    R369_2_I_RB_SP_1_14 AT %MW84091.14 : BOOL; (* R369_2_I_RB_SP_1_14 *)
    R369_2_I_RB_SP_1_15 AT %MW84091.15 : BOOL; (* R369_2_I_RB_SP_1_15 *)
    R369_2_I_RB_TC_이상 AT %MW84092.8 : BOOL; (* R369_2_I_RB_TC_이상 *)
    R369_2_I_RB_TIP_CHANGE AT %MW84093.13 : BOOL; (* R369_2_I_RB_TIP_CHANGE *)
    R369_2_I_RB_TIP_DRESSING AT %MW84090.7 : BOOL; (* R369_2_I_RB_TIP_DRESSING *)
    R369_2_I_RB__PLT_카운터리셋완료 AT %MW84093.10 : BOOL; (* R369_2_I_RB__PLT_카운터리셋완료 *)
    R369_2_I_RB_공기압_이상 AT %MW84092.9 : BOOL; (* R369_2_I_RB_공기압_이상 *)
    R369_2_I_RB_냉각수_이상 AT %MW84092.10 : BOOL; (* R369_2_I_RB_냉각수_이상 *)
    R369_2_I_RB_비상정지_NC AT %MW84090.8 : BOOL; (* R369_2_I_RB_비상정지_NC *)
    R369_2_I_RB_비전이상 AT %MW84092.14 : BOOL; (* R369_2_I_RB_비전이상 *)
    R369_2_I_RB_상호인터록_INT1 AT %MW84093.0 : BOOL; (* R369_2_I_RB_상호인터록_INT1 *)
    R369_2_I_RB_상호인터록_INT2 AT %MW84093.1 : BOOL; (* R369_2_I_RB_상호인터록_INT2 *)
    R369_2_I_RB_상호인터록_INT3 AT %MW84093.2 : BOOL; (* R369_2_I_RB_상호인터록_INT3 *)
    R369_2_I_RB_상호인터록_INT4 AT %MW84093.3 : BOOL; (* R369_2_I_RB_상호인터록_INT4 *)
    R369_2_I_RB_상호인터록_INT5 AT %MW84093.4 : BOOL; (* R369_2_I_RB_상호인터록_INT5 *)
    R369_2_I_RB_상호인터록_INT6 AT %MW84093.5 : BOOL; (* R369_2_I_RB_상호인터록_INT6 *)
    R369_2_I_RB_상호인터록_INT7 AT %MW84093.6 : BOOL; (* R369_2_I_RB_상호인터록_INT7 *)
    R369_2_I_RB_상호인터록_INT8 AT %MW84093.7 : BOOL; (* R369_2_I_RB_상호인터록_INT8 *)
    R369_2_I_RB_실러이상 AT %MW84092.13 : BOOL; (* R369_2_I_RB_실러이상 *)
    R369_2_I_RB_용접카운터이상 AT %MW84092.15 : BOOL; (* R369_2_I_RB_용접카운터이상 *)
    R369_2_I_RB_용접타점수 AT %MW84095 : WORD; (* R369_2_I_RB_용접타점수 *)
    R369_2_I_RB_운전준비 AT %MW84090.3 : BOOL; (* R369_2_I_RB_운전준비 *)
    R369_2_I_RB_원위치 AT %MW84090.0 : BOOL; (* R369_2_I_RB_원위치 *)
    R369_2_I_RB_이상리셋 AT %MW84090.2 : BOOL; (* R369_2_I_RB_이상리셋 *)
    R369_2_I_RB_자동 AT %MW84090.4 : BOOL; (* R369_2_I_RB_자동 *)
    R369_2_I_RB_자동기동 AT %MW84090.5 : BOOL; (* R369_2_I_RB_자동기동 *)
    R369_2_I_RB_최종_작업완료 AT %MW84090.1 : BOOL; (* R369_2_I_RB_최종_작업완료 *)
    R369_2_I_RB_통신이상 AT %MW84092.12 : BOOL; (* R369_2_I_RB_통신이상 *)
    R369_2_M_I_RB_1차_작업완료 AT %MW20091.2 : BOOL; (* R369_2_M_I_RB_1차_작업완료 *)
    R369_2_M_I_RB_2차_작업완료 AT %MW20091.3 : BOOL; (* R369_2_M_I_RB_2차_작업완료 *)
    R369_2_M_I_RB_3차_작업완료 AT %MW20091.4 : BOOL; (* R369_2_M_I_RB_3차_작업완료 *)
    R369_2_M_I_RB_4차_작업완료 AT %MW20091.5 : BOOL; (* R369_2_M_I_RB_4차_작업완료 *)
    R369_2_M_I_RB_5차_작업완료 AT %MW20091.6 : BOOL; (* R369_2_M_I_RB_5차_작업완료 *)
    R369_2_M_I_RB_6차_작업완료 AT %MW20091.7 : BOOL; (* R369_2_M_I_RB_6차_작업완료 *)
    R369_2_M_I_RB_7차_작업완료 AT %MW20091.8 : BOOL; (* R369_2_M_I_RB_7차_작업완료 *)
    R369_2_M_I_RB_PAUSE_보조 AT %MW20090.5 : BOOL; (* R369_2_M_I_RB_PAUSE_보조 *)
    R369_2_M_I_RB_PLC_RUN_CHK_이상 AT %MW20090.7 : BOOL; (* R369_2_M_I_RB_PLC_RUN_CHK_이상 *)
    R369_2_M_I_RB_간섭무_1 AT %MW20092.0 : BOOL; (* R369_2_M_I_RB_간섭무_1 *)
    R369_2_M_I_RB_간섭무_10 AT %MW20092.9 : BOOL; (* R369_2_M_I_RB_간섭무_10 *)
    R369_2_M_I_RB_간섭무_11 AT %MW20092.10 : BOOL; (* R369_2_M_I_RB_간섭무_11 *)
    R369_2_M_I_RB_간섭무_12 AT %MW20092.11 : BOOL; (* R369_2_M_I_RB_간섭무_12 *)
    R369_2_M_I_RB_간섭무_2 AT %MW20092.1 : BOOL; (* R369_2_M_I_RB_간섭무_2 *)
    R369_2_M_I_RB_간섭무_3 AT %MW20092.2 : BOOL; (* R369_2_M_I_RB_간섭무_3 *)
    R369_2_M_I_RB_간섭무_4 AT %MW20092.3 : BOOL; (* R369_2_M_I_RB_간섭무_4 *)
    R369_2_M_I_RB_간섭무_5 AT %MW20092.4 : BOOL; (* R369_2_M_I_RB_간섭무_5 *)
    R369_2_M_I_RB_간섭무_6 AT %MW20092.5 : BOOL; (* R369_2_M_I_RB_간섭무_6 *)
    R369_2_M_I_RB_간섭무_7 AT %MW20092.6 : BOOL; (* R369_2_M_I_RB_간섭무_7 *)
    R369_2_M_I_RB_간섭무_8 AT %MW20092.7 : BOOL; (* R369_2_M_I_RB_간섭무_8 *)
    R369_2_M_I_RB_간섭무_9 AT %MW20092.8 : BOOL; (* R369_2_M_I_RB_간섭무_9 *)
    R369_2_M_I_RB_비상정지 AT %MW20090.4 : BOOL; (* R369_2_M_I_RB_비상정지 *)
    R369_2_M_I_RB_운전준비 AT %MW20090.0 : BOOL; (* R369_2_M_I_RB_운전준비 *)
    R369_2_M_I_RB_원위치 AT %MW20090.3 : BOOL; (* R369_2_M_I_RB_원위치 *)
    R369_2_M_I_RB_이상 AT %MW20090.2 : BOOL; (* R369_2_M_I_RB_이상 *)
    R369_2_M_I_RB_자동 AT %MW20090.1 : BOOL; (* R369_2_M_I_RB_자동 *)
    R369_2_M_I_RB_최종작업완료 AT %MW20091.0 : BOOL; (* R369_2_M_I_RB_최종작업완료 *)
    R369_2_M_I_RB_프로그램_이상 AT %MW20090.6 : BOOL; (* R369_2_M_I_RB_프로그램_이상 *)
    R369_2_M_O_RB_1_CYCLE_SET AT %MW21090.3 : BOOL; (* R369_2_M_O_RB_1_CYCLE_SET *)
    R369_2_M_O_RB_1_CYCLE_리셋 AT %MW21090.4 : BOOL; (* R369_2_M_O_RB_1_CYCLE_리셋 *)
    R369_2_M_O_RB_1차_작업완료_리셋 AT %MW21092.0 : BOOL; (* R369_2_M_O_RB_1차_작업완료_리셋 *)
    R369_2_M_O_RB_2차_작업완료_리셋 AT %MW21092.1 : BOOL; (* R369_2_M_O_RB_2차_작업완료_리셋 *)
    R369_2_M_O_RB_2차_진입OK AT %MW21091.8 : BOOL; (* R369_2_M_O_RB_2차_진입OK *)
    R369_2_M_O_RB_3차_작업완료_리셋 AT %MW21092.2 : BOOL; (* R369_2_M_O_RB_3차_작업완료_리셋 *)
    R369_2_M_O_RB_3차_진입OK AT %MW21091.9 : BOOL; (* R369_2_M_O_RB_3차_진입OK *)
    R369_2_M_O_RB_4차_작업완료_리셋 AT %MW21092.3 : BOOL; (* R369_2_M_O_RB_4차_작업완료_리셋 *)
    R369_2_M_O_RB_4차_진입OK AT %MW21091.10 : BOOL; (* R369_2_M_O_RB_4차_진입OK *)
    R369_2_M_O_RB_5차_작업완료_리셋 AT %MW21092.4 : BOOL; (* R369_2_M_O_RB_5차_작업완료_리셋 *)
    R369_2_M_O_RB_5차_진입OK AT %MW21091.11 : BOOL; (* R369_2_M_O_RB_5차_진입OK *)
    R369_2_M_O_RB_6차_작업완료_리셋 AT %MW21092.5 : BOOL; (* R369_2_M_O_RB_6차_작업완료_리셋 *)
    R369_2_M_O_RB_6차_진입OK AT %MW21091.12 : BOOL; (* R369_2_M_O_RB_6차_진입OK *)
    R369_2_M_O_RB_7차_작업완료_리셋 AT %MW21092.6 : BOOL; (* R369_2_M_O_RB_7차_작업완료_리셋 *)
    R369_2_M_O_RB_7차_진입OK AT %MW21091.13 : BOOL; (* R369_2_M_O_RB_7차_진입OK *)
    R369_2_M_O_RB_ATD_OK AT %MW21090.6 : BOOL; (* R369_2_M_O_RB_ATD_OK *)
    R369_2_M_O_RB_PLT_10_진입OK AT %MW21093.10 : BOOL; (* R369_2_M_O_RB_PLT_10_진입OK *)
    R369_2_M_O_RB_PLT_11_진입OK AT %MW21093.11 : BOOL; (* R369_2_M_O_RB_PLT_11_진입OK *)
    R369_2_M_O_RB_PLT_12_진입OK AT %MW21093.12 : BOOL; (* R369_2_M_O_RB_PLT_12_진입OK *)
    R369_2_M_O_RB_PLT_1_진입OK AT %MW21093.1 : BOOL; (* R369_2_M_O_RB_PLT_1_진입OK *)
    R369_2_M_O_RB_PLT_2_진입OK AT %MW21093.2 : BOOL; (* R369_2_M_O_RB_PLT_2_진입OK *)
    R369_2_M_O_RB_PLT_3_진입OK AT %MW21093.3 : BOOL; (* R369_2_M_O_RB_PLT_3_진입OK *)
    R369_2_M_O_RB_PLT_4_진입OK AT %MW21093.4 : BOOL; (* R369_2_M_O_RB_PLT_4_진입OK *)
    R369_2_M_O_RB_PLT_5_진입OK AT %MW21093.5 : BOOL; (* R369_2_M_O_RB_PLT_5_진입OK *)
    R369_2_M_O_RB_PLT_6_진입OK AT %MW21093.6 : BOOL; (* R369_2_M_O_RB_PLT_6_진입OK *)
    R369_2_M_O_RB_PLT_7_진입OK AT %MW21093.7 : BOOL; (* R369_2_M_O_RB_PLT_7_진입OK *)
    R369_2_M_O_RB_PLT_8_진입OK AT %MW21093.8 : BOOL; (* R369_2_M_O_RB_PLT_8_진입OK *)
    R369_2_M_O_RB_PLT_9_진입OK AT %MW21093.9 : BOOL; (* R369_2_M_O_RB_PLT_9_진입OK *)
    R369_2_M_O_RB_PLT_카운터리셋_보조 AT %MW21090.10 : BOOL; (* R369_2_M_O_RB_PLT_카운터리셋_보조 *)
    R369_2_M_O_RB_PROG_NO AT %MW21094 : WORD;
    R369_2_M_O_RB_RESTART_OK AT %MW21090.2 : BOOL; (* R369_2_M_O_RB_RESTART_OK *)
    R369_2_M_O_RB_START_OK AT %MW21090.0 : BOOL; (* R369_2_M_O_RB_START_OK *)
    R369_2_M_O_RB_TEST_MODE_5000회 AT %MW21090.12 : BOOL; (* R369_2_M_O_RB_TEST_MODE_5000회 *)
    R369_2_M_O_RB_TIP_교체_시작 AT %MW21090.7 : BOOL; (* R369_2_M_O_RB_TIP_교체_시작 *)
    R369_2_M_O_RB_TIP_교체_완료 AT %MW21090.8 : BOOL; (* R369_2_M_O_RB_TIP_교체_완료 *)
    R369_2_M_O_RB_VIP_MODE AT %MW21090.11 : BOOL; (* R369_2_M_O_RB_VIP_MODE *)
    R369_2_M_O_RB_냉각수_차단_요청 AT %MW21090.9 : BOOL; (* R369_2_M_O_RB_냉각수_차단_요청 *)
    R369_2_M_O_RB_진입OK_AX차종 AT %MW21091.0 : BOOL; (* R369_2_M_O_RB_진입OK_AX차종 *)
    R369_2_M_O_RB_진입OK_B차종 AT %MW21091.1 : BOOL; (* R369_2_M_O_RB_진입OK_B차종 *)
    R369_2_M_O_RB_진입OK_C차종 AT %MW21091.2 : BOOL; (* R369_2_M_O_RB_진입OK_C차종 *)
    R369_2_M_O_RB_진입OK_D차종 AT %MW21091.3 : BOOL; (* R369_2_M_O_RB_진입OK_D차종 *)
    R369_2_M_O_RB_진입OK_E차종 AT %MW21091.4 : BOOL; (* R369_2_M_O_RB_진입OK_E차종 *)
    R369_2_M_O_RB_진입OK_F차종 AT %MW21091.5 : BOOL; (* R369_2_M_O_RB_진입OK_F차종 *)
    R369_2_M_O_RB_진입OK_G차종 AT %MW21091.6 : BOOL; (* R369_2_M_O_RB_진입OK_G차종 *)
    R369_2_M_O_RB_진입OK_H차종 AT %MW21091.7 : BOOL; (* R369_2_M_O_RB_진입OK_H차종 *)
    R369_2_M_O_RB_최종_작업완료_리셋 AT %MW21090.5 : BOOL; (* R369_2_M_O_RB_최종_작업완료_리셋 *)
    R369_2_M_O_RB_프로그램_OK AT %MW21090.1 : BOOL; (* R369_2_M_O_RB_프로그램_OK *)
    R369_2_O_RB_0_5S_통신_CHK AT %MW94093.14 : BOOL; (* R369_2_O_RB_0_5S_통신_CHK *)
    R369_2_O_RB_2차_진입OK AT %MW94091.8 : BOOL; (* R369_2_O_RB_2차_진입OK *)
    R369_2_O_RB_3차_진입OK AT %MW94091.9 : BOOL; (* R369_2_O_RB_3차_진입OK *)
    R369_2_O_RB_4차_진입OK AT %MW94091.10 : BOOL; (* R369_2_O_RB_4차_진입OK *)
    R369_2_O_RB_5차_진입OK AT %MW94091.11 : BOOL; (* R369_2_O_RB_5차_진입OK *)
    R369_2_O_RB_6차_진입OK AT %MW94091.12 : BOOL; (* R369_2_O_RB_6차_진입OK *)
    R369_2_O_RB_7차_진입OK AT %MW94091.13 : BOOL; (* R369_2_O_RB_7차_진입OK *)
    R369_2_O_RB_AX_1차_진입OK AT %MW94091.0 : BOOL; (* R369_2_O_RB_AX_1차_진입OK *)
    R369_2_O_RB_B_1차_진입OK AT %MW94091.1 : BOOL; (* R369_2_O_RB_B_1차_진입OK *)
    R369_2_O_RB_C_1차_진입OK AT %MW94091.2 : BOOL; (* R369_2_O_RB_C_1차_진입OK *)
    R369_2_O_RB_D_1차_진입OK AT %MW94091.3 : BOOL; (* R369_2_O_RB_D_1차_진입OK *)
    R369_2_O_RB_EACH_작업완료_리셋 AT %MW94090.14 : BOOL; (* R369_2_O_RB_EACH_작업완료_리셋 *)
    R369_2_O_RB_EXT_READY AT %MW94090.11 : BOOL; (* R369_2_O_RB_EXT_READY *)
    R369_2_O_RB_E_1차_진입OK AT %MW94091.4 : BOOL; (* R369_2_O_RB_E_1차_진입OK *)
    R369_2_O_RB_F_1차_진입OK AT %MW94091.5 : BOOL; (* R369_2_O_RB_F_1차_진입OK *)
    R369_2_O_RB_GATE_OPEN_NC AT %MW94093.11 : BOOL; (* R369_2_O_RB_GATE_OPEN_NC *)
    R369_2_O_RB_G_1차_진입OK AT %MW94091.6 : BOOL; (* R369_2_O_RB_G_1차_진입OK *)
    R369_2_O_RB_H_1차_진입OK AT %MW94091.7 : BOOL; (* R369_2_O_RB_H_1차_진입OK *)
    R369_2_O_RB_OUTPUT AT %MW94090 : ARRAY[0..3] OF WORD; (* R369_2_O_RB_OUTPUT *)
    R369_2_O_RB_PAUSE_NC AT %MW94090.13 : BOOL; (* R369_2_O_RB_PAUSE_NC *)
    R369_2_O_RB_PLT10_진입OK AT %MW94092.9 : BOOL; (* R369_2_O_RB_PLT10_진입OK *)
    R369_2_O_RB_PLT11_진입OK AT %MW94092.10 : BOOL; (* R369_2_O_RB_PLT11_진입OK *)
    R369_2_O_RB_PLT12_진입OK AT %MW94092.11 : BOOL; (* R369_2_O_RB_PLT12_진입OK *)
    R369_2_O_RB_PLT1_진입OK AT %MW94092.0 : BOOL; (* R369_2_O_RB_PLT1_진입OK *)
    R369_2_O_RB_PLT2_진입OK AT %MW94092.1 : BOOL; (* R369_2_O_RB_PLT2_진입OK *)
    R369_2_O_RB_PLT3_진입OK AT %MW94092.2 : BOOL; (* R369_2_O_RB_PLT3_진입OK *)
    R369_2_O_RB_PLT4_진입OK AT %MW94092.3 : BOOL; (* R369_2_O_RB_PLT4_진입OK *)
    R369_2_O_RB_PLT5_진입OK AT %MW94092.4 : BOOL; (* R369_2_O_RB_PLT5_진입OK *)
    R369_2_O_RB_PLT6_진입OK AT %MW94092.5 : BOOL; (* R369_2_O_RB_PLT6_진입OK *)
    R369_2_O_RB_PLT7_진입OK AT %MW94092.6 : BOOL; (* R369_2_O_RB_PLT7_진입OK *)
    R369_2_O_RB_PLT8_진입OK AT %MW94092.7 : BOOL; (* R369_2_O_RB_PLT8_진입OK *)
    R369_2_O_RB_PLT9_진입OK AT %MW94092.8 : BOOL; (* R369_2_O_RB_PLT9_진입OK *)
    R369_2_O_RB_PLT_카운터_리셋_요구 AT %MW94093.10 : BOOL; (* R369_2_O_RB_PLT_카운터_리셋_요구 *)
    R369_2_O_RB_PROG_선택1 AT %MW94090.0 : BOOL; (* R369_2_O_RB_PROG_선택1 *)
    R369_2_O_RB_PROG_선택128 AT %MW94090.7 : BOOL; (* R369_2_O_RB_PROG_선택128 *)
    R369_2_O_RB_PROG_선택16 AT %MW94090.4 : BOOL; (* R369_2_O_RB_PROG_선택16 *)
    R369_2_O_RB_PROG_선택2 AT %MW94090.1 : BOOL; (* R369_2_O_RB_PROG_선택2 *)
    R369_2_O_RB_PROG_선택32 AT %MW94090.5 : BOOL; (* R369_2_O_RB_PROG_선택32 *)
    R369_2_O_RB_PROG_선택4 AT %MW94090.2 : BOOL; (* R369_2_O_RB_PROG_선택4 *)
    R369_2_O_RB_PROG_선택64 AT %MW94090.6 : BOOL; (* R369_2_O_RB_PROG_선택64 *)
    R369_2_O_RB_PROG_선택8 AT %MW94090.3 : BOOL; (* R369_2_O_RB_PROG_선택8 *)
    R369_2_O_RB_SP_1_14 AT %MW94091.14 : BOOL; (* R369_2_O_RB_SP_1_14 *)
    R369_2_O_RB_SP_1_15 AT %MW94091.15 : BOOL; (* R369_2_O_RB_SP_1_15 *)
    R369_2_O_RB_SP_2_12 AT %MW94092.12 : BOOL; (* R369_2_O_RB_SP_2_12 *)
    R369_2_O_RB_SP_2_13 AT %MW94092.13 : BOOL; (* R369_2_O_RB_SP_2_13 *)
    R369_2_O_RB_SP_2_14 AT %MW94092.14 : BOOL; (* R369_2_O_RB_SP_2_14 *)
    R369_2_O_RB_SP_5000TH_ON AT %MW94092.15 : BOOL; (* R369_2_O_RB_SP_5000TH_ON *)
    R369_2_O_RB_TIP_CHANGE_END AT %MW94093.9 : BOOL; (* R369_2_O_RB_TIP_CHANGE_END *)
    R369_2_O_RB_TIP_CHANGE_START AT %MW94093.8 : BOOL; (* R369_2_O_RB_TIP_CHANGE_START *)
    R369_2_O_RB_TIP_DRESS_SATRT AT %MW94090.12 : BOOL; (* R369_2_O_RB_TIP_DRESS_SATRT *)
    R369_2_O_RB_VIP_MODE AT %MW94093.15 : BOOL; (* R369_2_O_RB_VIP_MODE *)
    R369_2_O_RB_기동 AT %MW94090.9 : BOOL; (* R369_2_O_RB_기동 *)
    R369_2_O_RB_냉각수차단 AT %MW94090.15 : BOOL; (* R369_2_O_RB_냉각수차단 *)
    R369_2_O_RB_부저정지 AT %MW94093.13 : BOOL; (* R369_2_O_RB_부저정지 *)
    R369_2_O_RB_비상정지_NC AT %MW94093.12 : BOOL; (* R369_2_O_RB_비상정지_NC *)
    R369_2_O_RB_상호인터록_INT1 AT %MW94093.0 : BOOL; (* R369_2_O_RB_상호인터록_INT1 *)
    R369_2_O_RB_상호인터록_INT2 AT %MW94093.1 : BOOL; (* R369_2_O_RB_상호인터록_INT2 *)
    R369_2_O_RB_상호인터록_INT3 AT %MW94093.2 : BOOL; (* R369_2_O_RB_상호인터록_INT3 *)
    R369_2_O_RB_상호인터록_INT4 AT %MW94093.3 : BOOL; (* R369_2_O_RB_상호인터록_INT4 *)
    R369_2_O_RB_상호인터록_INT5 AT %MW94093.4 : BOOL; (* R369_2_O_RB_상호인터록_INT5 *)
    R369_2_O_RB_상호인터록_INT6 AT %MW94093.5 : BOOL; (* R369_2_O_RB_상호인터록_INT6 *)
    R369_2_O_RB_상호인터록_INT7 AT %MW94093.6 : BOOL; (* R369_2_O_RB_상호인터록_INT7 *)
    R369_2_O_RB_상호인터록_INT8 AT %MW94093.7 : BOOL; (* R369_2_O_RB_상호인터록_INT8 *)
    R369_2_O_RB_이상_리셋 AT %MW94090.10 : BOOL; (* R369_2_O_RB_이상_리셋 *)
    R369_2_O_RB_작업완료_리셋 AT %MW94090.8 : BOOL; (* R369_2_O_RB_작업완료_리셋 *)
    ROOF_RACK1_3_PLC_BOX_CP_TRIP AT %MW87401.15 : BOOL; (* ROOF RACK1 3 PLC BOX CP TRIP *)
    ROOF_RACK1_LC_정상1 AT %MW87403.0 : BOOL; (* ROOF RACK1 LC 정상1 *)
    ROOF_RACK1_LC_정상2 AT %MW87403.1 : BOOL; (* ROOF RACK1 LC 정상2 *)
    ROOF_RACK1_PRS_랙감지1 AT %MW87400.0 : BOOL; (* ROOF RACK1 PRS 랙감지1 *)
    ROOF_RACK1_PRS_랙감지2 AT %MW87400.1 : BOOL; (* ROOF RACK1 PRS 랙감지2 *)
    ROOF_RACK1_PRS_막장감지 AT %MW87400.2 : BOOL; (* ROOF RACK1 PRS 막장감지 *)
    ROOF_RACK1_발목감지_정상1 AT %MW87403.2 : BOOL; (* ROOF RACK1 발목감지 정상1 *)
    ROOF_RACK1_발목감지_정상2 AT %MW87403.3 : BOOL; (* ROOF RACK1 발목감지 정상2 *)
    ROOF_RACK2_LC_정상1 AT %MW87403.4 : BOOL; (* ROOF RACK2 LC 정상1 *)
    ROOF_RACK2_LC_정상2 AT %MW87403.5 : BOOL; (* ROOF RACK2 LC 정상2 *)
    ROOF_RACK2_PRS_랙감지1 AT %MW87400.8 : BOOL; (* ROOF RACK2 PRS 랙감지1 *)
    ROOF_RACK2_PRS_랙감지2 AT %MW87400.9 : BOOL; (* ROOF RACK2 PRS 랙감지2 *)
    ROOF_RACK2_PRS_막장감지 AT %MW87400.10 : BOOL; (* ROOF RACK2 PRS 막장감지 *)
    ROOF_RACK2_발목감지_정상1 AT %MW87403.6 : BOOL; (* ROOF RACK2 발목감지 정상1 *)
    ROOF_RACK2_발목감지_정상2 AT %MW87403.7 : BOOL; (* ROOF RACK2 발목감지 정상2 *)
    ROOF_RACK3_LC_정상1 AT %MW87403.8 : BOOL; (* ROOF RACK3 LC 정상1 *)
    ROOF_RACK3_LC_정상2 AT %MW87403.9 : BOOL; (* ROOF RACK3 LC 정상2 *)
    ROOF_RACK3_PRS_랙감지1 AT %MW87401.0 : BOOL; (* ROOF RACK3 PRS 랙감지1 *)
    ROOF_RACK3_PRS_랙감지2 AT %MW87401.1 : BOOL; (* ROOF RACK3 PRS 랙감지2 *)
    ROOF_RACK3_PRS_막장감지 AT %MW87401.2 : BOOL; (* ROOF RACK3 PRS 막장감지 *)
    ROOF_RACK3_발목감지_정상1 AT %MW87403.10 : BOOL; (* ROOF RACK3 발목감지 정상1 *)
    ROOF_RACK3_발목감지_정상2 AT %MW87403.11 : BOOL; (* ROOF RACK3 발목감지 정상2 *)
    ROOF_RACK4_6_PLC_BOX_CP_TRIP AT %MW87451.15 : BOOL; (* ROOF RACK4 6 PLC BOX CP TRIP *)
    ROOF_RACK4_LC_정상1 AT %MW87453.0 : BOOL; (* ROOF RACK4 LC 정상1 *)
    ROOF_RACK4_LC_정상2 AT %MW87453.1 : BOOL; (* ROOF RACK4 LC 정상2 *)
    ROOF_RACK4_PRS_랙감지1 AT %MW87450.0 : BOOL; (* ROOF RACK4 PRS 랙감지1 *)
    ROOF_RACK4_PRS_랙감지2 AT %MW87450.1 : BOOL; (* ROOF RACK4 PRS 랙감지2 *)
    ROOF_RACK4_PRS_막장감지 AT %MW87450.2 : BOOL; (* ROOF RACK4 PRS 막장감지 *)
    ROOF_RACK4_발목감지_정상1 AT %MW87453.2 : BOOL; (* ROOF RACK4 발목감지 정상1 *)
    ROOF_RACK4_발목감지_정상2 AT %MW87453.3 : BOOL; (* ROOF RACK4 발목감지 정상2 *)
    ROOF_RACK5_LC_정상1 AT %MW87453.4 : BOOL; (* ROOF RACK5 LC 정상1 *)
    ROOF_RACK5_LC_정상2 AT %MW87453.5 : BOOL; (* ROOF RACK5 LC 정상2 *)
    ROOF_RACK5_PRS_랙감지1 AT %MW87450.8 : BOOL; (* ROOF RACK5 PRS 랙감지1 *)
    ROOF_RACK5_PRS_랙감지2 AT %MW87450.9 : BOOL; (* ROOF RACK5 PRS 랙감지2 *)
    ROOF_RACK5_PRS_막장감지 AT %MW87450.10 : BOOL; (* ROOF RACK5 PRS 막장감지 *)
    ROOF_RACK5_발목감지_정상1 AT %MW87453.6 : BOOL; (* ROOF RACK5 발목감지 정상1 *)
    ROOF_RACK5_발목감지_정상2 AT %MW87453.7 : BOOL; (* ROOF RACK5 발목감지 정상2 *)
    ROOF_RACK6_LC_정상1 AT %MW87453.8 : BOOL; (* ROOF RACK6 LC 정상1 *)
    ROOF_RACK6_LC_정상2 AT %MW87453.9 : BOOL; (* ROOF RACK6 LC 정상2 *)
    ROOF_RACK6_PRS_랙감지1 AT %MW87451.0 : BOOL; (* ROOF RACK6 PRS 랙감지1 *)
    ROOF_RACK6_PRS_랙감지2 AT %MW87451.1 : BOOL; (* ROOF RACK6 PRS 랙감지2 *)
    ROOF_RACK6_PRS_막장감지 AT %MW87451.2 : BOOL; (* ROOF RACK6 PRS 막장감지 *)
    ROOF_RACK6_발목감지_정상1 AT %MW87453.10 : BOOL; (* ROOF RACK6 발목감지 정상1 *)
    ROOF_RACK6_발목감지_정상2 AT %MW87453.11 : BOOL; (* ROOF RACK6 발목감지 정상2 *)
    S362_6_INV1_BRAKE_CR_ON AT %MW95014.7 : BOOL; (* S362_6_INV1_BRAKE_CR_ON *)
    S362_6_INV1_MC_BRAKE_ON AT %MW85010.1 : BOOL; (* S362_6_INV1_MC_BRAKE_ON *)
    S362_6_INV1_NFB_ON AT %MW85013.0 : BOOL; (* S362_6_INV1_NFB_ON *)
    S362_6_INV1_NOMAL_OK AT %MW85010.0 : BOOL; (* S362_6_INV1_NOMAL_OK *)
    S362_6_INV1_RETURN AT %MW95014.1 : BOOL; (* S362_6_INV1_RETURN *)
    S362_6_INV1_SAFETY1_ON AT %MW95014.5 : BOOL; (* S362_6_INV1_SAFETY1_ON *)
    S362_6_INV1_SAFETY2_ON AT %MW95014.6 : BOOL; (* S362_6_INV1_SAFETY2_ON *)
    S362_6_INV1_TURN AT %MW95014.0 : BOOL; (* S362_6_INV1_TURN *)
    S362_6_INV1_이상_리셋 AT %MW95014.3 : BOOL; (* S362_6_INV1_이상_리셋 *)
    S362_6_INV2_BRAKE_CR_ON AT %MW95014.15 : BOOL; (* S362_6_INV2_BRAKE_CR_ON *)
    S362_6_INV2_MC_BRAKE_ON AT %MW85010.5 : BOOL; (* S362_6_INV2_MC_BRAKE_ON *)
    S362_6_INV2_NFB_ON AT %MW85013.1 : BOOL; (* S362_6_INV2_NFB_ON *)
    S362_6_INV2_NOMAL_OK AT %MW85010.4 : BOOL; (* S362_6_INV2_NOMAL_OK *)
    S362_6_INV2_RETURN AT %MW95014.9 : BOOL; (* S362_6_INV2_RETURN *)
    S362_6_INV2_SAFETY1_ON AT %MW95014.13 : BOOL; (* S362_6_INV2_SAFETY1_ON *)
    S362_6_INV2_SAFETY2_ON AT %MW95014.14 : BOOL; (* S362_6_INV2_SAFETY2_ON *)
    S362_6_INV2_TURN AT %MW95014.8 : BOOL; (* S362_6_INV2_TURN *)
    S362_6_INV2_이상_리셋 AT %MW95014.11 : BOOL; (* S362_6_INV2_이상_리셋 *)
    S362_6_INV3_BRAKE_CR_ON AT %MW95015.7 : BOOL; (* S362_6_INV3_BRAKE_CR_ON *)
    S362_6_INV3_MC_BRAKE_ON AT %MW85010.9 : BOOL; (* S362_6_INV3_MC_BRAKE_ON *)
    S362_6_INV3_NFB_ON AT %MW85013.2 : BOOL; (* S362_6_INV3_NFB_ON *)
    S362_6_INV3_NOMAL_OK AT %MW85010.8 : BOOL; (* S362_6_INV3_NOMAL_OK *)
    S362_6_INV3_RETURN AT %MW95015.1 : BOOL; (* S362_6_INV3_RETURN *)
    S362_6_INV3_SAFETY1_ON AT %MW95015.5 : BOOL; (* S362_6_INV3_SAFETY1_ON *)
    S362_6_INV3_SAFETY2_ON AT %MW95015.6 : BOOL; (* S362_6_INV3_SAFETY2_ON *)
    S362_6_INV3_TURN AT %MW95015.0 : BOOL; (* S362_6_INV3_TURN *)
    S362_6_INV3_이상_리셋 AT %MW95015.3 : BOOL; (* S362_6_INV3_이상_리셋 *)
    S362_6_INV4_BRAKE_CR_ON AT %MW95015.15 : BOOL; (* S362_6_INV4_BRAKE_CR_ON *)
    S362_6_INV4_MC_BRAKE_ON AT %MW85010.13 : BOOL; (* S362_6_INV4_MC_BRAKE_ON *)
    S362_6_INV4_NFB_ON AT %MW85013.3 : BOOL; (* S362_6_INV4_NFB_ON *)
    S362_6_INV4_NOMAL_OK AT %MW85010.12 : BOOL; (* S362_6_INV4_NOMAL_OK *)
    S362_6_INV4_RETURN AT %MW95015.9 : BOOL; (* S362_6_INV4_RETURN *)
    S362_6_INV4_SAFETY1_ON AT %MW95015.13 : BOOL; (* S362_6_INV4_SAFETY1_ON *)
    S362_6_INV4_SAFETY2_ON AT %MW95015.14 : BOOL; (* S362_6_INV4_SAFETY2_ON *)
    S362_6_INV4_TURN AT %MW95015.8 : BOOL; (* S362_6_INV4_TURN *)
    S362_6_INV4_이상_리셋 AT %MW95015.11 : BOOL; (* S362_6_INV4_이상_리셋 *)
    S362_6_INV_BRAKE_CP_OFF AT %MW85013.13 : BOOL; (* S362_6_INV_BRAKE_CP_OFF *)
    S362_6_INV_DC_CP_TRIP AT %MW85013.12 : BOOL; (* S362_6_INV_DC_CP_TRIP *)
    S362_6_INV_PS1_DC_OK AT %MW85013.14 : BOOL; (* S362_6_INV_PS1_DC_OK *)
    S362_6_INV_SPD_NOMAL AT %MW85013.15 : BOOL; (* S362_6_INV_SPD_NOMAL *)
    S362_6_INV_제어_CP_OFF AT %MW85013.11 : BOOL; (* S362_6_INV_제어_CP_OFF *)
    S362_7_10_PLC_BOX_CP_TRIP AT %MW87102.15 : BOOL; (* S362_7_10_PLC_BOX_CP_TRIP *)
    S362_7_10_공기압_AIR_CHECK AT %MW87102.14 : BOOL; (* S362_7_10_공기압_AIR_CHECK *)
    S362_EPB_AX_비상정지1 AT %MW87105.0 : BOOL; (* S362_EPB_AX_비상정지1 *)
    S362_EPB_AX_비상정지2 AT %MW87105.1 : BOOL; (* S362_EPB_AX_비상정지2 *)
    S362_INDEX_LH_TURN_감지1 AT %MW87102.4 : BOOL; (* S362_INDEX_LH_TURN_감지1 *)
    S362_INDEX_LH_TURN_감지2 AT %MW87102.5 : BOOL; (* S362_INDEX_LH_TURN_감지2 *)
    S362_INDEX_LH_TURN_감지3 AT %MW87102.6 : BOOL; (* S362_INDEX_LH_TURN_감지3 *)
    S362_INDEX_LH_TURN_원점 AT %MW87102.7 : BOOL; (* S362_INDEX_LH_TURN_원점 *)
    S362_INDEX_RH_TURN_감지1 AT %MW87102.0 : BOOL; (* S362_INDEX_RH_TURN_감지1 *)
    S362_INDEX_RH_TURN_감지2 AT %MW87102.1 : BOOL; (* S362_INDEX_RH_TURN_감지2 *)
    S362_INDEX_RH_TURN_감지3 AT %MW87102.2 : BOOL; (* S362_INDEX_RH_TURN_감지3 *)
    S362_INDEX_RH_TURN_원점 AT %MW87102.3 : BOOL; (* S362_INDEX_RH_TURN_원점 *)
    S362_LC_정상1 AT %MW87105.3 : BOOL;
    S362_LC_정상2 AT %MW87105.4 : BOOL;
    S362_LH_CUT_OFF_BOX_ON AT %MW87102.10 : BOOL;
    S362_LS_AX_SLIDE_전진 AT %MW87100.8 : BOOL; (* S362_LS_AX_SLIDE_전진 *)
    S362_LS_AX_SLIDE_후진 AT %MW87100.9 : BOOL; (* S362_LS_AX_SLIDE_후진 *)
    S362_MAT_정상1 AT %MW87105.6 : BOOL;
    S362_MAT_정상2 AT %MW87105.7 : BOOL;
    S362_M_SLD_LOCK_전진_LAMP AT %MW11104 : WORD; (* S362_M_SLD_LOCK_전진_LAMP *)
    S362_M_SLD_LOCK_후진_LAMP AT %MW11105 : WORD; (* S362_M_SLD_LOCK_후진_LAMP *)
    S362_M_SLIDE_전진_LAMP AT %MW11102 : WORD; (* S362_M_SLIDE_전진_LAMP *)
    S362_M_SLIDE_후진_LAMP AT %MW11103 : WORD; (* S362_M_SLIDE_후진_LAMP *)
    S362_M_TURN_LOCK_전진_LAMP AT %MW11100 : WORD; (* S362_M_TURN_LOCK_전진_LAMP *)
    S362_M_TURN_LOCK_후진_LAMP AT %MW11101 : WORD; (* S362_M_TURN_LOCK_후진_LAMP *)
    S362_PB_AX_작업_완료 AT %MW87102.9 : BOOL; (* S362_PB_AX_작업_완료 *)
    S362_PRS_AX_COM_LH_CHECK AT %MW87101.1 : BOOL; (* S362_PRS_AX_COM_LH_CHECK *)
    S362_PRS_AX_COM_RH_CHECK AT %MW87101.0 : BOOL; (* S362_PRS_AX_COM_RH_CHECK *)
    S362_PRS_AX_GR_LH_CHECK AT %MW87101.3 : BOOL; (* S362_PRS_AX_GR_LH_CHECK *)
    S362_PRS_AX_GR_RH_CHECK AT %MW87101.2 : BOOL; (* S362_PRS_AX_GR_RH_CHECK *)
    S362_PRS_AX_RAIL_LH_CHECK AT %MW87101.7 : BOOL; (* S362_PRS_AX_RAIL_LH_CHECK *)
    S362_PRS_AX_RAIL_RH_CHECK AT %MW87101.6 : BOOL; (* S362_PRS_AX_RAIL_RH_CHECK *)
    S362_PRS_AX_SR_LH_CHECK AT %MW87101.5 : BOOL; (* S362_PRS_AX_SR_LH_CHECK *)
    S362_PRS_AX_SR_RH_CHECK AT %MW87101.4 : BOOL; (* S362_PRS_AX_SR_RH_CHECK *)
    S362_RH_CUT_OFF_BOX_ON AT %MW87102.11 : BOOL;
    S362_RS_FRT_SLD_LOCK_전진 AT %MW87100.4 : BOOL; (* S362_RS_FRT_SLD_LOCK_전진 *)
    S362_RS_FRT_SLD_LOCK_후진 AT %MW87100.5 : BOOL; (* S362_RS_FRT_SLD_LOCK_후진 *)
    S362_RS_LH_IDX_LOCK_전진 AT %MW87100.2 : BOOL; (* S362_RS_LH_IDX_LOCK_전진 *)
    S362_RS_LH_IDX_LOCK_후진 AT %MW87100.3 : BOOL; (* S362_RS_LH_IDX_LOCK_후진 *)
    S362_RS_RH_IDX_LOCK_전진 AT %MW87100.0 : BOOL; (* S362_RS_RH_IDX_LOCK_전진 *)
    S362_RS_RH_IDX_LOCK_후진 AT %MW87100.1 : BOOL; (* S362_RS_RH_IDX_LOCK_후진 *)
    S362_RS_RR_SLD_LOCK_전진 AT %MW87100.6 : BOOL; (* S362_RS_RR_SLD_LOCK_전진 *)
    S362_RS_RR_SLD_LOCK_후진 AT %MW87100.7 : BOOL; (* S362_RS_RR_SLD_LOCK_후진 *)
    S362_SOL_AX_BRAKE_ON AT %MW97103.6 : BOOL; (* S362_SOL_AX_BRAKE_ON *)
    S362_SOL_AX_SLIDE_전진 AT %MW97103.4 : BOOL; (* S362_SOL_AX_SLIDE_전진 *)
    S362_SOL_AX_SLIDE_후진 AT %MW97103.5 : BOOL; (* S362_SOL_AX_SLIDE_후진 *)
    S362_SOL_AX_SLI_LOCK_전진 AT %MW97103.2 : BOOL; (* S362_SOL_AX_SLI_LOCK_전진 *)
    S362_SOL_AX_SLI_LOCK_후진 AT %MW97103.3 : BOOL; (* S362_SOL_AX_SLI_LOCK_후진 *)
    S362_SOL_TURN_LOCK_전진 AT %MW97103.0 : BOOL; (* S362_SOL_TURN_LOCK_전진 *)
    S362_SOL_TURN_LOCK_후진 AT %MW97103.1 : BOOL; (* S362_SOL_TURN_LOCK_후진 *)
    S364_7_15_PLC_BOX_CP_TRIP AT %MW87152.15 : BOOL; (* S364_7_15_PLC_BOX_CP_TRIP *)
    S364_7_16_PLC_BOX_CP_TRIP AT %MW87162.15 : BOOL; (* S364_7_16_PLC_BOX_CP_TRIP *)
    S364_EPB_AX_비상정지1 AT %MW87155.0 : BOOL; (* S364_EPB_AX_비상정지1 *)
    S364_EPB_AX_비상정지2 AT %MW87155.1 : BOOL; (* S364_EPB_AX_비상정지2 *)
    S364_LC_정상1 AT %MW87165.3 : BOOL;
    S364_LC_정상2 AT %MW87165.4 : BOOL;
    S364_MAT_정상1 AT %MW87165.6 : BOOL;
    S364_MAT_정상2 AT %MW87165.7 : BOOL;
    S364_M_AX_CLAMP_전진_LAMP AT %MW11602 : WORD; (* S364_M_AX_CLAMP_전진_LAMP *)
    S364_M_AX_CLAMP_후진_LAMP AT %MW11603 : WORD; (* S364_M_AX_CLAMP_후진_LAMP *)
    S364_M_AX_LATCH_전진_LAMP AT %MW11600 : WORD; (* S364_M_AX_LATCH_전진_LAMP *)
    S364_M_AX_LATCH_후진_LAMP AT %MW11601 : WORD; (* S364_M_AX_LATCH_후진_LAMP *)
    S364_M_AX_LH_SLD_CLP_전진_LAMP AT %MW11606 : WORD; (* S364_M_AX_LH_SLD_CLP_전진_LAMP *)
    S364_M_AX_LH_SLD_CLP_후진_LAMP AT %MW11607 : WORD; (* S364_M_AX_LH_SLD_CLP_후진_LAMP *)
    S364_M_AX_LH_SLD_LAT_전진_LAMP AT %MW11604 : WORD; (* S364_M_AX_LH_SLD_LAT_전진_LAMP *)
    S364_M_AX_LH_SLD_LAT_후진_LAMP AT %MW11605 : WORD; (* S364_M_AX_LH_SLD_LAT_후진_LAMP *)
    S364_M_AX_LH_SLD_전진_LAMP AT %MW11614 : WORD; (* S364_M_AX_LH_SLD_전진_LAMP *)
    S364_M_AX_LH_SLD_후진_LAMP AT %MW11615 : WORD; (* S364_M_AX_LH_SLD_후진_LAMP *)
    S364_M_AX_RH_SLD_CLP_전진_LAMP AT %MW11622 : WORD; (* S364_M_AX_RH_SLD_CLP_전진_LAMP *)
    S364_M_AX_RH_SLD_CLP_후진_LAMP AT %MW11623 : WORD; (* S364_M_AX_RH_SLD_CLP_후진_LAMP *)
    S364_M_AX_RH_SLD_LAT_전진_LAMP AT %MW11620 : WORD; (* S364_M_AX_RH_SLD_LAT_전진_LAMP *)
    S364_M_AX_RH_SLD_LAT_후진_LAMP AT %MW11621 : WORD; (* S364_M_AX_RH_SLD_LAT_후진_LAMP *)
    S364_M_AX_RH_SLD_전진_LAMP AT %MW11630 : WORD; (* S364_M_AX_RH_SLD_전진_LAMP *)
    S364_M_AX_RH_SLD_후진_LAMP AT %MW11631 : WORD; (* S364_M_AX_RH_SLD_후진_LAMP *)
    S364_PB_AX_작업_완료 AT %MW87152.9 : BOOL; (* S364_PB_AX_작업_완료 *)
    S364_PRS_AX_LH_RACK_CHK1 AT %MW87162.0 : BOOL; (* S364_PRS_AX_LH_RACK_CHK1 *)
    S364_PRS_AX_LH_RACK_CHK2 AT %MW87162.1 : BOOL; (* S364_PRS_AX_LH_RACK_CHK2 *)
    S364_PRS_AX_LH_RACK_CHK3 AT %MW87162.2 : BOOL; (* S364_PRS_AX_LH_RACK_CHK3 *)
    S364_PRS_AX_LH_ROOF_FRT_CHK AT %MW87162.3 : BOOL; (* S364_PRS_AX_LH_ROOF_FRT_CHK *)
    S364_PRS_AX_LH_ROOF_RR_CHK AT %MW87162.4 : BOOL; (* S364_PRS_AX_LH_ROOF_RR_CHK *)
    S364_PRS_AX_RH_RACK_CHK1 AT %MW87152.0 : BOOL; (* S364_PRS_AX_RH_RACK_CHK1 *)
    S364_PRS_AX_RH_RACK_CHK2 AT %MW87152.1 : BOOL; (* S364_PRS_AX_RH_RACK_CHK2 *)
    S364_PRS_AX_RH_RACK_CHK3 AT %MW87152.2 : BOOL; (* S364_PRS_AX_RH_RACK_CHK3 *)
    S364_PRS_AX_RH_ROOF_FRT_CHK AT %MW87152.3 : BOOL; (* S364_PRS_AX_RH_ROOF_FRT_CHK *)
    S364_PRS_AX_RH_ROOF_RR_CHK AT %MW87152.4 : BOOL; (* S364_PRS_AX_RH_ROOF_RR_CHK *)
    S364_RS_AX_LH_CLAMP_후진1 AT %MW87160.3 : BOOL; (* S364_RS_AX_LH_CLAMP_후진1 *)
    S364_RS_AX_LH_CLAMP_후진2 AT %MW87160.4 : BOOL; (* S364_RS_AX_LH_CLAMP_후진2 *)
    S364_RS_AX_LH_LATCH_후진1 AT %MW87160.0 : BOOL; (* S364_RS_AX_LH_LATCH_후진1 *)
    S364_RS_AX_LH_LATCH_후진2 AT %MW87160.1 : BOOL; (* S364_RS_AX_LH_LATCH_후진2 *)
    S364_RS_AX_LH_SLD_CLP_전진 AT %MW87161.0 : BOOL; (* S364_RS_AX_LH_SLD_CLP_전진 *)
    S364_RS_AX_LH_SLD_CLP_후진1 AT %MW87161.1 : BOOL; (* S364_RS_AX_LH_SLD_CLP_후진1 *)
    S364_RS_AX_LH_SLD_CLP_후진2 AT %MW87161.2 : BOOL; (* S364_RS_AX_LH_SLD_CLP_후진2 *)
    S364_RS_AX_LH_SLD_CLP_후진3 AT %MW87161.3 : BOOL; (* S364_RS_AX_LH_SLD_CLP_후진3 *)
    S364_RS_AX_LH_SLD_CLP_후진4 AT %MW87161.4 : BOOL; (* S364_RS_AX_LH_SLD_CLP_후진4 *)
    S364_RS_AX_LH_SLD_LAT_전진 AT %MW87160.8 : BOOL; (* S364_RS_AX_LH_SLD_LAT_전진 *)
    S364_RS_AX_LH_SLD_LAT_후진1 AT %MW87160.9 : BOOL; (* S364_RS_AX_LH_SLD_LAT_후진1 *)
    S364_RS_AX_LH_SLD_LAT_후진2 AT %MW87160.10 : BOOL; (* S364_RS_AX_LH_SLD_LAT_후진2 *)
    S364_RS_AX_LH_SLD_LAT_후진3 AT %MW87160.11 : BOOL; (* S364_RS_AX_LH_SLD_LAT_후진3 *)
    S364_RS_AX_LH_SLD_LAT_후진4 AT %MW87160.12 : BOOL; (* S364_RS_AX_LH_SLD_LAT_후진4 *)
    S364_RS_AX_LH_SLIDE_전진 AT %MW87151.8 : BOOL; (* S364_RS_AX_LH_SLIDE_전진 *)
    S364_RS_AX_LH_SLIDE_후진 AT %MW87151.9 : BOOL; (* S364_RS_AX_LH_SLIDE_후진 *)
    S364_RS_AX_RH_CLAMP_전진 AT %MW87150.4 : BOOL; (* S364_RS_AX_RH_CLAMP_전진 *)
    S364_RS_AX_RH_CLAMP_후진1 AT %MW87150.5 : BOOL; (* S364_RS_AX_RH_CLAMP_후진1 *)
    S364_RS_AX_RH_CLAMP_후진2 AT %MW87150.6 : BOOL; (* S364_RS_AX_RH_CLAMP_후진2 *)
    S364_RS_AX_RH_LATCH_전진 AT %MW87150.0 : BOOL; (* S364_RS_AX_RH_LATCH_전진 *)
    S364_RS_AX_RH_LATCH_후진1 AT %MW87150.1 : BOOL; (* S364_RS_AX_RH_LATCH_후진1 *)
    S364_RS_AX_RH_LATCH_후진2 AT %MW87150.2 : BOOL; (* S364_RS_AX_RH_LATCH_후진2 *)
    S364_RS_AX_RH_SLD_CLP_전진 AT %MW87151.0 : BOOL; (* S364_RS_AX_RH_SLD_CLP_전진 *)
    S364_RS_AX_RH_SLD_CLP_후진1 AT %MW87151.1 : BOOL; (* S364_RS_AX_RH_SLD_CLP_후진1 *)
    S364_RS_AX_RH_SLD_CLP_후진2 AT %MW87151.2 : BOOL; (* S364_RS_AX_RH_SLD_CLP_후진2 *)
    S364_RS_AX_RH_SLD_CLP_후진3 AT %MW87151.3 : BOOL; (* S364_RS_AX_RH_SLD_CLP_후진3 *)
    S364_RS_AX_RH_SLD_CLP_후진4 AT %MW87151.4 : BOOL; (* S364_RS_AX_RH_SLD_CLP_후진4 *)
    S364_RS_AX_RH_SLD_LAT_전진 AT %MW87150.8 : BOOL; (* S364_RS_AX_RH_SLD_LAT_전진 *)
    S364_RS_AX_RH_SLD_LAT_후진1 AT %MW87150.9 : BOOL; (* S364_RS_AX_RH_SLD_LAT_후진1 *)
    S364_RS_AX_RH_SLD_LAT_후진2 AT %MW87150.10 : BOOL; (* S364_RS_AX_RH_SLD_LAT_후진2 *)
    S364_RS_AX_RH_SLD_LAT_후진3 AT %MW87150.11 : BOOL; (* S364_RS_AX_RH_SLD_LAT_후진3 *)
    S364_RS_AX_RH_SLD_LAT_후진4 AT %MW87150.12 : BOOL; (* S364_RS_AX_RH_SLD_LAT_후진4 *)
    S364_RS_AX_RH_SLIDE_전진 AT %MW87151.10 : BOOL; (* S364_RS_AX_RH_SLIDE_전진 *)
    S364_RS_AX_RH_SLIDE_후진 AT %MW87151.11 : BOOL; (* S364_RS_AX_RH_SLIDE_후진 *)
    S364_SOL_AX_CLAMP_전진 AT %MW97153.2 : BOOL; (* S364_SOL_AX_CLAMP_전진 *)
    S364_SOL_AX_CLAMP_후진 AT %MW97153.3 : BOOL; (* S364_SOL_AX_CLAMP_후진 *)
    S364_SOL_AX_LATCH_전진 AT %MW97153.0 : BOOL; (* S364_SOL_AX_LATCH_전진 *)
    S364_SOL_AX_LATCH_후진 AT %MW97153.1 : BOOL; (* S364_SOL_AX_LATCH_후진 *)
    S364_SOL_AX_LH_BRAKE_ON AT %MW97154.2 : BOOL; (* S364_SOL_AX_LH_BRAKE_ON *)
    S364_SOL_AX_LH_SLD_CLP_전진 AT %MW97153.6 : BOOL; (* S364_SOL_AX_LH_SLD_CLP_전진 *)
    S364_SOL_AX_LH_SLD_CLP_후진 AT %MW97153.7 : BOOL; (* S364_SOL_AX_LH_SLD_CLP_후진 *)
    S364_SOL_AX_LH_SLD_LAT_전진 AT %MW97153.4 : BOOL; (* S364_SOL_AX_LH_SLD_LAT_전진 *)
    S364_SOL_AX_LH_SLD_LAT_후진 AT %MW97153.5 : BOOL; (* S364_SOL_AX_LH_SLD_LAT_후진 *)
    S364_SOL_AX_LH_SLIDE_전진 AT %MW97154.0 : BOOL; (* S364_SOL_AX_LH_SLIDE_전진 *)
    S364_SOL_AX_LH_SLIDE_후진 AT %MW97154.1 : BOOL; (* S364_SOL_AX_LH_SLIDE_후진 *)
    S364_SOL_AX_RH_BRAKE_ON AT %MW97154.6 : BOOL; (* S364_SOL_AX_RH_BRAKE_ON *)
    S364_SOL_AX_RH_SLD_CLP_전진 AT %MW97153.10 : BOOL; (* S364_SOL_AX_RH_SLD_CLP_전진 *)
    S364_SOL_AX_RH_SLD_CLP_후진 AT %MW97153.11 : BOOL; (* S364_SOL_AX_RH_SLD_CLP_후진 *)
    S364_SOL_AX_RH_SLD_LAT_전진 AT %MW97153.8 : BOOL; (* S364_SOL_AX_RH_SLD_LAT_전진 *)
    S364_SOL_AX_RH_SLD_LAT_후진 AT %MW97153.9 : BOOL; (* S364_SOL_AX_RH_SLD_LAT_후진 *)
    S364_SOL_AX_RH_SLIDE_전진 AT %MW97154.4 : BOOL; (* S364_SOL_AX_RH_SLIDE_전진 *)
    S364_SOL_AX_RH_SLIDE_후진 AT %MW97154.5 : BOOL; (* S364_SOL_AX_RH_SLIDE_후진 *)
    S364_공기압_AIR_CHECK AT %MW87152.14 : BOOL; (* S364_공기압_AIR_CHECK *)
    S365_6_1_PLC_BOX_CP_TRIP AT %MW86012.15 : BOOL; (* S365_6_1_PLC_BOX_CP_TRIP *)
    S365_PHS_ROOF_PNL_썬루프_감지 AT %MW86010.3 : BOOL;
    S365_PRS_ROOF_PNL_제품감지1 AT %MW86010.0 : BOOL;
    S365_PRS_ROOF_PNL_제품감지2 AT %MW86010.1 : BOOL;
    S365_PRS_ROOF_PNL_제품감지3 AT %MW86010.2 : BOOL;
    S366L_PRS_AX_COM_CHECK AT %MW88100.8 : BOOL; (* S366L_PRS_AX_COM_CHECK *)
    S366L_PRS_AX_GR_CHECK AT %MW88100.9 : BOOL; (* S366L_PRS_AX_GR_CHECK *)
    S366L_PRS_AX_RAIL_CHECK AT %MW88100.11 : BOOL; (* S366L_PRS_AX_RAIL_CHECK *)
    S366L_PRS_AX_ROOF_FRT_CHECK AT %MW88100.12 : BOOL; (* S366L_PRS_AX_ROOF_FRT_CHECK *)
    S366L_PRS_AX_ROOF_RR_CHECK AT %MW88100.13 : BOOL; (* S366L_PRS_AX_ROOF_RR_CHECK *)
    S366L_PRS_AX_SR_CHECK AT %MW88100.10 : BOOL; (* S366L_PRS_AX_SR_CHECK *)
    S366L_RS_AX_CLAMP_전진 AT %MW88100.0 : BOOL; (* S366L_RS_AX_CLAMP_전진 *)
    S366L_RS_AX_CLAMP_후진1 AT %MW88100.1 : BOOL; (* S366L_RS_AX_CLAMP_후진1 *)
    S366L_RS_AX_CLAMP_후진2 AT %MW88100.2 : BOOL; (* S366L_RS_AX_CLAMP_후진2 *)
    S366L_RS_AX_CLAMP_후진3 AT %MW88100.3 : BOOL; (* S366L_RS_AX_CLAMP_후진3 *)
    S366L_RS_AX_CLAMP_후진4 AT %MW88100.4 : BOOL; (* S366L_RS_AX_CLAMP_후진4 *)
    S366L_RS_AX_CLAMP_후진5 AT %MW88100.5 : BOOL; (* S366L_RS_AX_CLAMP_후진5 *)
    S366R_8_10_PLC_BOX_CP_TRIP AT %MW88100.15 : BOOL; (* S366L_LS_AX_MAINTENANCE_CHK *)
    S366R_8_20_PLC_BOX_CP_TRIP AT %MW88200.15 : BOOL; (* S366R_LS_AX_MAINTENANCE_CHK *)
    S366R_PRS_AX_COM_CHECK AT %MW88200.8 : BOOL; (* S366R_PRS_AX_COM_CHECK *)
    S366R_PRS_AX_GR_CHECK AT %MW88200.9 : BOOL; (* S366R_PRS_AX_GR_CHECK *)
    S366R_PRS_AX_RAIL_CHECK AT %MW88200.11 : BOOL; (* S366R_PRS_AX_RAIL_CHECK *)
    S366R_PRS_AX_ROOF_FRT_CHECK AT %MW88200.12 : BOOL; (* S366R_PRS_AX_ROOF_FRT_CHECK *)
    S366R_PRS_AX_ROOF_RR_CHECK AT %MW88200.13 : BOOL; (* S366R_PRS_AX_ROOF_RR_CHECK *)
    S366R_PRS_AX_SR_CHECK AT %MW88200.10 : BOOL; (* S366R_PRS_AX_SR_CHECK *)
    S366R_RS_AX_CLAMP_전진 AT %MW88200.0 : BOOL; (* S366R_RS_AX_CLAMP_전진 *)
    S366R_RS_AX_CLAMP_후진1 AT %MW88200.1 : BOOL; (* S366R_RS_AX_CLAMP_후진1 *)
    S366R_RS_AX_CLAMP_후진2 AT %MW88200.2 : BOOL; (* S366R_RS_AX_CLAMP_후진2 *)
    S366R_RS_AX_CLAMP_후진3 AT %MW88200.3 : BOOL; (* S366R_RS_AX_CLAMP_후진3 *)
    S366R_RS_AX_CLAMP_후진4 AT %MW88200.4 : BOOL; (* S366R_RS_AX_CLAMP_후진4 *)
    S366R_RS_AX_CLAMP_후진5 AT %MW88200.5 : BOOL; (* S366R_RS_AX_CLAMP_후진5 *)
    S366_6_10_PLC_BOX_CP_TRIP AT %MW86102.15 : BOOL; (* S366_6_10_PLC_BOX_CP_TRIP *)
    S366_INDEX_LH_TURN_감지1 AT %MW86101.4 : BOOL; (* S366_INDEX_LH_TURN_감지1 *)
    S366_INDEX_LH_TURN_감지2 AT %MW86101.5 : BOOL; (* S366_INDEX_LH_TURN_감지2 *)
    S366_INDEX_LH_TURN_감지3 AT %MW86101.6 : BOOL; (* S366_INDEX_LH_TURN_감지3 *)
    S366_INDEX_LH_TURN_원점 AT %MW86101.7 : BOOL; (* S366_INDEX_LH_TURN_원점 *)
    S366_INDEX_RH_TURN_감지1 AT %MW86101.0 : BOOL; (* S366_INDEX_RH_TURN_감지1 *)
    S366_INDEX_RH_TURN_감지2 AT %MW86101.1 : BOOL; (* S366_INDEX_RH_TURN_감지2 *)
    S366_INDEX_RH_TURN_감지3 AT %MW86101.2 : BOOL; (* S366_INDEX_RH_TURN_감지3 *)
    S366_INDEX_RH_TURN_원점 AT %MW86101.3 : BOOL; (* S366_INDEX_RH_TURN_원점 *)
    S366_LH_CUT_OFF_BOX_ON AT %MW86102.10 : BOOL;
    S366_LS_MAINTENANCE1 AT %MW86102.0 : BOOL;
    S366_LS_MAINTENANCE2 AT %MW86102.1 : BOOL;
    S366_M_AX_LH_CLP_전진_LAMP AT %MW12608 : WORD; (* S366_M_AX_LH_CLP_전진_LAMP *)
    S366_M_AX_LH_CLP_후진_LAMP AT %MW12609 : WORD; (* S366_M_AX_LH_CLP_후진_LAMP *)
    S366_M_AX_RH_CLP_전진_LAMP AT %MW12624 : WORD; (* S366_M_AX_RH_CLP_전진_LAMP *)
    S366_M_AX_RH_CLP_후진_LAMP AT %MW12625 : WORD; (* S366_M_AX_RH_CLP_후진_LAMP *)
    S366_M_TURN_LOCK_전진_LAMP AT %MW12600 : WORD; (* S366_M_TURN_LOCK_전진_LAMP *)
    S366_M_TURN_LOCK_후진_LAMP AT %MW12601 : WORD; (* S366_M_TURN_LOCK_후진_LAMP *)
    S366_M_TURN_전진_LAMP AT %MW12602 : WORD; (* S366_M_TURN_전진_LAMP *)
    S366_M_TURN_후진_LAMP AT %MW12603 : WORD; (* S366_M_TURN_후진_LAMP *)
    S366_RH_CUT_OFF_BOX_ON AT %MW86102.11 : BOOL;
    S366_RS_AX_IDX_LOCK_전진1 AT %MW86100.0 : BOOL; (* S366_RS_AX_IDX_LOCK_전진1 *)
    S366_RS_AX_IDX_LOCK_전진2 AT %MW86100.2 : BOOL; (* S366_RS_AX_IDX_LOCK_전진2 *)
    S366_RS_AX_IDX_LOCK_후진1 AT %MW86100.1 : BOOL; (* S366_RS_AX_IDX_LOCK_후진1 *)
    S366_RS_AX_IDX_LOCK_후진2 AT %MW86100.3 : BOOL; (* S366_RS_AX_IDX_LOCK_후진2 *)
    S366_SOL_AX_LH_CLP_전진 AT %MW98101.0 : BOOL;
    S366_SOL_AX_LH_CLP_후진 AT %MW98101.1 : BOOL;
    S366_SOL_AX_LOCK_G_전진 AT %MW96103.0 : BOOL; (* S366_SOL_AX_LOCK_G_전진 *)
    S366_SOL_AX_LOCK_G_후진 AT %MW96103.1 : BOOL; (* S366_SOL_AX_LOCK_G_후진 *)
    S366_SOL_AX_RH_CLP_전진 AT %MW98201.0 : BOOL;
    S366_SOL_AX_RH_CLP_후진 AT %MW98201.1 : BOOL;
    S366_공기압_AIR_CHECK AT %MW86102.14 : BOOL; (* S366_공기압_AIR_CHECK *)
    S367_6_20_PLC_BOX_CP_TRIP AT %MW86202.15 : BOOL; (* S367_6_20_PLC_BOX_CP_TRIP *)
    S367_6_21_PLC_BOX_CP_TRIP AT %MW86212.15 : BOOL; (* S367_6_21_PLC_BOX_CP_TRIP *)
    S367_M_LH_AX_CLAMP_전진_LAMP AT %MW13104 : WORD; (* S367_M_LH_AX_CLAMP_전진_LAMP *)
    S367_M_LH_AX_CLAMP_후진_LAMP AT %MW13105 : WORD; (* S367_M_LH_AX_CLAMP_후진_LAMP *)
    S367_M_LH_AX_LATCH_전진_LAMP AT %MW13100 : WORD; (* S367_M_LH_AX_LATCH_전진_LAMP *)
    S367_M_LH_AX_LATCH_후진_LAMP AT %MW13101 : WORD; (* S367_M_LH_AX_LATCH_후진_LAMP *)
    S367_M_LH_AX_SR_LAT_전진_LAMP AT %MW13102 : WORD; (* S367_M_LH_AX_SR_LAT_전진_LAMP *)
    S367_M_LH_AX_SR_LAT_후진_LAMP AT %MW13103 : WORD; (* S367_M_LH_AX_SR_LAT_후진_LAMP *)
    S367_M_RH_AX_CLAMP_전진_LAMP AT %MW13120 : WORD; (* S367_M_RH_AX_CLAMP_전진_LAMP *)
    S367_M_RH_AX_CLAMP_후진_LAMP AT %MW13121 : WORD; (* S367_M_RH_AX_CLAMP_후진_LAMP *)
    S367_M_RH_AX_LATCH_전진_LAMP AT %MW13116 : WORD; (* S367_M_RH_AX_LATCH_전진_LAMP *)
    S367_M_RH_AX_LATCH_후진_LAMP AT %MW13117 : WORD; (* S367_M_RH_AX_LATCH_후진_LAMP *)
    S367_M_RH_AX_SR_LAT_전진_LAMP AT %MW13118 : WORD; (* S367_M_RH_AX_SR_LAT_전진_LAMP *)
    S367_M_RH_AX_SR_LAT_후진_LAMP AT %MW13119 : WORD; (* S367_M_RH_AX_SR_LAT_후진_LAMP *)
    S367_PRS_AX_LH_ROOF_FRT_CHK AT %MW86212.0 : BOOL; (* S367_PRS_AX_LH_ROOF_FRT_CHK *)
    S367_PRS_AX_LH_ROOF_RR_CHK AT %MW86212.1 : BOOL; (* S367_PRS_AX_LH_ROOF_RR_CHK *)
    S367_PRS_AX_RH_ROOF_FRT_CHK AT %MW86202.0 : BOOL; (* S367_PRS_AX_RH_ROOF_FRT_CHK *)
    S367_PRS_AX_RH_ROOF_RR_CHK AT %MW86202.1 : BOOL; (* S367_PRS_AX_RH_ROOF_RR_CHK *)
    S367_RS_AX_LH_CLAMP_전진 AT %MW86210.8 : BOOL; (* S367_RS_AX_LH_CLAMP_전진 *)
    S367_RS_AX_LH_CLAMP_후진1 AT %MW86210.9 : BOOL; (* S367_RS_AX_LH_CLAMP_후진1 *)
    S367_RS_AX_LH_CLAMP_후진2 AT %MW86210.10 : BOOL; (* S367_RS_AX_LH_CLAMP_후진2 *)
    S367_RS_AX_LH_CLAMP_후진3 AT %MW86210.11 : BOOL; (* S367_RS_AX_LH_CLAMP_후진3 *)
    S367_RS_AX_LH_CLAMP_후진4 AT %MW86210.12 : BOOL; (* S367_RS_AX_LH_CLAMP_후진4 *)
    S367_RS_AX_LH_CLAMP_후진5 AT %MW86210.13 : BOOL; (* S367_RS_AX_LH_CLAMP_후진5 *)
    S367_RS_AX_LH_GR_LATCH_전진 AT %MW86210.0 : BOOL; (* S367_RS_AX_LH_GR_LATCH_전진 *)
    S367_RS_AX_LH_GR_LATCH_후진1 AT %MW86210.1 : BOOL; (* S367_RS_AX_LH_GR_LATCH_후진1 *)
    S367_RS_AX_LH_GR_LATCH_후진2 AT %MW86210.2 : BOOL; (* S367_RS_AX_LH_GR_LATCH_후진2 *)
    S367_RS_AX_LH_GR_LATCH_후진3 AT %MW86210.3 : BOOL; (* S367_RS_AX_LH_GR_LATCH_후진3 *)
    S367_RS_AX_LH_GR_LATCH_후진4 AT %MW86210.4 : BOOL; (* S367_RS_AX_LH_GR_LATCH_후진4 *)
    S367_RS_AX_LH_GR_LATCH_후진5 AT %MW86210.5 : BOOL; (* S367_RS_AX_LH_GR_LATCH_후진5 *)
    S367_RS_AX_LH_SR_LATCH_전진 AT %MW86211.0 : BOOL; (* S367_RS_AX_LH_SR_LATCH_전진 *)
    S367_RS_AX_LH_SR_LATCH_후진1 AT %MW86211.1 : BOOL; (* S367_RS_AX_LH_SR_LATCH_후진1 *)
    S367_RS_AX_LH_SR_LATCH_후진2 AT %MW86211.2 : BOOL; (* S367_RS_AX_LH_SR_LATCH_후진2 *)
    S367_RS_AX_LH_SR_LATCH_후진3 AT %MW86211.3 : BOOL; (* S367_RS_AX_LH_SR_LATCH_후진3 *)
    S367_RS_AX_RH_CLAMP_전진 AT %MW86200.8 : BOOL; (* S367_RS_AX_RH_CLAMP_전진 *)
    S367_RS_AX_RH_CLAMP_후진1 AT %MW86200.9 : BOOL; (* S367_RS_AX_RH_CLAMP_후진1 *)
    S367_RS_AX_RH_CLAMP_후진2 AT %MW86200.10 : BOOL; (* S367_RS_AX_RH_CLAMP_후진2 *)
    S367_RS_AX_RH_CLAMP_후진3 AT %MW86200.11 : BOOL; (* S367_RS_AX_RH_CLAMP_후진3 *)
    S367_RS_AX_RH_CLAMP_후진4 AT %MW86200.12 : BOOL; (* S367_RS_AX_RH_CLAMP_후진4 *)
    S367_RS_AX_RH_CLAMP_후진5 AT %MW86200.13 : BOOL; (* S367_RS_AX_RH_CLAMP_후진5 *)
    S367_RS_AX_RH_GR_LATCH_전진 AT %MW86200.0 : BOOL; (* S367_RS_AX_RH_GR_LATCH_전진 *)
    S367_RS_AX_RH_GR_LATCH_후진1 AT %MW86200.1 : BOOL; (* S367_RS_AX_RH_GR_LATCH_후진1 *)
    S367_RS_AX_RH_GR_LATCH_후진2 AT %MW86200.2 : BOOL; (* S367_RS_AX_RH_GR_LATCH_후진2 *)
    S367_RS_AX_RH_GR_LATCH_후진3 AT %MW86200.3 : BOOL; (* S367_RS_AX_RH_GR_LATCH_후진3 *)
    S367_RS_AX_RH_GR_LATCH_후진4 AT %MW86200.4 : BOOL; (* S367_RS_AX_RH_GR_LATCH_후진4 *)
    S367_RS_AX_RH_GR_LATCH_후진5 AT %MW86200.5 : BOOL; (* S367_RS_AX_RH_GR_LATCH_후진5 *)
    S367_RS_AX_RH_SR_LATCH_전진 AT %MW86201.0 : BOOL; (* S367_RS_AX_RH_SR_LATCH_전진 *)
    S367_RS_AX_RH_SR_LATCH_후진1 AT %MW86201.1 : BOOL; (* S367_RS_AX_RH_SR_LATCH_후진1 *)
    S367_RS_AX_RH_SR_LATCH_후진2 AT %MW86201.2 : BOOL; (* S367_RS_AX_RH_SR_LATCH_후진2 *)
    S367_RS_AX_RH_SR_LATCH_후진3 AT %MW86201.3 : BOOL; (* S367_RS_AX_RH_SR_LATCH_후진3 *)
    S367_SOL_AX_LH_CLAMP_전진 AT %MW96213.6 : BOOL; (* S367_SOL_AX_LH_CLAMP_전진 *)
    S367_SOL_AX_LH_CLAMP_후진 AT %MW96213.7 : BOOL; (* S367_SOL_AX_LH_CLAMP_후진 *)
    S367_SOL_AX_LH_GR_LATCH_전진 AT %MW96213.2 : BOOL; (* S367_SOL_AX_LH_GR_LATCH_전진 *)
    S367_SOL_AX_LH_GR_LATCH_후진 AT %MW96213.3 : BOOL; (* S367_SOL_AX_LH_GR_LATCH_후진 *)
    S367_SOL_AX_LH_SR_LATCH_전진 AT %MW96213.10 : BOOL; (* S367_SOL_AX_LH_SR_LATCH_전진 *)
    S367_SOL_AX_LH_SR_LATCH_후진 AT %MW96213.11 : BOOL; (* S367_SOL_AX_LH_SR_LATCH_후진 *)
    S367_SOL_AX_RH_CLAMP_전진 AT %MW96213.4 : BOOL; (* S367_SOL_AX_RH_CLAMP_전진 *)
    S367_SOL_AX_RH_CLAMP_후진 AT %MW96213.5 : BOOL; (* S367_SOL_AX_RH_CLAMP_후진 *)
    S367_SOL_AX_RH_GR_LATCH_전진 AT %MW96213.0 : BOOL; (* S367_SOL_AX_RH_GR_LATCH_전진 *)
    S367_SOL_AX_RH_GR_LATCH_후진 AT %MW96213.1 : BOOL; (* S367_SOL_AX_RH_GR_LATCH_후진 *)
    S367_SOL_AX_RH_SR_LATCH_전진 AT %MW96213.8 : BOOL; (* S367_SOL_AX_RH_SR_LATCH_전진 *)
    S367_SOL_AX_RH_SR_LATCH_후진 AT %MW96213.9 : BOOL; (* S367_SOL_AX_RH_SR_LATCH_후진 *)
    S367_공기압_AIR_CHECK AT %MW86202.14 : BOOL; (* S367_공기압_AIR_CHECK *)
    S368L_RS_HANGER_급기_전진단 AT %MW86311.13 : BOOL;
    S368L_RS_HANGER_급기_후진단 AT %MW86311.14 : BOOL;
    S368L_RS_HANGER_급전_전진단 AT %MW86311.11 : BOOL;
    S368L_RS_HANGER_급전_후진단 AT %MW86311.12 : BOOL;
    S368L_SOL_HANGER_급전급기_전진 AT %MW96313.8 : BOOL;
    S368L_SOL_HANGER_급전급기_후진 AT %MW96313.9 : BOOL;
    S368_6_30_PLC_BOX_CP_TRIP AT %MW86302.15 : BOOL; (* S368_6_30_PLC_BOX_CP_TRIP *)
    S368_6_31_PLC_BOX_CP_TRIP AT %MW86312.15 : BOOL; (* S368_6_31_PLC_BOX_CP_TRIP *)
    S368_M_HANGER_CLP_전진_LAMP AT %MW13622 : WORD; (* S368_M_HANGER_CLP_전진_LAMP *)
    S368_M_HANGER_CLP_후진_LAMP AT %MW13623 : WORD; (* S368_M_HANGER_CLP_후진_LAMP *)
    S368_M_HANGER_급전급기_ADV_LAMP AT %MW13606 : WORD; (* S368_M_LH_HANG_CLP_전진_LAMP *)
    S368_M_HANGER_급전급기_RET_LAMP AT %MW13607 : WORD; (* S368_M_LH_HANG_CLP_후진_LAMP *)
    S368_M_LH_AX_CLAMP_전진_LAMP AT %MW13604 : WORD; (* S368_M_LH_AX_CLAMP_전진_LAMP *)
    S368_M_LH_AX_CLAMP_후진_LAMP AT %MW13605 : WORD; (* S368_M_LH_AX_CLAMP_후진_LAMP *)
    S368_M_LH_AX_LATCH_전진_LAMP AT %MW13600 : WORD; (* S368_M_LH_AX_LATCH_전진_LAMP *)
    S368_M_LH_AX_LATCH_후진_LAMP AT %MW13601 : WORD; (* S368_M_LH_AX_LATCH_후진_LAMP *)
    S368_M_LH_AX_SR_LAT_전진_LAMP AT %MW13602 : WORD; (* S368_M_LH_AX_SR_LAT_전진_LAMP *)
    S368_M_LH_AX_SR_LAT_후진_LAMP AT %MW13603 : WORD; (* S368_M_LH_AX_SR_LAT_후진_LAMP *)
    S368_M_RH_AX_CLAMP_전진_LAMP AT %MW13620 : WORD; (* S368_M_RH_AX_CLAMP_전진_LAMP *)
    S368_M_RH_AX_CLAMP_후진_LAMP AT %MW13621 : WORD; (* S368_M_RH_AX_CLAMP_후진_LAMP *)
    S368_M_RH_AX_LATCH_전진_LAMP AT %MW13616 : WORD; (* S368_M_RH_AX_LATCH_전진_LAMP *)
    S368_M_RH_AX_LATCH_후진_LAMP AT %MW13617 : WORD; (* S368_M_RH_AX_LATCH_후진_LAMP *)
    S368_M_RH_AX_SR_LAT_전진_LAMP AT %MW13618 : WORD; (* S368_M_RH_AX_SR_LAT_전진_LAMP *)
    S368_M_RH_AX_SR_LAT_후진_LAMP AT %MW13619 : WORD; (* S368_M_RH_AX_SR_LAT_후진_LAMP *)
    S368_PRS_AX_LH_HANGER_CHECK AT %MW86312.2 : BOOL; (* S368_PRS_AX_LH_HANGER_CHECK *)
    S368_PRS_AX_LH_ROOF_FRT_CHECK AT %MW86312.0 : BOOL; (* S368_PRS_AX_LH_ROOF_FRT_CHECK *)
    S368_PRS_AX_LH_ROOF_RR_CHECK AT %MW86312.1 : BOOL; (* S368_PRS_AX_LH_ROOF_RR_CHECK *)
    S368_PRS_AX_RH_HANGER_CHECK AT %MW86302.2 : BOOL; (* S368_PRS_AX_RH_HANGER_CHECK *)
    S368_PRS_AX_RH_ROOF_FRT_CHECK AT %MW86302.0 : BOOL; (* S368_PRS_AX_RH_ROOF_FRT_CHECK *)
    S368_PRS_AX_RH_ROOF_RR_CHECK AT %MW86302.1 : BOOL; (* S368_PRS_AX_RH_ROOF_RR_CHECK *)
    S368_RS_AX_HANGER_CLP_전진 AT %MW86301.8 : BOOL; (* S368_RS_AX_HANGER_CLP_전진 *)
    S368_RS_AX_HANGER_CLP_후진1 AT %MW86301.9 : BOOL; (* S368_RS_AX_HANGER_CLP_후진1 *)
    S368_RS_AX_HANGER_CLP_후진2 AT %MW86301.10 : BOOL; (* S368_RS_AX_HANGER_CLP_후진2 *)
    S368_RS_AX_LH_CLAMP_전진 AT %MW86310.8 : BOOL; (* S368_RS_AX_LH_CLAMP_전진 *)
    S368_RS_AX_LH_CLAMP_후진1 AT %MW86310.9 : BOOL; (* S368_RS_AX_LH_CLAMP_후진1 *)
    S368_RS_AX_LH_CLAMP_후진2 AT %MW86310.10 : BOOL; (* S368_RS_AX_LH_CLAMP_후진2 *)
    S368_RS_AX_LH_CLAMP_후진3 AT %MW86310.11 : BOOL; (* S368_RS_AX_LH_CLAMP_후진3 *)
    S368_RS_AX_LH_CLAMP_후진4 AT %MW86310.12 : BOOL; (* S368_RS_AX_LH_CLAMP_후진4 *)
    S368_RS_AX_LH_CLAMP_후진5 AT %MW86310.13 : BOOL; (* S368_RS_AX_LH_CLAMP_후진5 *)
    S368_RS_AX_LH_GR_LATCH_전진 AT %MW86310.0 : BOOL; (* S368_RS_AX_LH_GR_LATCH_전진 *)
    S368_RS_AX_LH_GR_LATCH_후진1 AT %MW86310.1 : BOOL; (* S368_RS_AX_LH_GR_LATCH_후진1 *)
    S368_RS_AX_LH_GR_LATCH_후진2 AT %MW86310.2 : BOOL; (* S368_RS_AX_LH_GR_LATCH_후진2 *)
    S368_RS_AX_LH_GR_LATCH_후진3 AT %MW86310.3 : BOOL; (* S368_RS_AX_LH_GR_LATCH_후진3 *)
    S368_RS_AX_LH_GR_LATCH_후진4 AT %MW86310.4 : BOOL; (* S368_RS_AX_LH_GR_LATCH_후진4 *)
    S368_RS_AX_LH_GR_LATCH_후진5 AT %MW86310.5 : BOOL; (* S368_RS_AX_LH_GR_LATCH_후진5 *)
    S368_RS_AX_LH_HANG_CLP_후진1 AT %MW86311.8 : BOOL; (* S368_RS_AX_LH_HANG_CLP_후진1 *)
    S368_RS_AX_LH_HANG_CLP_후진2 AT %MW86311.9 : BOOL; (* S368_RS_AX_LH_HANG_CLP_후진2 *)
    S368_RS_AX_LH_SR_LATCH_전진 AT %MW86311.0 : BOOL; (* S368_RS_AX_LH_SR_LATCH_전진 *)
    S368_RS_AX_LH_SR_LATCH_후진1 AT %MW86311.1 : BOOL; (* S368_RS_AX_LH_SR_LATCH_후진1 *)
    S368_RS_AX_LH_SR_LATCH_후진2 AT %MW86311.2 : BOOL; (* S368_RS_AX_LH_SR_LATCH_후진2 *)
    S368_RS_AX_LH_SR_LATCH_후진3 AT %MW86311.3 : BOOL; (* S368_RS_AX_LH_SR_LATCH_후진3 *)
    S368_RS_AX_LH_SR_LATCH_후진4 AT %MW86311.4 : BOOL; (* S368_RS_AX_LH_SR_LATCH_후진4 *)
    S368_RS_AX_RH_CLAMP_전진 AT %MW86300.8 : BOOL; (* S368_RS_AX_RH_CLAMP_전진 *)
    S368_RS_AX_RH_CLAMP_후진1 AT %MW86300.9 : BOOL; (* S368_RS_AX_RH_CLAMP_후진1 *)
    S368_RS_AX_RH_CLAMP_후진2 AT %MW86300.10 : BOOL; (* S368_RS_AX_RH_CLAMP_후진2 *)
    S368_RS_AX_RH_CLAMP_후진3 AT %MW86300.11 : BOOL; (* S368_RS_AX_RH_CLAMP_후진3 *)
    S368_RS_AX_RH_CLAMP_후진4 AT %MW86300.12 : BOOL; (* S368_RS_AX_RH_CLAMP_후진4 *)
    S368_RS_AX_RH_CLAMP_후진5 AT %MW86300.13 : BOOL; (* S368_RS_AX_RH_CLAMP_후진5 *)
    S368_RS_AX_RH_GR_LATCH_전진 AT %MW86300.0 : BOOL; (* S368_RS_AX_RH_GR_LATCH_전진 *)
    S368_RS_AX_RH_GR_LATCH_후진1 AT %MW86300.1 : BOOL; (* S368_RS_AX_RH_GR_LATCH_후진1 *)
    S368_RS_AX_RH_GR_LATCH_후진2 AT %MW86300.2 : BOOL; (* S368_RS_AX_RH_GR_LATCH_후진2 *)
    S368_RS_AX_RH_GR_LATCH_후진3 AT %MW86300.3 : BOOL; (* S368_RS_AX_RH_GR_LATCH_후진3 *)
    S368_RS_AX_RH_GR_LATCH_후진4 AT %MW86300.4 : BOOL; (* S368_RS_AX_RH_GR_LATCH_후진4 *)
    S368_RS_AX_RH_GR_LATCH_후진5 AT %MW86300.5 : BOOL; (* S368_RS_AX_RH_GR_LATCH_후진5 *)
    S368_RS_AX_RH_SR_LATCH_전진 AT %MW86301.0 : BOOL; (* S368_RS_AX_RH_SR_LATCH_전진 *)
    S368_RS_AX_RH_SR_LATCH_후진1 AT %MW86301.1 : BOOL; (* S368_RS_AX_RH_SR_LATCH_후진1 *)
    S368_RS_AX_RH_SR_LATCH_후진2 AT %MW86301.2 : BOOL; (* S368_RS_AX_RH_SR_LATCH_후진2 *)
    S368_RS_AX_RH_SR_LATCH_후진3 AT %MW86301.3 : BOOL; (* S368_RS_AX_RH_SR_LATCH_후진3 *)
    S368_RS_AX_RH_SR_LATCH_후진4 AT %MW86301.4 : BOOL; (* S368_RS_AX_RH_SR_LATCH_후진4 *)
    S368_SOL_AX_HANG_CLP_전진 AT %MW96303.12 : BOOL; (* S368_SOL_AX_HANG_CLP_전진 *)
    S368_SOL_AX_HANG_CLP_후진 AT %MW96303.13 : BOOL; (* S368_SOL_AX_HANG_CLP_후진 *)
    S368_SOL_AX_LH_CLAMP_전진 AT %MW96303.6 : BOOL; (* S368_SOL_AX_LH_CLAMP_전진 *)
    S368_SOL_AX_LH_CLAMP_후진 AT %MW96303.7 : BOOL; (* S368_SOL_AX_LH_CLAMP_후진 *)
    S368_SOL_AX_LH_GR_LATCH_전진 AT %MW96303.2 : BOOL; (* S368_SOL_AX_LH_GR_LATCH_전진 *)
    S368_SOL_AX_LH_GR_LATCH_후진 AT %MW96303.3 : BOOL; (* S368_SOL_AX_LH_GR_LATCH_후진 *)
    S368_SOL_AX_LH_SR_LATCH_전진 AT %MW96303.10 : BOOL; (* S368_SOL_AX_LH_SR_LATCH_전진 *)
    S368_SOL_AX_LH_SR_LATCH_후진 AT %MW96303.11 : BOOL; (* S368_SOL_AX_LH_SR_LATCH_후진 *)
    S368_SOL_AX_RH_CLAMP_전진 AT %MW96303.4 : BOOL; (* S368_SOL_AX_RH_CLAMP_전진 *)
    S368_SOL_AX_RH_CLAMP_후진 AT %MW96303.5 : BOOL; (* S368_SOL_AX_RH_CLAMP_후진 *)
    S368_SOL_AX_RH_GR_LATCH_전진 AT %MW96303.0 : BOOL; (* S368_SOL_AX_RH_GR_LATCH_전진 *)
    S368_SOL_AX_RH_GR_LATCH_후진 AT %MW96303.1 : BOOL; (* S368_SOL_AX_RH_GR_LATCH_후진 *)
    S368_SOL_AX_RH_SR_LATCH_전진 AT %MW96303.8 : BOOL; (* S368_SOL_AX_RH_SR_LATCH_전진 *)
    S368_SOL_AX_RH_SR_LATCH_후진 AT %MW96303.9 : BOOL; (* S368_SOL_AX_RH_SR_LATCH_후진 *)
    S368_공기압_AIR_CHECK AT %MW86302.14 : BOOL; (* S368_공기압_AIR_CHECK *)
    S369LD_6_41_PLC_BOX_CP_TRIP AT %MW86412.15 : BOOL; (* S369LD_6_41_PLC_BOX_CP_TRIP *)
    S369LD_RS_AX_LH_LATCH_전진 AT %MW86411.0 : BOOL; (* S369LD_RS_AX_LH_LATCH_전진 *)
    S369LD_RS_AX_LH_LATCH_후진1 AT %MW86411.1 : BOOL; (* S369LD_RS_AX_LH_LATCH_후진1 *)
    S369LD_RS_AX_LH_LATCH_후진2 AT %MW86411.2 : BOOL; (* S369LD_RS_AX_LH_LATCH_후진2 *)
    S369LD_RS_AX_LH_LATCH_후진3 AT %MW86411.3 : BOOL; (* S369LD_RS_AX_LH_LATCH_후진3 *)
    S369LD_RS_AX_LH_LATCH_후진4 AT %MW86411.4 : BOOL; (* S369LD_RS_AX_LH_LATCH_후진4 *)
    S369LD_RS_AX_RH_LATCH_전진 AT %MW86410.8 : BOOL; (* S369LD_RS_AX_RH_LATCH_전진 *)
    S369LD_RS_AX_RH_LATCH_후진1 AT %MW86410.9 : BOOL; (* S369LD_RS_AX_RH_LATCH_후진1 *)
    S369LD_RS_AX_RH_LATCH_후진2 AT %MW86410.10 : BOOL; (* S369LD_RS_AX_RH_LATCH_후진2 *)
    S369LD_RS_AX_RH_LATCH_후진3 AT %MW86410.11 : BOOL; (* S369LD_RS_AX_RH_LATCH_후진3 *)
    S369LD_RS_AX_RH_LATCH_후진4 AT %MW86410.12 : BOOL; (* S369LD_RS_AX_RH_LATCH_후진4 *)
    S369LD_RS_EJECT_상승1 AT %MW86410.0 : BOOL; (* S369LD_RS_EJECT_상승1 *)
    S369LD_RS_EJECT_상승2 AT %MW86410.2 : BOOL; (* S369LD_RS_EJECT_상승2 *)
    S369LD_RS_EJECT_하강1 AT %MW86410.1 : BOOL; (* S369LD_RS_EJECT_하강1 *)
    S369LD_RS_EJECT_하강2 AT %MW86410.3 : BOOL; (* S369LD_RS_EJECT_하강2 *)
    S369LD_SOL_AX_LH_LATCH_전진 AT %MW96413.4 : BOOL; (* S369LD_SOL_AX_LH_LATCH_전진 *)
    S369LD_SOL_AX_LH_LATCH_후진 AT %MW96413.5 : BOOL; (* S369LD_SOL_AX_LH_LATCH_후진 *)
    S369LD_SOL_AX_RH_LATCH_전진 AT %MW96413.2 : BOOL; (* S369LD_SOL_AX_RH_LATCH_전진 *)
    S369LD_SOL_AX_RH_LATCH_후진 AT %MW96413.3 : BOOL; (* S369LD_SOL_AX_RH_LATCH_후진 *)
    S369LD_SOL_EJECT_상승 AT %MW96413.0 : BOOL; (* S369LD_SOL_EJECT_상승 *)
    S369LD_SOL_EJECT_하강 AT %MW96413.1 : BOOL; (* S369LD_SOL_EJECT_하강 *)
    S369LD_공기압_AIR_CHECK AT %MW86412.14 : BOOL; (* S369LD_공기압_AIR_CHECK *)
    S369UD_6_42_PLC_BOX_CP_TRIP AT %MW86422.15 : BOOL; (* S369UD_6_42_PLC_BOX_CP_TRIP *)
    S369UD_RS_AX_DOCK_CLP_전진 AT %MW86421.8 : BOOL; (* S369UD_RS_AX_DOCK_CLP_전진 *)
    S369UD_RS_AX_DOCK_CLP_후진1 AT %MW86421.9 : BOOL; (* S369UD_RS_AX_DOCK_CLP_후진1 *)
    S369UD_RS_AX_DOCK_CLP_후진2 AT %MW86421.10 : BOOL; (* S369UD_RS_AX_DOCK_CLP_후진2 *)
    S369UD_RS_AX_DOCK_CLP_후진3 AT %MW86421.11 : BOOL; (* S369UD_RS_AX_DOCK_CLP_후진3 *)
    S369UD_RS_AX_DOCK_CLP_후진4 AT %MW86421.12 : BOOL; (* S369UD_RS_AX_DOCK_CLP_후진4 *)
    S369UD_RS_AX_LH_LATCH_전진 AT %MW86421.0 : BOOL; (* S369UD_RS_AX_LH_LATCH_전진 *)
    S369UD_RS_AX_LH_LATCH_후진1 AT %MW86421.1 : BOOL; (* S369UD_RS_AX_LH_LATCH_후진1 *)
    S369UD_RS_AX_LH_LATCH_후진2 AT %MW86421.2 : BOOL; (* S369UD_RS_AX_LH_LATCH_후진2 *)
    S369UD_RS_AX_LH_LATCH_후진3 AT %MW86421.3 : BOOL; (* S369UD_RS_AX_LH_LATCH_후진3 *)
    S369UD_RS_AX_LH_LATCH_후진4 AT %MW86421.4 : BOOL; (* S369UD_RS_AX_LH_LATCH_후진4 *)
    S369UD_RS_AX_RH_LATCH_전진 AT %MW86420.8 : BOOL; (* S369UD_RS_AX_RH_LATCH_전진 *)
    S369UD_RS_AX_RH_LATCH_후진1 AT %MW86420.9 : BOOL; (* S369UD_RS_AX_RH_LATCH_후진1 *)
    S369UD_RS_AX_RH_LATCH_후진2 AT %MW86420.10 : BOOL; (* S369UD_RS_AX_RH_LATCH_후진2 *)
    S369UD_RS_AX_RH_LATCH_후진3 AT %MW86420.11 : BOOL; (* S369UD_RS_AX_RH_LATCH_후진3 *)
    S369UD_RS_AX_RH_LATCH_후진4 AT %MW86420.12 : BOOL; (* S369UD_RS_AX_RH_LATCH_후진4 *)
    S369UD_RS_EJECT_상승1 AT %MW86420.0 : BOOL; (* S369UD_RS_EJECT_상승1 *)
    S369UD_RS_EJECT_상승2 AT %MW86420.2 : BOOL; (* S369UD_RS_EJECT_상승2 *)
    S369UD_RS_EJECT_하강1 AT %MW86420.1 : BOOL; (* S369UD_RS_EJECT_하강1 *)
    S369UD_RS_EJECT_하강2 AT %MW86420.3 : BOOL; (* S369UD_RS_EJECT_하강2 *)
    S369UD_SOL_AX_DOCK_CLP_전진 AT %MW96423.6 : BOOL; (* S369UD_SOL_AX_DOCK_CLP_전진 *)
    S369UD_SOL_AX_DOCK_CLP_후진 AT %MW96423.7 : BOOL; (* S369UD_SOL_AX_DOCK_CLP_후진 *)
    S369UD_SOL_AX_LH_LATCH_전진 AT %MW96423.4 : BOOL; (* S369UD_SOL_AX_LH_LATCH_전진 *)
    S369UD_SOL_AX_LH_LATCH_후진 AT %MW96423.5 : BOOL; (* S369UD_SOL_AX_LH_LATCH_후진 *)
    S369UD_SOL_AX_RH_LATCH_전진 AT %MW96423.2 : BOOL; (* S369UD_SOL_AX_RH_LATCH_전진 *)
    S369UD_SOL_AX_RH_LATCH_후진 AT %MW96423.3 : BOOL; (* S369UD_SOL_AX_RH_LATCH_후진 *)
    S369UD_SOL_EJECT_상승 AT %MW96423.0 : BOOL; (* S369UD_SOL_EJECT_상승 *)
    S369UD_SOL_EJECT_하강 AT %MW96423.1 : BOOL; (* S369UD_SOL_EJECT_하강 *)
    S369UD_공기압_AIR_CHECK AT %MW86422.14 : BOOL; (* S369UD_공기압_AIR_CHECK *)
    S369_1_6_40_PLC_BOX_CP_TRIP AT %MW86402.15 : BOOL; (* S369_1_6_40_PLC_BOX_CP_TRIP *)
    S369_1_PHS_ROOF_PNL_썬루프_감지 AT %MW86400.3 : BOOL;
    S369_1_PRS_ROOF_PNL_제품감지1 AT %MW86400.0 : BOOL;
    S369_1_PRS_ROOF_PNL_제품감지2 AT %MW86400.1 : BOOL;
    S369_1_PRS_ROOF_PNL_제품감지3 AT %MW86400.2 : BOOL;
    S369_CONVEY_I_JERK_LIMIT AT %MD25004 : DINT;
    S369_CONVEY_I_SOFT리미트_비활성 AT %MW50000.12 : BOOL;
    S369_CONVEY_I_STO_비활성 AT %MW50000.1 : BOOL;
    S369_CONVEY_I_X20_터미널블럭 AT %MW50004 : WORD;
    S369_CONVEY_I_대기모드 AT %MW50000.14 : BOOL;
    S369_CONVEY_I_동작모드 AT %MW50002 : UINT;
    S369_CONVEY_I_모터기동중 AT %MW50000.4 : BOOL;
    S369_CONVEY_I_브레이크_풀림 AT %MW50000.3 : BOOL;
    S369_CONVEY_I_새위치_적용완료 AT %MW50000.6 : BOOL;
    S369_CONVEY_I_서보_운전준비 AT %MW50000.0 : BOOL;
    S369_CONVEY_I_서보동작모드 AT %MW50005 : UINT;
    S369_CONVEY_I_서보드라이브_경고 AT %MW50000.9 : BOOL;
    S369_CONVEY_I_서보드라이브_이상 AT %MW50000.8 : BOOL;
    S369_CONVEY_I_서보출력ON AT %MW50000.2 : BOOL;
    S369_CONVEY_I_설정속도완료 AT %MW50000.11 : BOOL;
    S369_CONVEY_I_실제속도 AT %MW50001 : UINT;
    S369_CONVEY_I_실제토크 AT %MW50003 : UINT;
    S369_CONVEY_I_위치_도착완료 AT %MW50000.7 : BOOL;
    S369_CONVEY_I_주행트레인_활성 AT %MW50000.10 : BOOL;
    S369_CONVEY_I_현재위치값 AT %MD25003 : DINT;
    S369_CONVEY_I_활성드라이브_참조 AT %MW50000.5 : BOOL;
    S369_CONVEY_O_JERK_LIMIT AT %MD25014 : DINT;
    S369_CONVEY_O_JOG_모드비활성 AT %MW50020.5 : BOOL;
    S369_CONVEY_O_JOG_모드활성 AT %MW50020.4 : BOOL;
    S369_CONVEY_O_SOFT_리미트_비활성 AT %MW50020.12 : BOOL;
    S369_CONVEY_O_가속설정 AT %MW50022 : UINT;
    S369_CONVEY_O_감속설정 AT %MW50023 : UINT;
    S369_CONVEY_O_구동모드설정 AT %MW50025 : UINT;
    S369_CONVEY_O_기동정지 AT %MW50020.1 : BOOL;
    S369_CONVEY_O_대기상태 AT %MW50020.14 : BOOL;
    S369_CONVEY_O_모터기동 AT %MW50020.7 : BOOL;
    S369_CONVEY_O_브레이크_풀림 AT %MW50020.3 : BOOL;
    S369_CONVEY_O_비상정지 AT %MW50020.0 : BOOL;
    S369_CONVEY_O_상대위치_적용 AT %MW50020.6 : BOOL;
    S369_CONVEY_O_이동속도_설정 AT %MW50021 : UINT;
    S369_CONVEY_O_이동위치_설정 AT %MD25013 : DINT;
    S369_CONVEY_O_이상리셋 AT %MW50020.8 : BOOL;
    S369_CONVEY_O_출력금지 AT %MW50020.13 : BOOL;
    S369_M_LD_EJECT_상승_LAMP AT %MW14100 : WORD; (* S369_M_LD_EJECT_상승_LAMP *)
    S369_M_LD_EJECT_하강_LAMP AT %MW14101 : WORD; (* S369_M_LD_EJECT_하강_LAMP *)
    S369_M_LD_LH_LAT_전진_LAMP AT %MW14102 : WORD; (* S369_M_LD_LH_LAT_전진_LAMP *)
    S369_M_LD_LH_LAT_후진_LAMP AT %MW14103 : WORD; (* S369_M_LD_LH_LAT_후진_LAMP *)
    S369_M_LD_RH_LAT_전진_LAMP AT %MW14104 : WORD; (* S369_M_LD_RH_LAT_전진_LAMP *)
    S369_M_LD_RH_LAT_후진_LAMP AT %MW14105 : WORD; (* S369_M_LD_RH_LAT_후진_LAMP *)
    S369_M_UD_DOCK_CLP_전진_LAMP AT %MW14122 : WORD; (* S369_M_UD_DOCK_CLP_전진_LAMP *)
    S369_M_UD_DOCK_CLP_후진_LAMP AT %MW14123 : WORD; (* S369_M_UD_DOCK_CLP_후진_LAMP *)
    S369_M_UD_EJECT_상승_LAMP AT %MW14116 : WORD; (* S369_M_UD_EJECT_상승_LAMP *)
    S369_M_UD_EJECT_하강_LAMP AT %MW14117 : WORD; (* S369_M_UD_EJECT_하강_LAMP *)
    S369_M_UD_LH_LAT_전진_LAMP AT %MW14118 : WORD; (* S369_M_UD_LH_LAT_전진_LAMP *)
    S369_M_UD_LH_LAT_후진_LAMP AT %MW14119 : WORD; (* S369_M_UD_LH_LAT_후진_LAMP *)
    S369_M_UD_RH_LAT_전진_LAMP AT %MW14120 : WORD; (* S369_M_UD_RH_LAT_전진_LAMP *)
    S369_M_UD_RH_LAT_후진_LAMP AT %MW14121 : WORD; (* S369_M_UD_RH_LAT_후진_LAMP *)
    S369_PHS_언로딩_이젝터_제품감지1 AT %MW86422.8 : BOOL; (* S369UD_PHS_AX_UD_제품감지_CHK1 *)
    S369_PHS_언로딩_이젝터_제품감지2 AT %MW86422.9 : BOOL; (* S369UD_PHS_AX_UD_제품감지_CHK2 *)
    S369_PRS_로딩_이젝터_LH_제품감지 AT %MW86412.1 : BOOL; (* S369LD_PRS_AX_LD_EJT_LH_CHK *)
    S369_PRS_로딩_이젝터_RH_제품감지 AT %MW86412.0 : BOOL; (* S369LD_PRS_AX_LD_EJT_RH_CHK *)
    S369_SERVO_MC_ON AT %MW85022.0 : BOOL; (* SERVO_BRAKE_ON *)
    S369_SERVO_NFB_ON AT %MW85023.0 : BOOL;
    S369_로딩버퍼_제품감지1 AT %MW86412.5 : BOOL; (* S369LD_LS_AX_CON_BELT_CHK1 *)
    S369_언로딩버퍼_제품감지1 AT %MW86422.5 : BOOL; (* S369UD_LS_AX_CON_BELT_CHK1 *)
    S369_이송버퍼01_제품감지1 AT %MW86422.6 : BOOL; (* S369UD_LS_AX_CON_BELT_CHK2 *)
    S369_이송버퍼02_제품감지1 AT %MW86422.7 : BOOL; (* S369UD_LS_AX_CON_BELT_CHK3 *)
    S369_이송버퍼03_제품감지1 AT %MW86412.7 : BOOL; (* S369LD_LS_AX_CON_BELT_CHK3 *)
    S369_이송버퍼04_제품감지1 AT %MW86412.6 : BOOL; (* S369LD_LS_AX_CON_BELT_CHK2 *)
    SERVO_PNL_SPD_NOMAL AT %MW85023.14 : BOOL; (* SERVO_PNL_SPD_NOMAL *)
    SERVO_PS1_1_DC_OK AT %MW85023.12 : BOOL; (* SERVO_PS1_1_DC_OK *)
    SERVO_PS1_2_DC_OK AT %MW85023.13 : BOOL; (* SERVO_PS1_2_DC_OK *)
    SERVO_PS_CP_TRIP AT %MW85023.15 : BOOL; (* SERVO_PS_CP_TRIP *)
    SERVO_SAFETY_CR_ON AT %MW95024.0 : BOOL; (* SERVO_BRAKE_CR_ON *)
    SEW_INTPUT AT %MW50000 : ARRAY[0..15] OF WORD;
    SEW_OUTPUT AT %MW50020 : ARRAY[0..15] OF WORD;
    _0004_EB01_CFG_ER AT %MW184022.0 : BOOL; (* EB 구성 에러 *)
    _0004_EB01_DEER AT %MW184022.1 : BOOL; (* EB 운전 중 탈락 *)
    _0004_EB02_CFG_ER AT %MW184024.8 : BOOL; (* EB 구성 에러 *)
    _0004_EB02_DEER AT %MW184024.9 : BOOL; (* EB 운전 중 탈락 *)
    _0004_EB03_CFG_ER AT %MW184027.0 : BOOL; (* EB 구성 에러 *)
    _0004_EB03_DEER AT %MW184027.1 : BOOL; (* EB 운전 중 탈락 *)
    _0004_EB04_CFG_ER AT %MW184029.8 : BOOL; (* EB 구성 에러 *)
    _0004_EB04_DEER AT %MW184029.9 : BOOL; (* EB 운전 중 탈락 *)
    _0004_EB05_CFG_ER AT %MW184032.0 : BOOL; (* EB 구성 에러 *)
    _0004_EB05_DEER AT %MW184032.1 : BOOL; (* EB 운전 중 탈락 *)
    _0004_EB06_CFG_ER AT %MW184034.8 : BOOL; (* EB 구성 에러 *)
    _0004_EB06_DEER AT %MW184034.9 : BOOL; (* EB 운전 중 탈락 *)
    _0004_EB07_CFG_ER AT %MW184037.0 : BOOL; (* EB 구성 에러 *)
    _0004_EB07_DEER AT %MW184037.1 : BOOL; (* EB 운전 중 탈락 *)
    _0004_EB08_CFG_ER AT %MW184039.8 : BOOL; (* EB 구성 에러 *)
    _0004_EB08_DEER AT %MW184039.9 : BOOL; (* EB 운전 중 탈락 *)
    _0004_EB09_CFG_ER AT %MW184042.0 : BOOL; (* EB 구성 에러 *)
    _0004_EB09_DEER AT %MW184042.1 : BOOL; (* EB 운전 중 탈락 *)
    _0005_EB01_CFG_ER AT %MW185022.0 : BOOL; (* EB 구성 에러 *)
    _0005_EB01_DEER AT %MW185022.1 : BOOL; (* EB 운전 중 탈락 *)
    _0005_EB01_IO_DEER AT %MW185023.2 : BOOL; (* EB IO 탈락 에러 *)
    _0005_EB01_IO_TYER AT %MW185023.1 : BOOL; (* EB IO 타입 에러 *)
    _0005_EB02_CFG_ER AT %MW185028.0 : BOOL; (* EB 구성 에러 *)
    _0005_EB02_DEER AT %MW185028.1 : BOOL; (* EB 운전 중 탈락 *)
    _0005_EB02_IO_DEER AT %MW185029.2 : BOOL; (* EB IO 탈락 에러 *)
    _0005_EB02_IO_TYER AT %MW185029.1 : BOOL; (* EB IO 타입 에러 *)
    _0005_EB63_S00_SVC_ER AT %MW185036.7 : BOOL; (* 통신 서비스 에러 *)
    _0006_EB01_CFG_ER AT %MW186022.0 : BOOL; (* EB 구성 에러 *)
    _0006_EB01_DEER AT %MW186022.1 : BOOL; (* EB 운전 중 탈락 *)
    _0006_EB01_IO_DEER AT %MW186023.2 : BOOL; (* EB IO 탈락 에러 *)
    _0006_EB01_IO_TYER AT %MW186023.1 : BOOL; (* EB IO 타입 에러 *)
    _0006_EB10_CFG_ER AT %MW186028.0 : BOOL; (* EB 구성 에러 *)
    _0006_EB10_DEER AT %MW186028.1 : BOOL; (* EB 운전 중 탈락 *)
    _0006_EB10_IO_DEER AT %MW186029.2 : BOOL; (* EB IO 탈락 에러 *)
    _0006_EB10_IO_TYER AT %MW186029.1 : BOOL; (* EB IO 타입 에러 *)
    _0006_EB20_CFG_ER AT %MW186034.0 : BOOL; (* EB 구성 에러 *)
    _0006_EB20_DEER AT %MW186034.1 : BOOL; (* EB 운전 중 탈락 *)
    _0006_EB20_IO_DEER AT %MW186035.2 : BOOL; (* EB IO 탈락 에러 *)
    _0006_EB20_IO_TYER AT %MW186035.1 : BOOL; (* EB IO 타입 에러 *)
    _0006_EB21_CFG_ER AT %MW186040.0 : BOOL; (* EB 구성 에러 *)
    _0006_EB21_DEER AT %MW186040.1 : BOOL; (* EB 운전 중 탈락 *)
    _0006_EB21_IO_DEER AT %MW186041.2 : BOOL; (* EB IO 탈락 에러 *)
    _0006_EB21_IO_TYER AT %MW186041.1 : BOOL; (* EB IO 타입 에러 *)
    _0006_EB30_CFG_ER AT %MW186046.0 : BOOL; (* EB 구성 에러 *)
    _0006_EB30_DEER AT %MW186046.1 : BOOL; (* EB 운전 중 탈락 *)
    _0006_EB30_IO_DEER AT %MW186047.2 : BOOL; (* EB IO 탈락 에러 *)
    _0006_EB30_IO_TYER AT %MW186047.1 : BOOL; (* EB IO 타입 에러 *)
    _0006_EB31_CFG_ER AT %MW186052.0 : BOOL; (* EB 구성 에러 *)
    _0006_EB31_DEER AT %MW186052.1 : BOOL; (* EB 운전 중 탈락 *)
    _0006_EB31_IO_DEER AT %MW186053.2 : BOOL; (* EB IO 탈락 에러 *)
    _0006_EB31_IO_TYER AT %MW186053.1 : BOOL; (* EB IO 타입 에러 *)
    _0006_EB40_CFG_ER AT %MW186058.0 : BOOL; (* EB 구성 에러 *)
    _0006_EB40_DEER AT %MW186058.1 : BOOL; (* EB 운전 중 탈락 *)
    _0006_EB40_IO_DEER AT %MW186059.2 : BOOL; (* EB IO 탈락 에러 *)
    _0006_EB40_IO_TYER AT %MW186059.1 : BOOL; (* EB IO 타입 에러 *)
    _0006_EB41_CFG_ER AT %MW186064.0 : BOOL; (* EB 구성 에러 *)
    _0006_EB41_DEER AT %MW186064.1 : BOOL; (* EB 운전 중 탈락 *)
    _0006_EB41_IO_DEER AT %MW186065.2 : BOOL; (* EB IO 탈락 에러 *)
    _0006_EB41_IO_TYER AT %MW186065.1 : BOOL; (* EB IO 타입 에러 *)
    _0006_EB42_CFG_ER AT %MW186070.0 : BOOL; (* EB 구성 에러 *)
    _0006_EB42_DEER AT %MW186070.1 : BOOL; (* EB 운전 중 탈락 *)
    _0006_EB42_IO_DEER AT %MW186071.2 : BOOL; (* EB IO 탈락 에러 *)
    _0006_EB42_IO_TYER AT %MW186071.1 : BOOL; (* EB IO 타입 에러 *)
    _0007_EB01_CFG_ER AT %MW187022.0 : BOOL; (* EB 구성 에러 *)
    _0007_EB01_DEER AT %MW187022.1 : BOOL; (* EB 운전 중 탈락 *)
    _0007_EB01_IO_DEER AT %MW187023.2 : BOOL; (* EB IO 탈락 에러 *)
    _0007_EB01_IO_TYER AT %MW187023.1 : BOOL; (* EB IO 타입 에러 *)
    _0007_EB02_CFG_ER AT %MW187028.0 : BOOL; (* EB 구성 에러 *)
    _0007_EB02_DEER AT %MW187028.1 : BOOL; (* EB 운전 중 탈락 *)
    _0007_EB02_IO_DEER AT %MW187029.2 : BOOL; (* EB IO 탈락 에러 *)
    _0007_EB02_IO_TYER AT %MW187029.1 : BOOL; (* EB IO 타입 에러 *)
    _0007_EB03_CFG_ER AT %MW187034.0 : BOOL; (* EB 구성 에러 *)
    _0007_EB03_DEER AT %MW187034.1 : BOOL; (* EB 운전 중 탈락 *)
    _0007_EB03_IO_DEER AT %MW187035.2 : BOOL; (* EB IO 탈락 에러 *)
    _0007_EB03_IO_TYER AT %MW187035.1 : BOOL; (* EB IO 타입 에러 *)
    _0007_EB10_CFG_ER AT %MW187040.0 : BOOL; (* EB 구성 에러 *)
    _0007_EB10_DEER AT %MW187040.1 : BOOL; (* EB 운전 중 탈락 *)
    _0007_EB10_IO_DEER AT %MW187041.2 : BOOL; (* EB IO 탈락 에러 *)
    _0007_EB10_IO_TYER AT %MW187041.1 : BOOL; (* EB IO 타입 에러 *)
    _0007_EB11_CFG_ER AT %MW187046.0 : BOOL; (* EB 구성 에러 *)
    _0007_EB11_DEER AT %MW187046.1 : BOOL; (* EB 운전 중 탈락 *)
    _0007_EB11_IO_DEER AT %MW187047.2 : BOOL; (* EB IO 탈락 에러 *)
    _0007_EB11_IO_TYER AT %MW187047.1 : BOOL; (* EB IO 타입 에러 *)
    _0007_EB12_CFG_ER AT %MW187052.0 : BOOL; (* EB 구성 에러 *)
    _0007_EB12_DEER AT %MW187052.1 : BOOL; (* EB 운전 중 탈락 *)
    _0007_EB12_IO_DEER AT %MW187053.2 : BOOL; (* EB IO 탈락 에러 *)
    _0007_EB12_IO_TYER AT %MW187053.1 : BOOL; (* EB IO 타입 에러 *)
    _0007_EB15_CFG_ER AT %MW187058.0 : BOOL; (* EB 구성 에러 *)
    _0007_EB15_DEER AT %MW187058.1 : BOOL; (* EB 운전 중 탈락 *)
    _0007_EB15_IO_DEER AT %MW187059.2 : BOOL; (* EB IO 탈락 에러 *)
    _0007_EB15_IO_TYER AT %MW187059.1 : BOOL; (* EB IO 타입 에러 *)
    _0007_EB16_CFG_ER AT %MW187064.0 : BOOL; (* EB 구성 에러 *)
    _0007_EB16_DEER AT %MW187064.1 : BOOL; (* EB 운전 중 탈락 *)
    _0007_EB16_IO_DEER AT %MW187065.2 : BOOL; (* EB IO 탈락 에러 *)
    _0007_EB16_IO_TYER AT %MW187065.1 : BOOL; (* EB IO 타입 에러 *)
    _0007_EB40_CFG_ER AT %MW187070.0 : BOOL; (* EB 구성 에러 *)
    _0007_EB40_DEER AT %MW187070.1 : BOOL; (* EB 운전 중 탈락 *)
    _0007_EB40_IO_DEER AT %MW187071.2 : BOOL; (* EB IO 탈락 에러 *)
    _0007_EB40_IO_TYER AT %MW187071.1 : BOOL; (* EB IO 타입 에러 *)
    _0007_EB45_CFG_ER AT %MW187076.0 : BOOL; (* EB 구성 에러 *)
    _0007_EB45_DEER AT %MW187076.1 : BOOL; (* EB 운전 중 탈락 *)
    _0007_EB45_IO_DEER AT %MW187077.2 : BOOL; (* EB IO 탈락 에러 *)
    _0007_EB45_IO_TYER AT %MW187077.1 : BOOL; (* EB IO 타입 에러 *)
    _0007_EB63_CFG_ER AT %MW187088.0 : BOOL; (* EB 구성 에러 *)
    _0007_EB63_DEER AT %MW187088.1 : BOOL; (* EB 운전 중 탈락 *)
    _0007_EB63_IO_DEER AT %MW187089.2 : BOOL; (* EB IO 탈락 에러 *)
    _0007_EB63_IO_TYER AT %MW187089.1 : BOOL; (* EB IO 타입 에러 *)
    _MW87632_06 AT %MW87632.6 : BOOL; (* MCP 출력전원 CP TRIP *)
    _MW87632_07 AT %MW87632.7 : BOOL; (* MCP PC랙전원 CP TRIP *)
    _MW87632_08 AT %MW87632.8 : BOOL; (* MCP 현황판 CP TRIP *)
END_VAR

FUNCTION_BLOCK FB406_Car_Type_Move_Line_v1
VAR_INPUT RETAIN
    FWD_Pulse : BOOL;
    RET_Pulse : BOOL;
END_VAR
VAR_IN_OUT
    Source_DB : ARRAY[0..599] OF WORD;
END_VAR
VAR_INPUT
    Start_Add : INT;
    Stn_AMTG : INT;
    Word_per_Stn : INT;
    Cpu_Run_Pulse : BOOL;
END_VAR
VAR_OUTPUT
    Complete : BOOL;
END_VAR
VAR
    END : INT;
    Number_of_Array : INT;
    Temp1 : INT;
END_VAR

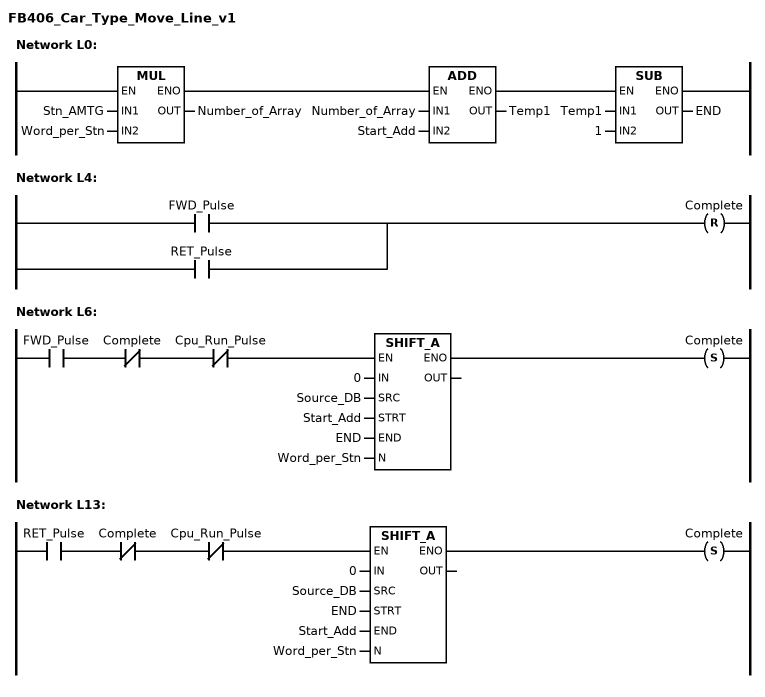
(* Rung L0 *)
Number_of_Array := Stn_AMTG * Word_per_Stn;
Temp1 := Number_of_Array + Start_Add;
END := Temp1 - 1;
(* Rung L4 *)
IF FWD_Pulse OR RET_Pulse THEN Complete := FALSE; END_IF;
(* Rung L6 *)
IF FWD_Pulse AND NOT Complete AND NOT Cpu_Run_Pulse THEN
    SHIFT_A(IN := 0, SRC := Source_DB, STRT := Start_Add, END := END, N := Word_per_Stn);
    Complete := TRUE;
END_IF;
(* Rung L13 *)
IF RET_Pulse AND NOT Complete AND NOT Cpu_Run_Pulse THEN
    SHIFT_A(IN := 0, SRC := Source_DB, STRT := END, END := Start_Add, N := Word_per_Stn);
    Complete := TRUE;
END_IF;
END_FUNCTION_BLOCK

FUNCTION_BLOCK FB407_Car_Type_Move_Stn_v1
VAR_INPUT RETAIN
    FWD_Pulse : BOOL;
    RET_Pulse : BOOL;
END_VAR
VAR_IN_OUT
    Source_DB : ARRAY[0..599] OF WORD;
    Dest_DB : ARRAY[0..599] OF WORD;
END_VAR
VAR_INPUT
    Source_Add : INT;
    Dest_Add : INT;
    Word_per_Stn : INT;
    Cpu_Run_Pulse : BOOL;
END_VAR
VAR_OUTPUT
    Complete : BOOL;
END_VAR
VAR
    _t1 : DINT;
    _t2 : DINT;
END_VAR

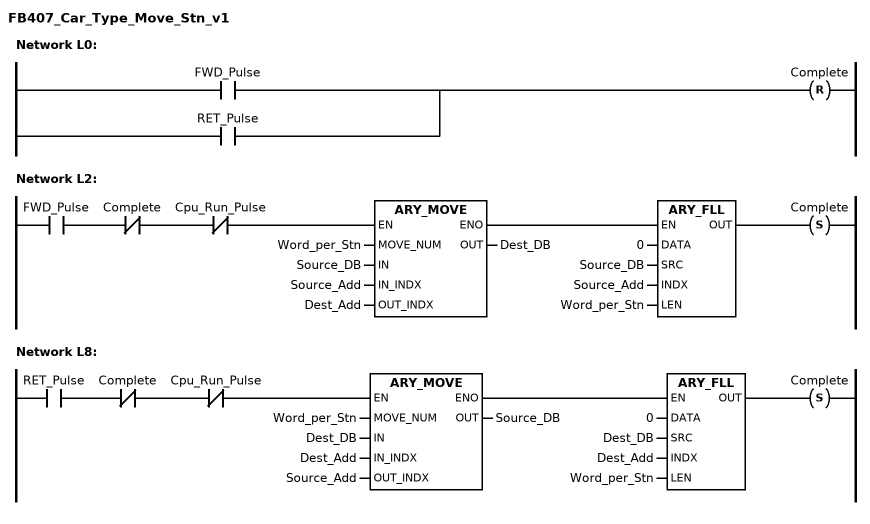
(* Rung L0 *)
IF FWD_Pulse OR RET_Pulse THEN Complete := FALSE; END_IF;
(* Rung L2 *)
IF FWD_Pulse AND NOT Complete AND NOT Cpu_Run_Pulse THEN
    Dest_DB := ARY_MOVE(MOVE_NUM := Word_per_Stn, IN := Source_DB, IN_INDX := Source_Add, OUT_INDX := Dest_Add);
    _t1 := ARY_FLL(DATA := 0, SRC := Source_DB, INDX := Source_Add, LEN := Word_per_Stn);
END_IF;
IF _t1 THEN Complete := TRUE; END_IF;
(* Rung L8 *)
IF RET_Pulse AND NOT Complete AND NOT Cpu_Run_Pulse THEN
    Source_DB := ARY_MOVE(MOVE_NUM := Word_per_Stn, IN := Dest_DB, IN_INDX := Dest_Add, OUT_INDX := Source_Add);
    _t2 := ARY_FLL(DATA := 0, SRC := Dest_DB, INDX := Dest_Add, LEN := Word_per_Stn);
END_IF;
IF _t2 THEN Complete := TRUE; END_IF;
END_FUNCTION_BLOCK

FUNCTION_BLOCK FB409_Car_Type_Clear_v1
VAR_INPUT RETAIN
    Clear_Pulse : BOOL;
END_VAR
VAR_IN_OUT
    Dest_DB : ARRAY[0..599] OF WORD;
END_VAR
VAR_INPUT
    Dest_Add : INT;
    Len_per_Stn_Word : INT;
    Cpu_Run_Pulse : BOOL;
END_VAR
VAR_OUTPUT
    Complete : BOOL;
END_VAR
VAR
    _t1 : DINT;
END_VAR

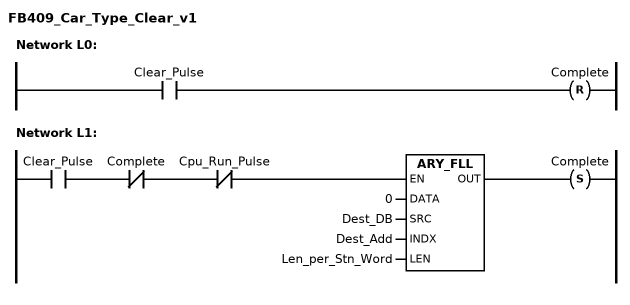
(* Rung L0 *)
IF Clear_Pulse THEN Complete := FALSE; END_IF;
(* Rung L1 *)
IF Clear_Pulse AND NOT Complete AND NOT Cpu_Run_Pulse THEN
    _t1 := ARY_FLL(DATA := 0, SRC := Dest_DB, INDX := Dest_Add, LEN := Len_per_Stn_Word);
END_IF;
IF _t1 THEN Complete := TRUE; END_IF;
END_FUNCTION_BLOCK

FUNCTION_BLOCK FB470_HMI_BType_Modify_LS
VAR_INPUT
    CCR_ON : BOOL;
    BT_Modify_ON : BOOL;
    BT_Combi_OK : BOOL;
    STN_SEL : UINT;
    Word_per_Stn : UINT;
    SET : BOOL;
    RST : BOOL;
END_VAR
VAR_IN_OUT
    HMI_Disp_DB : ARRAY[0..19] OF WORD;
    Modify_DB : ARRAY[0..19] OF WORD;
    CType_DB : ARRAY[0..599] OF WORD;
END_VAR
VAR_OUTPUT
    LP_CCR_On : BOOL;
    LP_Modify_On : BOOL;
END_VAR
VAR
    INDEX : INT;
    JMP : BOOL;
    NE : BOOL;
    RST_Delay : BOOL;
    SET_Delay : BOOL;
    STN_SEL_Temp : UINT;
    STN_SEL_Temp2 : UINT;
    T1 : TON;
    T2 : TON;
    Temp : WORD;
END_VAR
VAR
    _t1 : BOOL;
    _t2 : BOOL;
    _p3 : BOOL;
    _e4 : R_TRIG;
    _e5 : R_TRIG;
    _t6 : BOOL;
    _e7 : R_TRIG;
    _t8 : BOOL;
    _e9 : R_TRIG;
    _t10 : BOOL;
END_VAR

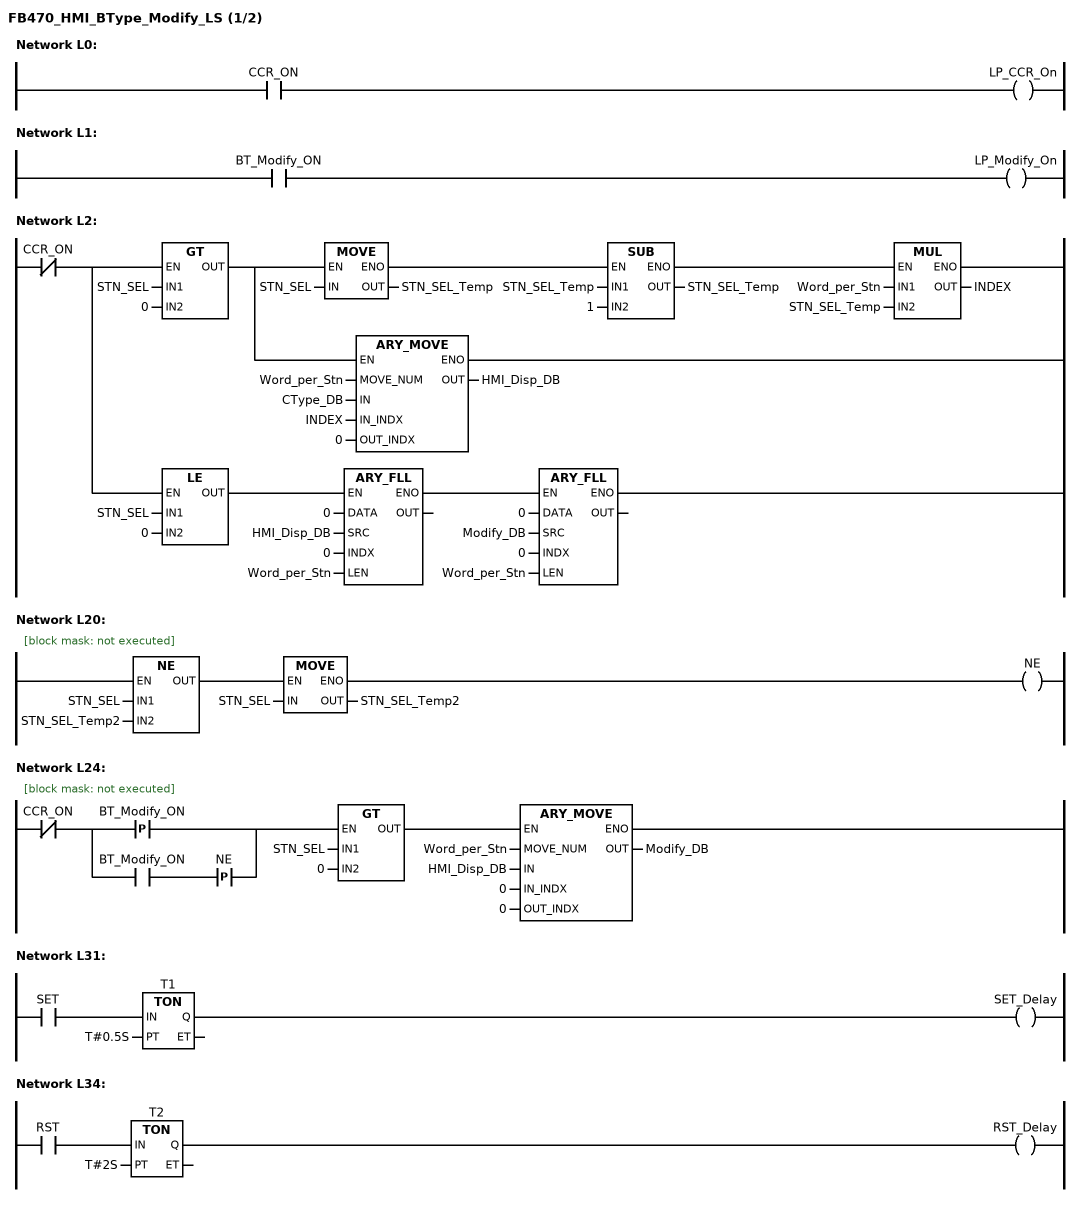
(* Rung L0 *)
LP_CCR_On := CCR_ON;
(* Rung L1 *)
LP_Modify_On := BT_Modify_ON;
(* Rung L2 *)
IF NOT CCR_ON THEN _t1 := STN_SEL > 0; END_IF;
IF _t1 THEN
    STN_SEL_Temp := STN_SEL;
    STN_SEL_Temp := STN_SEL_Temp - 1;
    INDEX := Word_per_Stn * STN_SEL_Temp;
    HMI_Disp_DB := ARY_MOVE(MOVE_NUM := Word_per_Stn, IN := CType_DB, IN_INDX := INDEX, OUT_INDX := 0);
END_IF;
IF NOT CCR_ON THEN _t2 := STN_SEL <= 0; END_IF;
IF _t2 THEN
    ARY_FLL(DATA := 0, SRC := HMI_Disp_DB, INDX := 0, LEN := Word_per_Stn);
    ARY_FLL(DATA := 0, SRC := Modify_DB, INDX := 0, LEN := Word_per_Stn);
END_IF;
(* Rung L20 is block-masked: not executed *)
// _p3 := STN_SEL <> STN_SEL_Temp2;
// IF _p3 THEN STN_SEL_Temp2 := STN_SEL; END_IF;
// NE := _p3;
(* Rung L24 is block-masked: not executed *)
// _e4(CLK := BT_Modify_ON);
// _e5(CLK := NE);
// IF NOT CCR_ON AND (_e4.Q OR (BT_Modify_ON AND _e5.Q)) THEN _t6 := STN_SEL > 0; END_IF;
// IF _t6 THEN
//     Modify_DB := ARY_MOVE(MOVE_NUM := Word_per_Stn, IN := HMI_Disp_DB, IN_INDX := 0, OUT_INDX := 0);
// END_IF;
(* Rung L31 *)
T1(IN := SET, PT := T#0.5S);
SET_Delay := T1.Q;
(* Rung L34 *)
T2(IN := RST, PT := T#2S);
RST_Delay := T2.Q;

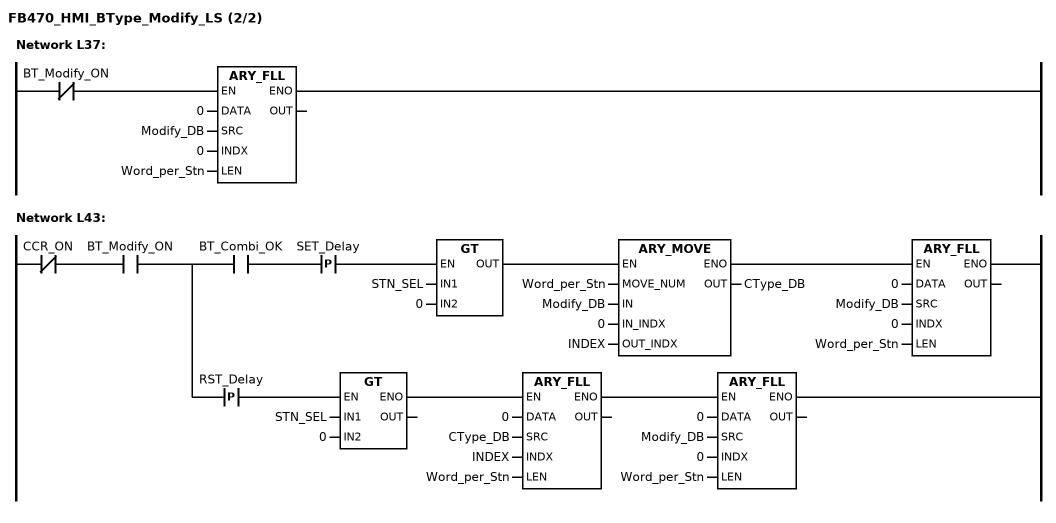
(* Rung L37 *)
IF NOT BT_Modify_ON THEN ARY_FLL(DATA := 0, SRC := Modify_DB, INDX := 0, LEN := Word_per_Stn); END_IF;
(* Rung L43 *)
_e7(CLK := SET_Delay);
IF NOT CCR_ON AND BT_Modify_ON AND BT_Combi_OK AND _e7.Q THEN _t8 := STN_SEL > 0; END_IF;
IF _t8 THEN
    CType_DB := ARY_MOVE(MOVE_NUM := Word_per_Stn, IN := Modify_DB, IN_INDX := 0, OUT_INDX := INDEX);
    ARY_FLL(DATA := 0, SRC := Modify_DB, INDX := 0, LEN := Word_per_Stn);
END_IF;
_e9(CLK := RST_Delay);
IF NOT CCR_ON AND BT_Modify_ON AND _e9.Q THEN
    _t10 := STN_SEL > 0;
    ARY_FLL(DATA := 0, SRC := CType_DB, INDX := INDEX, LEN := Word_per_Stn);
    ARY_FLL(DATA := 0, SRC := Modify_DB, INDX := 0, LEN := Word_per_Stn);
END_IF;
END_FUNCTION_BLOCK

FUNCTION_BLOCK FB501_CYCLE_TIME_AVE_v2
VAR_INPUT
    Auto_Run : BOOL;
    BT_ByPass : BOOL;
    Cycle_Start : BOOL;
    Cycle_End : BOOL;
    Count_RST : BOOL;
END_VAR
VAR_OUTPUT
    MAX : INT;
    MIN : INT;
    AVE : INT;
    Count : INT;
    Current : INT;
    Previous : INT;
    No_Work_Current : INT;
    No_Work_Previous : INT;
    Accumulated : DINT;
END_VAR
VAR
    AVE_D : DINT;
    Count_D : DINT;
    Current_D : DINT;
    MAX_D : DINT;
    MIN_D : DINT;
    NO_TIME_CHECK : BOOL;
    No_Work_Current_D : DINT;
    No_Work_Previous_D : DINT;
    Previous_D : DINT;
    Temp1 : DWORD;
END_VAR
VAR
    _e1 : R_TRIG;
    _p2 : BOOL;
    _e3 : R_TRIG;
    _e4 : R_TRIG;
    _t5 : BOOL;
END_VAR

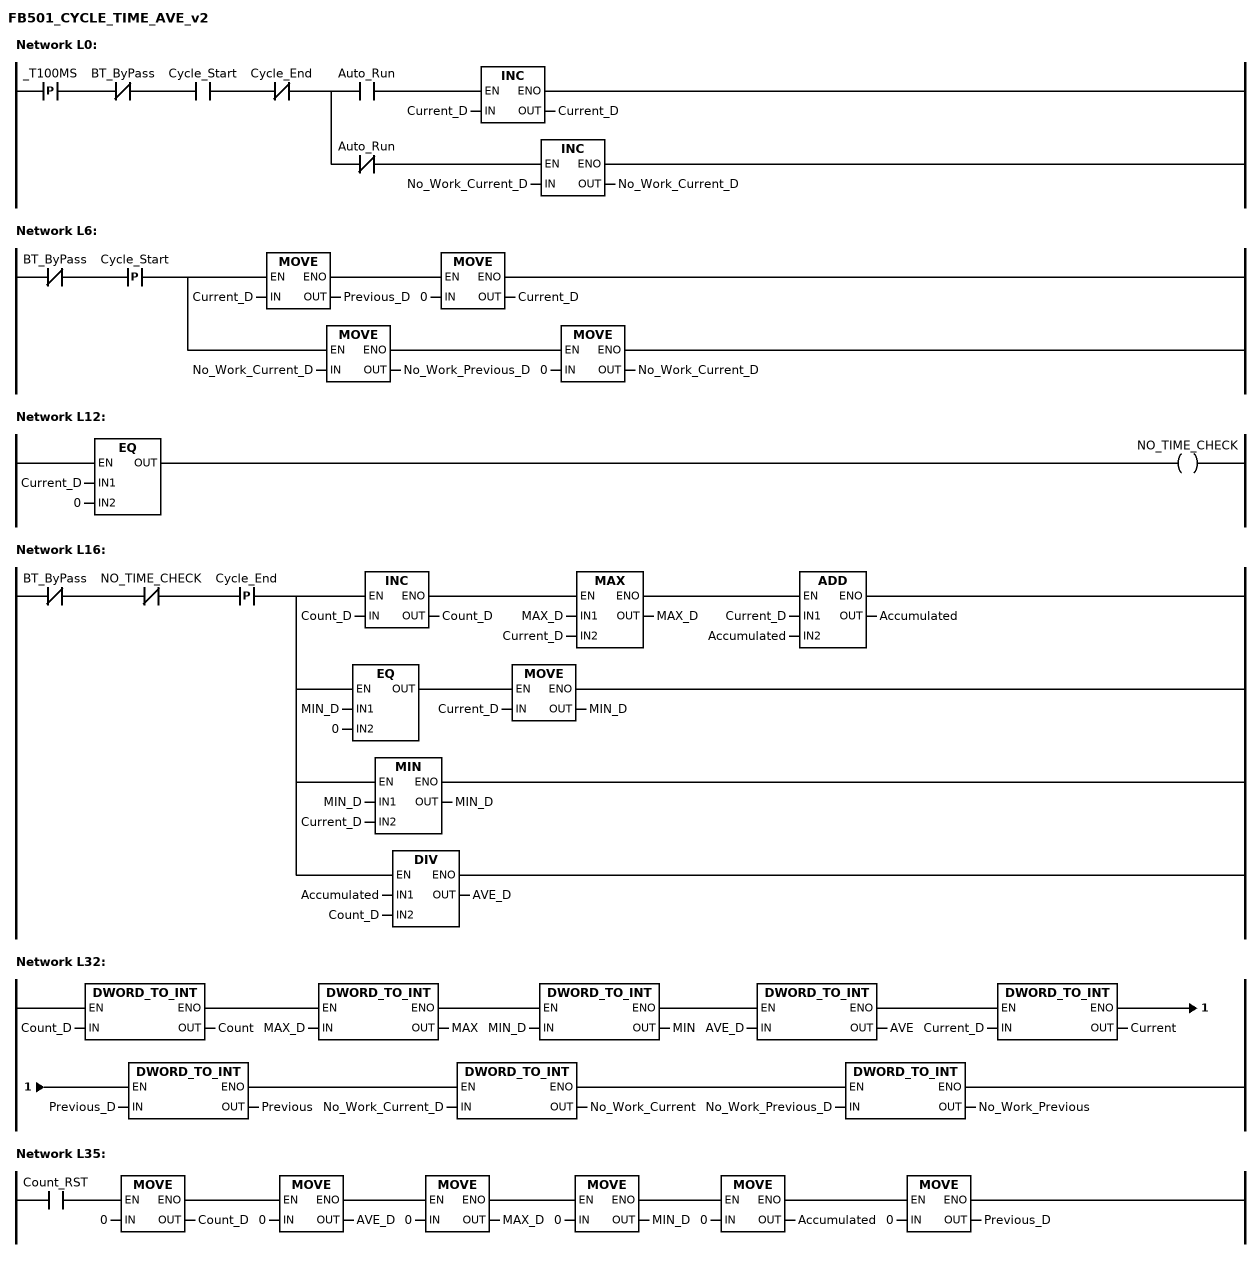
(* Rung L0 *)
_e1(CLK := _T100MS);
_p2 := _e1.Q AND NOT BT_ByPass AND Cycle_Start AND NOT Cycle_End;
IF _p2 AND Auto_Run THEN Current_D := INC(Current_D); END_IF;
IF _p2 AND NOT Auto_Run THEN No_Work_Current_D := INC(No_Work_Current_D); END_IF;
(* Rung L6 *)
_e3(CLK := Cycle_Start);
IF NOT BT_ByPass AND _e3.Q THEN
    Previous_D := Current_D;
    Current_D := 0;
    No_Work_Previous_D := No_Work_Current_D;
    No_Work_Current_D := 0;
END_IF;
(* Rung L12 *)
NO_TIME_CHECK := Current_D = 0;
(* Rung L16 *)
_e4(CLK := Cycle_End);
IF NOT BT_ByPass AND NOT NO_TIME_CHECK AND _e4.Q THEN
    Count_D := INC(Count_D);
    MAX_D := MAX(MAX_D, Current_D);
    Accumulated := Current_D + Accumulated;
    _t5 := MIN_D = 0;
END_IF;
IF _t5 THEN MIN_D := Current_D; END_IF;
IF NOT BT_ByPass AND NOT NO_TIME_CHECK AND _e4.Q THEN
    MIN_D := MIN(MIN_D, Current_D);
    AVE_D := Accumulated / Count_D;
END_IF;
(* Rung L32 *)
Count := DWORD_TO_INT(Count_D);
MAX := DWORD_TO_INT(MAX_D);
MIN := DWORD_TO_INT(MIN_D);
AVE := DWORD_TO_INT(AVE_D);
Current := DWORD_TO_INT(Current_D);
Previous := DWORD_TO_INT(Previous_D);
No_Work_Current := DWORD_TO_INT(No_Work_Current_D);
No_Work_Previous := DWORD_TO_INT(No_Work_Previous_D);
(* Rung L35 *)
IF Count_RST THEN
    Count_D := 0;
    AVE_D := 0;
    MAX_D := 0;
    MIN_D := 0;
    Accumulated := 0;
    Previous_D := 0;
END_IF;
END_FUNCTION_BLOCK

FUNCTION_BLOCK ACT_10_CYL
VAR_INPUT
    사용유무 : BOOL;
    운전준비 : BOOL;
    전진보조 : BOOL;
    후진보조 : BOOL;
    전진단수량 : UINT;
    후진단수량 : UINT;
    전진단1 : BOOL;
    후진단1 : BOOL;
    전진단2 : BOOL;
    후진단2 : BOOL;
    전진단3 : BOOL;
    후진단3 : BOOL;
    전진단4 : BOOL;
    후진단4 : BOOL;
    전진단5 : BOOL;
    후진단5 : BOOL;
    전진단6 : BOOL;
    후진단6 : BOOL;
    전진단7 : BOOL;
    후진단7 : BOOL;
    전진단8 : BOOL;
    후진단8 : BOOL;
    전진단9 : BOOL;
    후진단9 : BOOL;
    전진단10 : BOOL;
    후진단10 : BOOL;
    전진단_지연시간 : TIME;
    후진단_지연시간 : TIME;
    LS_ERR1_지연시간 : TIME;
    LS_ERR2_지연시간 : TIME;
    이상리셋 : BOOL;
END_VAR
VAR_OUTPUT
    SOL_ADV_출력 : BOOL;
    SOL_RET_출력 : BOOL;
    M_전진단 : BOOL;
    M_후진단 : BOOL;
    M_전진에러 : BOOL;
    M_후진에러 : BOOL;
    ADV_LAMP : WORD;
    RET_LAMP : WORD;
END_VAR
VAR
    ACT_USE : BOOL;
    ADV_END_TIME : TON;
    ADV_SOL_MEMO : BOOL;
    ERR_TIME1 : TON;
    LP_ADV_1 : BOOL;
    LP_ADV_10 : BOOL;
    LP_ADV_2 : BOOL;
    LP_ADV_3 : BOOL;
    LP_ADV_4 : BOOL;
    LP_ADV_5 : BOOL;
    LP_ADV_6 : BOOL;
    LP_ADV_7 : BOOL;
    LP_ADV_8 : BOOL;
    LP_ADV_9 : BOOL;
    LP_RET_1 : BOOL;
    LP_RET_10 : BOOL;
    LP_RET_2 : BOOL;
    LP_RET_3 : BOOL;
    LP_RET_4 : BOOL;
    LP_RET_5 : BOOL;
    LP_RET_6 : BOOL;
    LP_RET_7 : BOOL;
    LP_RET_8 : BOOL;
    LP_RET_9 : BOOL;
    LS_ERR_1 : BOOL;
    LS_ERR_2 : BOOL;
    RET_END_TIME : TON;
    RET_END_TIME1 : TON;
    RET_END_TIME2 : TON;
    RET_ERR_TIME : TON;
    RET_SOL_MEMO : BOOL;
    전진단10_PASS : BOOL;
    전진단2_PASS : BOOL;
    전진단3_PASS : BOOL;
    전진단4_PASS : BOOL;
    전진단5_PASS : BOOL;
    전진단6_PASS : BOOL;
    전진단7_PASS : BOOL;
    전진단8_PASS : BOOL;
    전진단9_PASS : BOOL;
    전진단LAMP_H_AUX : BYTE;
    전진단LAMP_L_AUX : BYTE;
    후진단10_PASS : BOOL;
    후진단2_PASS : BOOL;
    후진단3_PASS : BOOL;
    후진단4_PASS : BOOL;
    후진단5_PASS : BOOL;
    후진단6_PASS : BOOL;
    후진단7_PASS : BOOL;
    후진단8_PASS : BOOL;
    후진단9_PASS : BOOL;
    후진단LAMP_H_AUX : BYTE;
    후진단LAMP_L_AUX : BYTE;
END_VAR

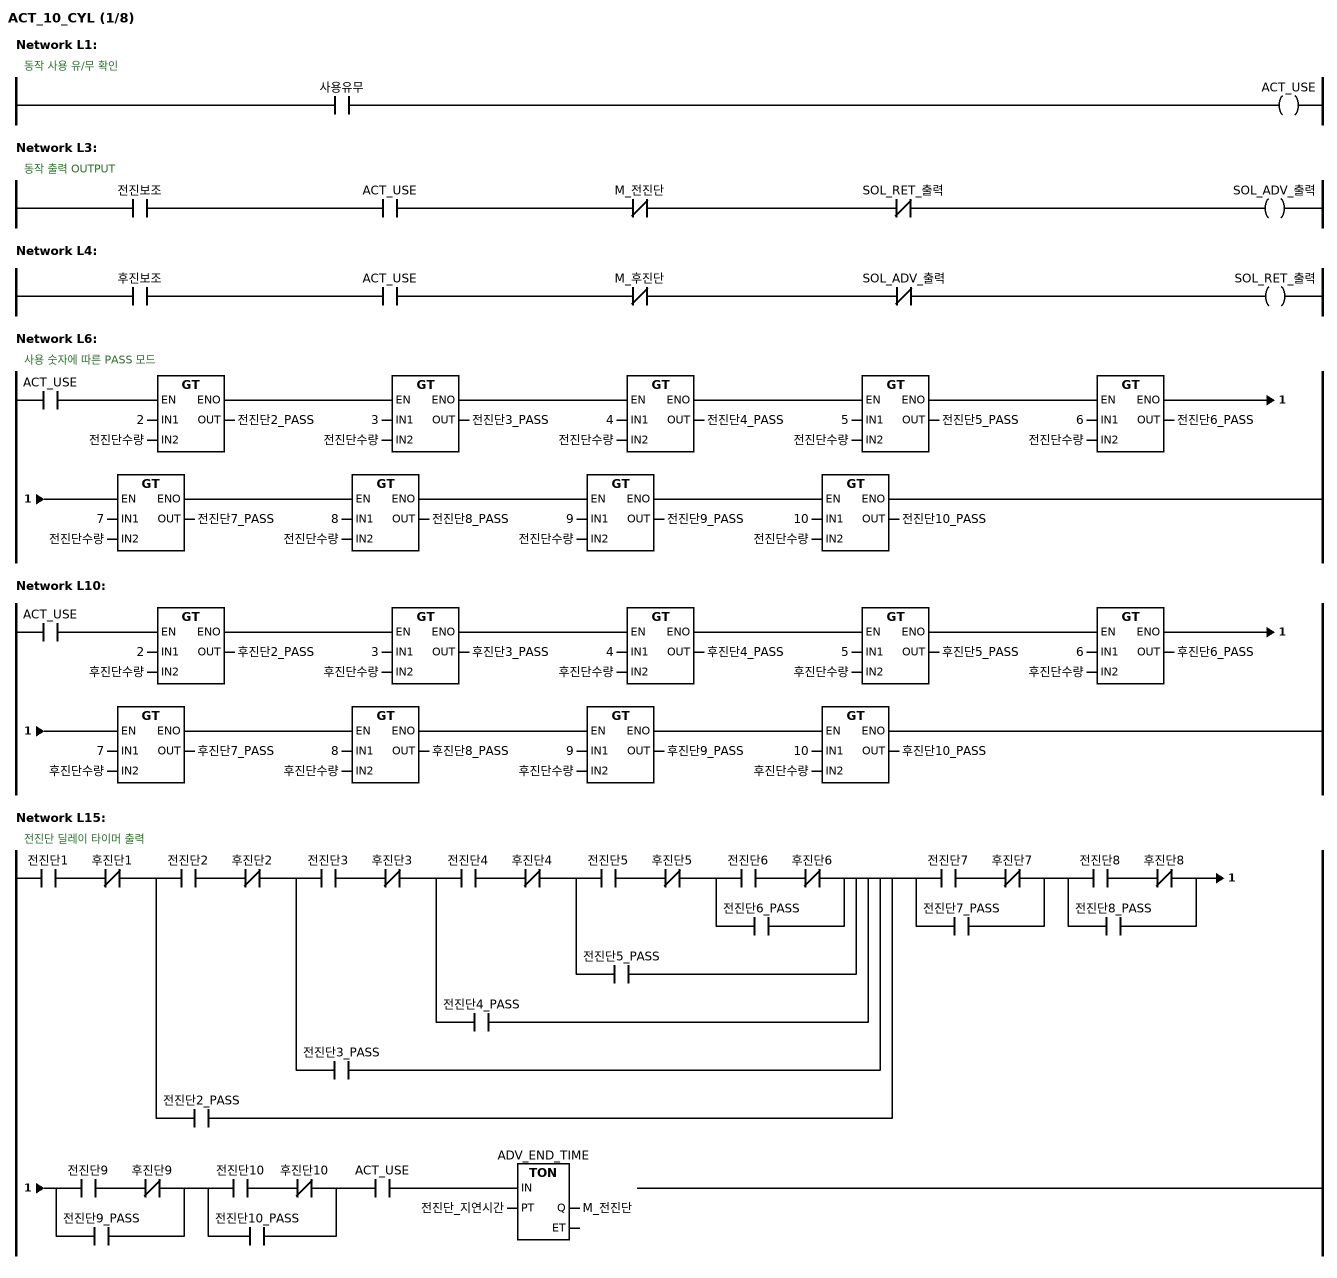
(* 동작 사용 유/무 확인 *)
(* Rung L1 *)
ACT_USE := 사용유무;
(* 동작 출력 OUTPUT *)
(* Rung L3 *)
SOL_ADV_출력 := 전진보조 AND ACT_USE AND NOT M_전진단 AND NOT SOL_RET_출력;
(* Rung L4 *)
SOL_RET_출력 := 후진보조 AND ACT_USE AND NOT M_후진단 AND NOT SOL_ADV_출력;
(* 사용 숫자에 따른 PASS 모드 *)
(* Rung L6 *)
IF ACT_USE THEN
    전진단2_PASS := 2 > 전진단수량;
    전진단3_PASS := 3 > 전진단수량;
    전진단4_PASS := 4 > 전진단수량;
    전진단5_PASS := 5 > 전진단수량;
    전진단6_PASS := 6 > 전진단수량;
    전진단7_PASS := 7 > 전진단수량;
    전진단8_PASS := 8 > 전진단수량;
    전진단9_PASS := 9 > 전진단수량;
    전진단10_PASS := 10 > 전진단수량;
END_IF;
(* Rung L10 *)
IF ACT_USE THEN
    후진단2_PASS := 2 > 후진단수량;
    후진단3_PASS := 3 > 후진단수량;
    후진단4_PASS := 4 > 후진단수량;
    후진단5_PASS := 5 > 후진단수량;
    후진단6_PASS := 6 > 후진단수량;
    후진단7_PASS := 7 > 후진단수량;
    후진단8_PASS := 8 > 후진단수량;
    후진단9_PASS := 9 > 후진단수량;
    후진단10_PASS := 10 > 후진단수량;
END_IF;
(* 전진단 딜레이 타이머 출력 *)
(* Rung L15 *)
ADV_END_TIME(IN := 전진단1 AND NOT 후진단1 AND ((전진단2 AND NOT 후진단2 AND ((전진단3 AND NOT 후진단3 AND ((전진단4 AND NOT 후진단4 AND ((전진단5 AND NOT 후진단5 AND ((전진단6 AND NOT 후진단6) OR 전진단6_PASS)) OR 전진단5_PASS)) OR 전진단4_PASS)) OR 전진단3_PASS)) OR 전진단2_PASS) AND ((전진단7 AND NOT 후진단7) OR 전진단7_PASS) AND ((전진단8 AND NOT 후진단8) OR 전진단8_PASS) AND ((전진단9 AND NOT 후진단9) OR 전진단9_PASS) AND ((전진단10 AND NOT 후진단10) OR 전진단10_PASS) AND ACT_USE, PT := 전진단_지연시간, Q => M_전진단);

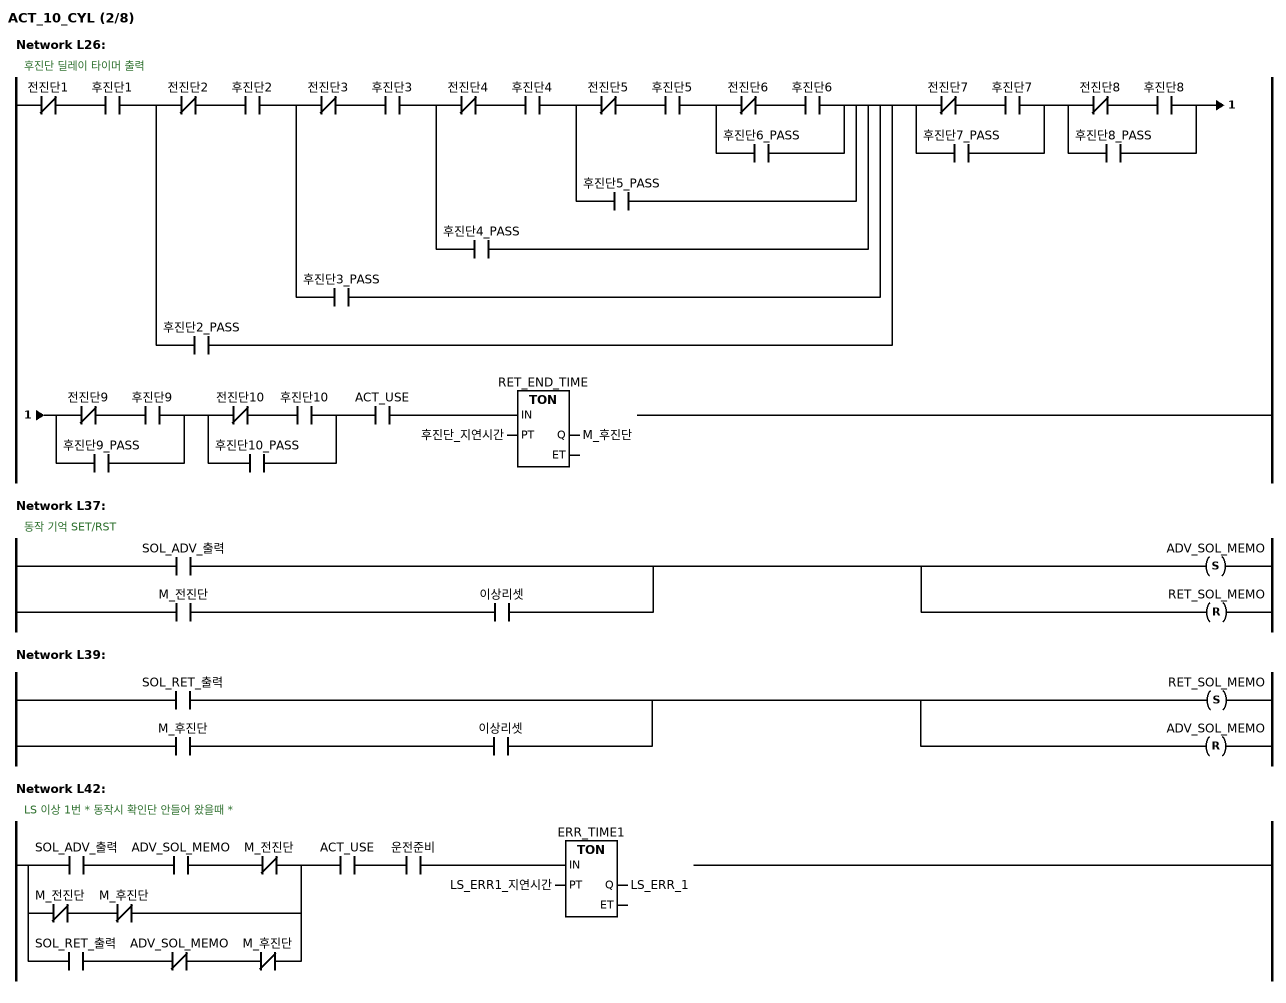
(* 후진단 딜레이 타이머 출력 *)
(* Rung L26 *)
RET_END_TIME(IN := NOT 전진단1 AND 후진단1 AND ((NOT 전진단2 AND 후진단2 AND ((NOT 전진단3 AND 후진단3 AND ((NOT 전진단4 AND 후진단4 AND ((NOT 전진단5 AND 후진단5 AND ((NOT 전진단6 AND 후진단6) OR 후진단6_PASS)) OR 후진단5_PASS)) OR 후진단4_PASS)) OR 후진단3_PASS)) OR 후진단2_PASS) AND ((NOT 전진단7 AND 후진단7) OR 후진단7_PASS) AND ((NOT 전진단8 AND 후진단8) OR 후진단8_PASS) AND ((NOT 전진단9 AND 후진단9) OR 후진단9_PASS) AND ((NOT 전진단10 AND 후진단10) OR 후진단10_PASS) AND ACT_USE, PT := 후진단_지연시간, Q => M_후진단);
(* 동작 기억 SET/RST *)
(* Rung L37 *)
IF SOL_ADV_출력 OR (M_전진단 AND 이상리셋) THEN
    ADV_SOL_MEMO := TRUE;
    RET_SOL_MEMO := FALSE;
END_IF;
(* Rung L39 *)
IF SOL_RET_출력 OR (M_후진단 AND 이상리셋) THEN
    RET_SOL_MEMO := TRUE;
    ADV_SOL_MEMO := FALSE;
END_IF;
(* LS 이상 1번 * 동작시 확인단 안들어 왔을때 * *)
(* Rung L42 *)
ERR_TIME1(IN := ((SOL_ADV_출력 AND ADV_SOL_MEMO AND NOT M_전진단) OR (NOT M_전진단 AND NOT M_후진단) OR (SOL_RET_출력 AND NOT ADV_SOL_MEMO AND NOT M_후진단)) AND ACT_USE AND 운전준비, PT := LS_ERR1_지연시간, Q => LS_ERR_1);

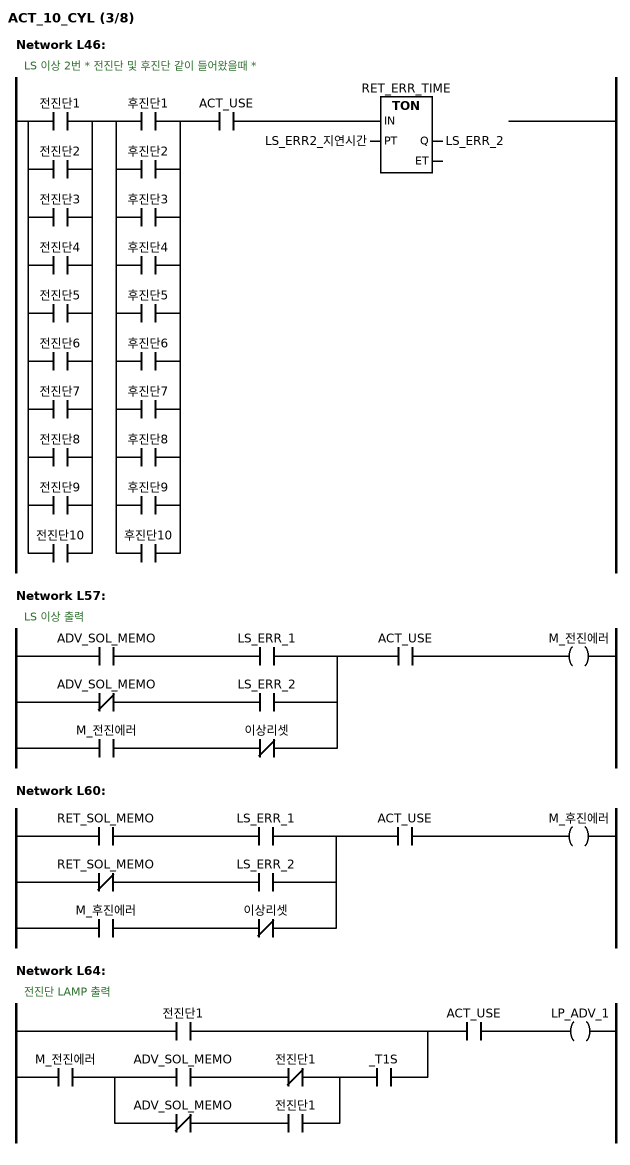
(* LS 이상 2번 * 전진단 및 후진단 같이 들어왔을때 * *)
(* Rung L46 *)
RET_ERR_TIME(IN := (전진단1 OR 전진단2 OR 전진단3 OR 전진단4 OR 전진단5 OR 전진단6 OR 전진단7 OR 전진단8 OR 전진단9 OR 전진단10) AND (후진단1 OR 후진단2 OR 후진단3 OR 후진단4 OR 후진단5 OR 후진단6 OR 후진단7 OR 후진단8 OR 후진단9 OR 후진단10) AND ACT_USE, PT := LS_ERR2_지연시간, Q => LS_ERR_2);
(* LS 이상 출력 *)
(* Rung L57 *)
M_전진에러 := ((ADV_SOL_MEMO AND LS_ERR_1) OR (NOT ADV_SOL_MEMO AND LS_ERR_2) OR (M_전진에러 AND NOT 이상리셋)) AND ACT_USE;
(* Rung L60 *)
M_후진에러 := ((RET_SOL_MEMO AND LS_ERR_1) OR (NOT RET_SOL_MEMO AND LS_ERR_2) OR (M_후진에러 AND NOT 이상리셋)) AND ACT_USE;
(* 전진단 LAMP 출력 *)
(* Rung L64 *)
LP_ADV_1 := (전진단1 OR (M_전진에러 AND ((ADV_SOL_MEMO AND NOT 전진단1) OR (NOT ADV_SOL_MEMO AND 전진단1)) AND _T1S)) AND ACT_USE;

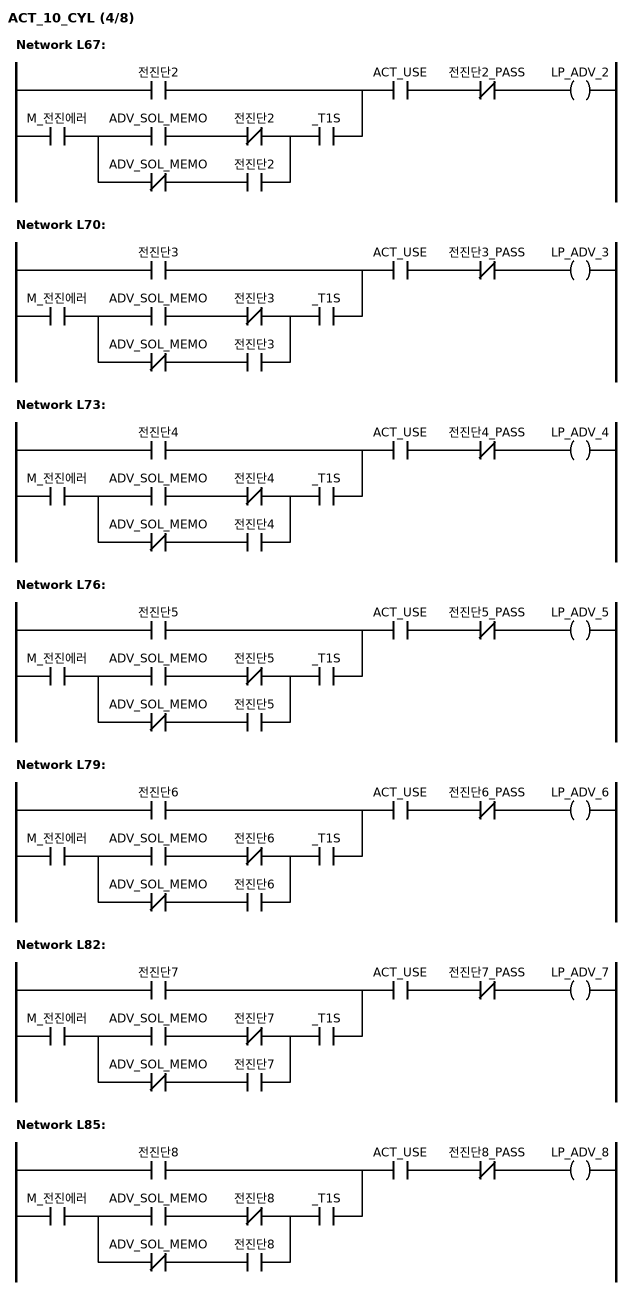
(* Rung L67 *)
LP_ADV_2 := (전진단2 OR (M_전진에러 AND ((ADV_SOL_MEMO AND NOT 전진단2) OR (NOT ADV_SOL_MEMO AND 전진단2)) AND _T1S)) AND ACT_USE AND NOT 전진단2_PASS;
(* Rung L70 *)
LP_ADV_3 := (전진단3 OR (M_전진에러 AND ((ADV_SOL_MEMO AND NOT 전진단3) OR (NOT ADV_SOL_MEMO AND 전진단3)) AND _T1S)) AND ACT_USE AND NOT 전진단3_PASS;
(* Rung L73 *)
LP_ADV_4 := (전진단4 OR (M_전진에러 AND ((ADV_SOL_MEMO AND NOT 전진단4) OR (NOT ADV_SOL_MEMO AND 전진단4)) AND _T1S)) AND ACT_USE AND NOT 전진단4_PASS;
(* Rung L76 *)
LP_ADV_5 := (전진단5 OR (M_전진에러 AND ((ADV_SOL_MEMO AND NOT 전진단5) OR (NOT ADV_SOL_MEMO AND 전진단5)) AND _T1S)) AND ACT_USE AND NOT 전진단5_PASS;
(* Rung L79 *)
LP_ADV_6 := (전진단6 OR (M_전진에러 AND ((ADV_SOL_MEMO AND NOT 전진단6) OR (NOT ADV_SOL_MEMO AND 전진단6)) AND _T1S)) AND ACT_USE AND NOT 전진단6_PASS;
(* Rung L82 *)
LP_ADV_7 := (전진단7 OR (M_전진에러 AND ((ADV_SOL_MEMO AND NOT 전진단7) OR (NOT ADV_SOL_MEMO AND 전진단7)) AND _T1S)) AND ACT_USE AND NOT 전진단7_PASS;
(* Rung L85 *)
LP_ADV_8 := (전진단8 OR (M_전진에러 AND ((ADV_SOL_MEMO AND NOT 전진단8) OR (NOT ADV_SOL_MEMO AND 전진단8)) AND _T1S)) AND ACT_USE AND NOT 전진단8_PASS;

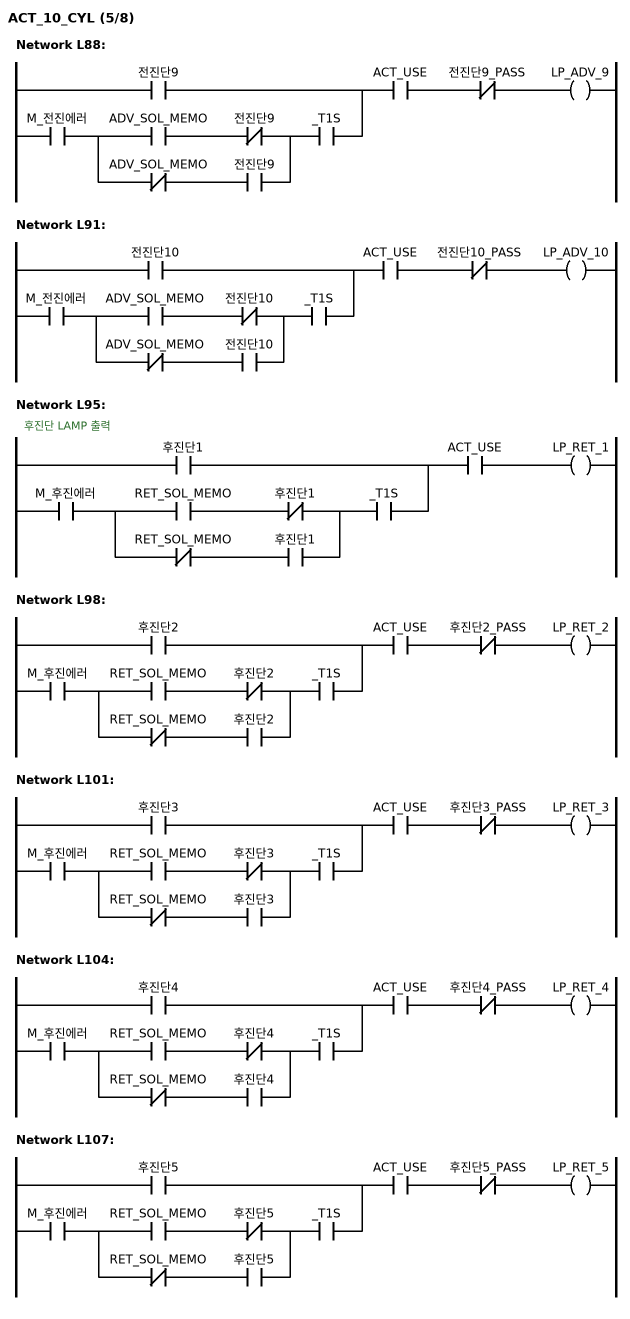
(* Rung L88 *)
LP_ADV_9 := (전진단9 OR (M_전진에러 AND ((ADV_SOL_MEMO AND NOT 전진단9) OR (NOT ADV_SOL_MEMO AND 전진단9)) AND _T1S)) AND ACT_USE AND NOT 전진단9_PASS;
(* Rung L91 *)
LP_ADV_10 := (전진단10 OR (M_전진에러 AND ((ADV_SOL_MEMO AND NOT 전진단10) OR (NOT ADV_SOL_MEMO AND 전진단10)) AND _T1S)) AND ACT_USE AND NOT 전진단10_PASS;
(* 후진단 LAMP 출력 *)
(* Rung L95 *)
LP_RET_1 := (후진단1 OR (M_후진에러 AND ((RET_SOL_MEMO AND NOT 후진단1) OR (NOT RET_SOL_MEMO AND 후진단1)) AND _T1S)) AND ACT_USE;
(* Rung L98 *)
LP_RET_2 := (후진단2 OR (M_후진에러 AND ((RET_SOL_MEMO AND NOT 후진단2) OR (NOT RET_SOL_MEMO AND 후진단2)) AND _T1S)) AND ACT_USE AND NOT 후진단2_PASS;
(* Rung L101 *)
LP_RET_3 := (후진단3 OR (M_후진에러 AND ((RET_SOL_MEMO AND NOT 후진단3) OR (NOT RET_SOL_MEMO AND 후진단3)) AND _T1S)) AND ACT_USE AND NOT 후진단3_PASS;
(* Rung L104 *)
LP_RET_4 := (후진단4 OR (M_후진에러 AND ((RET_SOL_MEMO AND NOT 후진단4) OR (NOT RET_SOL_MEMO AND 후진단4)) AND _T1S)) AND ACT_USE AND NOT 후진단4_PASS;
(* Rung L107 *)
LP_RET_5 := (후진단5 OR (M_후진에러 AND ((RET_SOL_MEMO AND NOT 후진단5) OR (NOT RET_SOL_MEMO AND 후진단5)) AND _T1S)) AND ACT_USE AND NOT 후진단5_PASS;

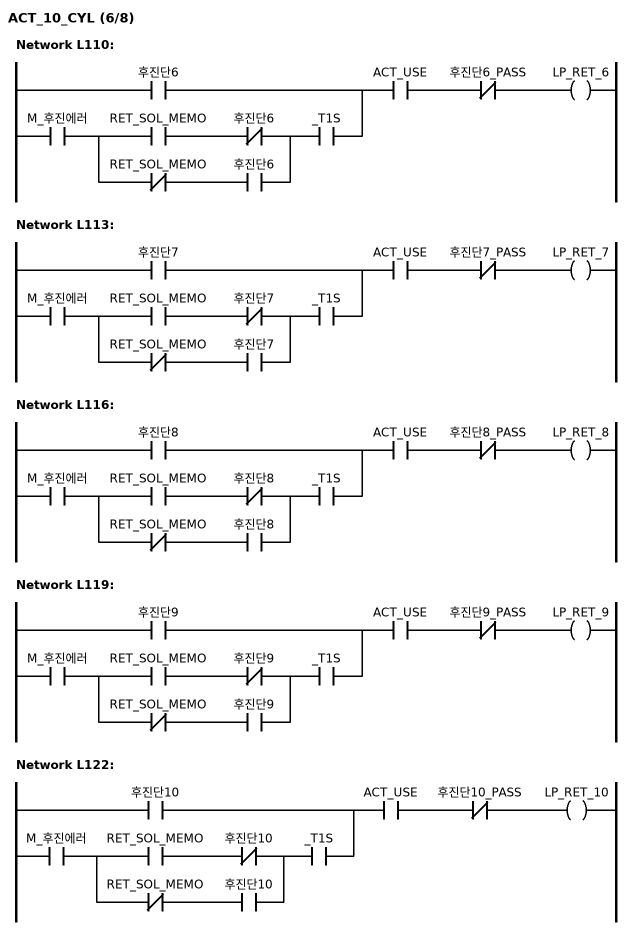
(* Rung L110 *)
LP_RET_6 := (후진단6 OR (M_후진에러 AND ((RET_SOL_MEMO AND NOT 후진단6) OR (NOT RET_SOL_MEMO AND 후진단6)) AND _T1S)) AND ACT_USE AND NOT 후진단6_PASS;
(* Rung L113 *)
LP_RET_7 := (후진단7 OR (M_후진에러 AND ((RET_SOL_MEMO AND NOT 후진단7) OR (NOT RET_SOL_MEMO AND 후진단7)) AND _T1S)) AND ACT_USE AND NOT 후진단7_PASS;
(* Rung L116 *)
LP_RET_8 := (후진단8 OR (M_후진에러 AND ((RET_SOL_MEMO AND NOT 후진단8) OR (NOT RET_SOL_MEMO AND 후진단8)) AND _T1S)) AND ACT_USE AND NOT 후진단8_PASS;
(* Rung L119 *)
LP_RET_9 := (후진단9 OR (M_후진에러 AND ((RET_SOL_MEMO AND NOT 후진단9) OR (NOT RET_SOL_MEMO AND 후진단9)) AND _T1S)) AND ACT_USE AND NOT 후진단9_PASS;
(* Rung L122 *)
LP_RET_10 := (후진단10 OR (M_후진에러 AND ((RET_SOL_MEMO AND NOT 후진단10) OR (NOT RET_SOL_MEMO AND 후진단10)) AND _T1S)) AND ACT_USE AND NOT 후진단10_PASS;

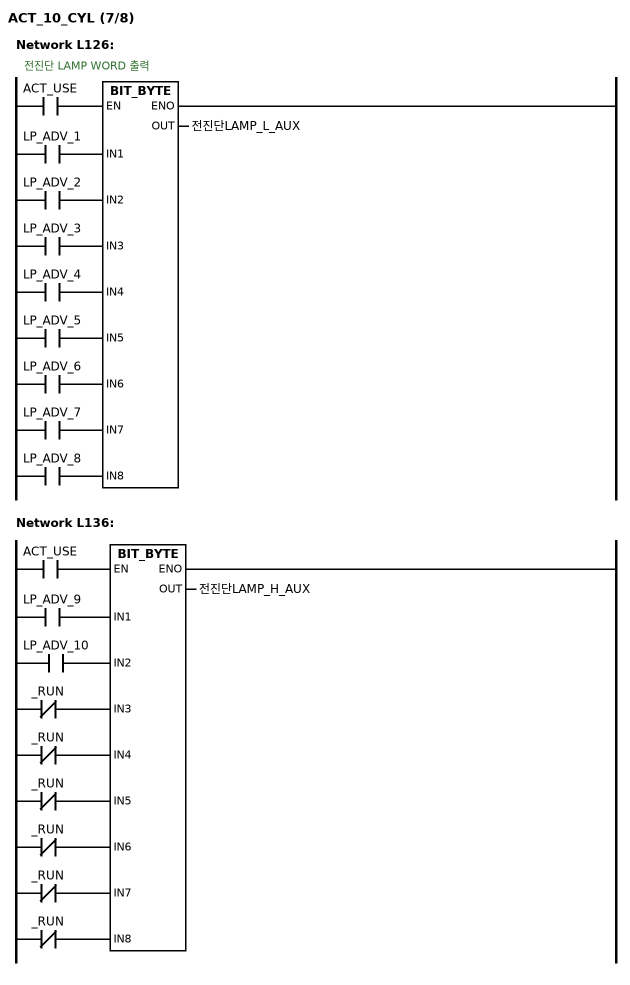
(* 전진단 LAMP WORD 출력 *)
(* Rung L126 *)
IF ACT_USE THEN
    전진단LAMP_L_AUX := BIT_BYTE(LP_ADV_1, LP_ADV_2, LP_ADV_3, LP_ADV_4, LP_ADV_5, LP_ADV_6, LP_ADV_7, LP_ADV_8);
END_IF;
(* Rung L136 *)
IF ACT_USE THEN
    전진단LAMP_H_AUX := BIT_BYTE(LP_ADV_9, LP_ADV_10, NOT _RUN, NOT _RUN, NOT _RUN, NOT _RUN, NOT _RUN, NOT _RUN);
END_IF;

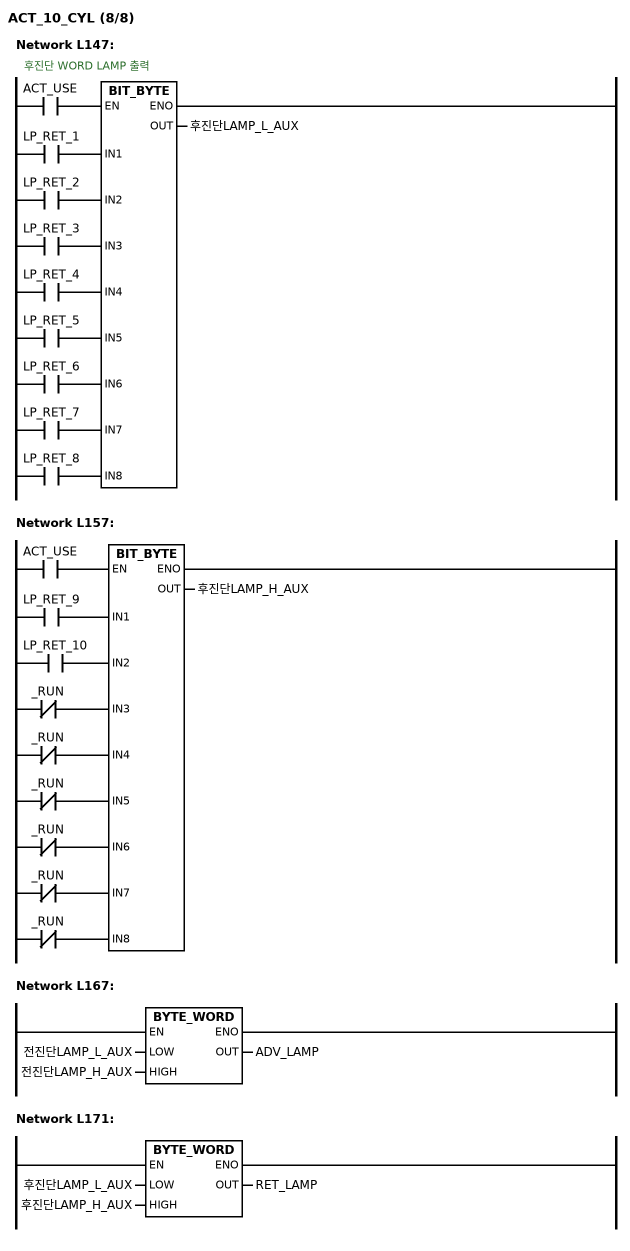
(* 후진단 WORD LAMP 출력 *)
(* Rung L147 *)
IF ACT_USE THEN
    후진단LAMP_L_AUX := BIT_BYTE(LP_RET_1, LP_RET_2, LP_RET_3, LP_RET_4, LP_RET_5, LP_RET_6, LP_RET_7, LP_RET_8);
END_IF;
(* Rung L157 *)
IF ACT_USE THEN
    후진단LAMP_H_AUX := BIT_BYTE(LP_RET_9, LP_RET_10, NOT _RUN, NOT _RUN, NOT _RUN, NOT _RUN, NOT _RUN, NOT _RUN);
END_IF;
(* Rung L167 *)
ADV_LAMP := BYTE_WORD(LOW := 전진단LAMP_L_AUX, HIGH := 전진단LAMP_H_AUX);
(* Rung L171 *)
RET_LAMP := BYTE_WORD(LOW := 후진단LAMP_L_AUX, HIGH := 후진단LAMP_H_AUX);
END_FUNCTION_BLOCK

FUNCTION_BLOCK ACT_6_CYL
VAR_INPUT
    사용유무 : BOOL;
    운전준비 : BOOL;
    전진보조 : BOOL;
    후진보조 : BOOL;
    전진단수량 : UINT;
    후진단수량 : UINT;
    전진단1 : BOOL;
    후진단1 : BOOL;
    전진단2 : BOOL;
    후진단2 : BOOL;
    전진단3 : BOOL;
    후진단3 : BOOL;
    전진단4 : BOOL;
    후진단4 : BOOL;
    전진단5 : BOOL;
    후진단5 : BOOL;
    전진단6 : BOOL;
    후진단6 : BOOL;
    전진단_지연시간 : TIME;
    후진단_지연시간 : TIME;
    LS_ERR1_지연시간 : TIME;
    LS_ERR2_지연시간 : TIME;
    이상리셋 : BOOL;
END_VAR
VAR_OUTPUT
    SOL_ADV_출력 : BOOL;
    SOL_RET_출력 : BOOL;
    M_전진단 : BOOL;
    M_후진단 : BOOL;
    M_전진에러 : BOOL;
    M_후진에러 : BOOL;
    ADV_LAMP : WORD;
    RET_LAMP : WORD;
END_VAR
VAR
    ACT_USE : BOOL;
    ADV_END_TIME : TON;
    ADV_SOL_MEMO : BOOL;
    ERR_TIME1 : TON;
    LP_ADV_1 : BOOL;
    LP_ADV_2 : BOOL;
    LP_ADV_3 : BOOL;
    LP_ADV_4 : BOOL;
    LP_ADV_5 : BOOL;
    LP_ADV_6 : BOOL;
    LP_RET_1 : BOOL;
    LP_RET_2 : BOOL;
    LP_RET_3 : BOOL;
    LP_RET_4 : BOOL;
    LP_RET_5 : BOOL;
    LP_RET_6 : BOOL;
    LS_ERR_1 : BOOL;
    LS_ERR_2 : BOOL;
    RET_END_TIME : TON;
    RET_ERR_TIME : TON;
    RET_SOL_MEMO : BOOL;
    ZERO_BYTE : BYTE;
    전진단2_PASS : BOOL;
    전진단3_PASS : BOOL;
    전진단4_PASS : BOOL;
    전진단5_PASS : BOOL;
    전진단6_PASS : BOOL;
    전진단LAMP_AUX : BYTE;
    후진단2_PASS : BOOL;
    후진단3_PASS : BOOL;
    후진단4_PASS : BOOL;
    후진단5_PASS : BOOL;
    후진단6_PASS : BOOL;
    후진단LAMP_AUX : BYTE;
END_VAR

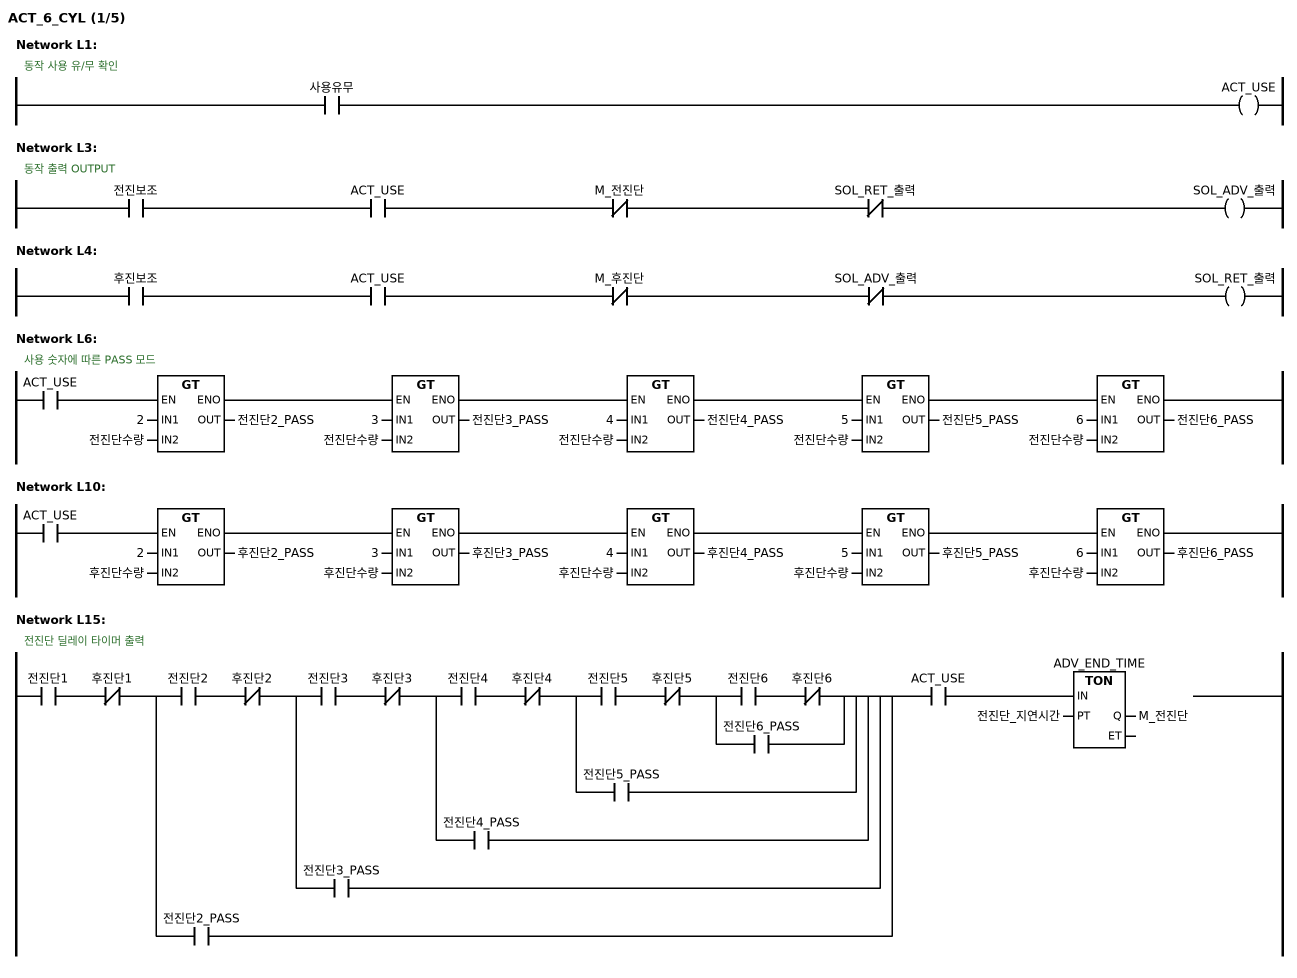
(* 동작 사용 유/무 확인 *)
(* Rung L1 *)
ACT_USE := 사용유무;
(* 동작 출력 OUTPUT *)
(* Rung L3 *)
SOL_ADV_출력 := 전진보조 AND ACT_USE AND NOT M_전진단 AND NOT SOL_RET_출력;
(* Rung L4 *)
SOL_RET_출력 := 후진보조 AND ACT_USE AND NOT M_후진단 AND NOT SOL_ADV_출력;
(* 사용 숫자에 따른 PASS 모드 *)
(* Rung L6 *)
IF ACT_USE THEN
    전진단2_PASS := 2 > 전진단수량;
    전진단3_PASS := 3 > 전진단수량;
    전진단4_PASS := 4 > 전진단수량;
    전진단5_PASS := 5 > 전진단수량;
    전진단6_PASS := 6 > 전진단수량;
END_IF;
(* Rung L10 *)
IF ACT_USE THEN
    후진단2_PASS := 2 > 후진단수량;
    후진단3_PASS := 3 > 후진단수량;
    후진단4_PASS := 4 > 후진단수량;
    후진단5_PASS := 5 > 후진단수량;
    후진단6_PASS := 6 > 후진단수량;
END_IF;
(* 전진단 딜레이 타이머 출력 *)
(* Rung L15 *)
ADV_END_TIME(IN := 전진단1 AND NOT 후진단1 AND ((전진단2 AND NOT 후진단2 AND ((전진단3 AND NOT 후진단3 AND ((전진단4 AND NOT 후진단4 AND ((전진단5 AND NOT 후진단5 AND ((전진단6 AND NOT 후진단6) OR 전진단6_PASS)) OR 전진단5_PASS)) OR 전진단4_PASS)) OR 전진단3_PASS)) OR 전진단2_PASS) AND ACT_USE, PT := 전진단_지연시간, Q => M_전진단);

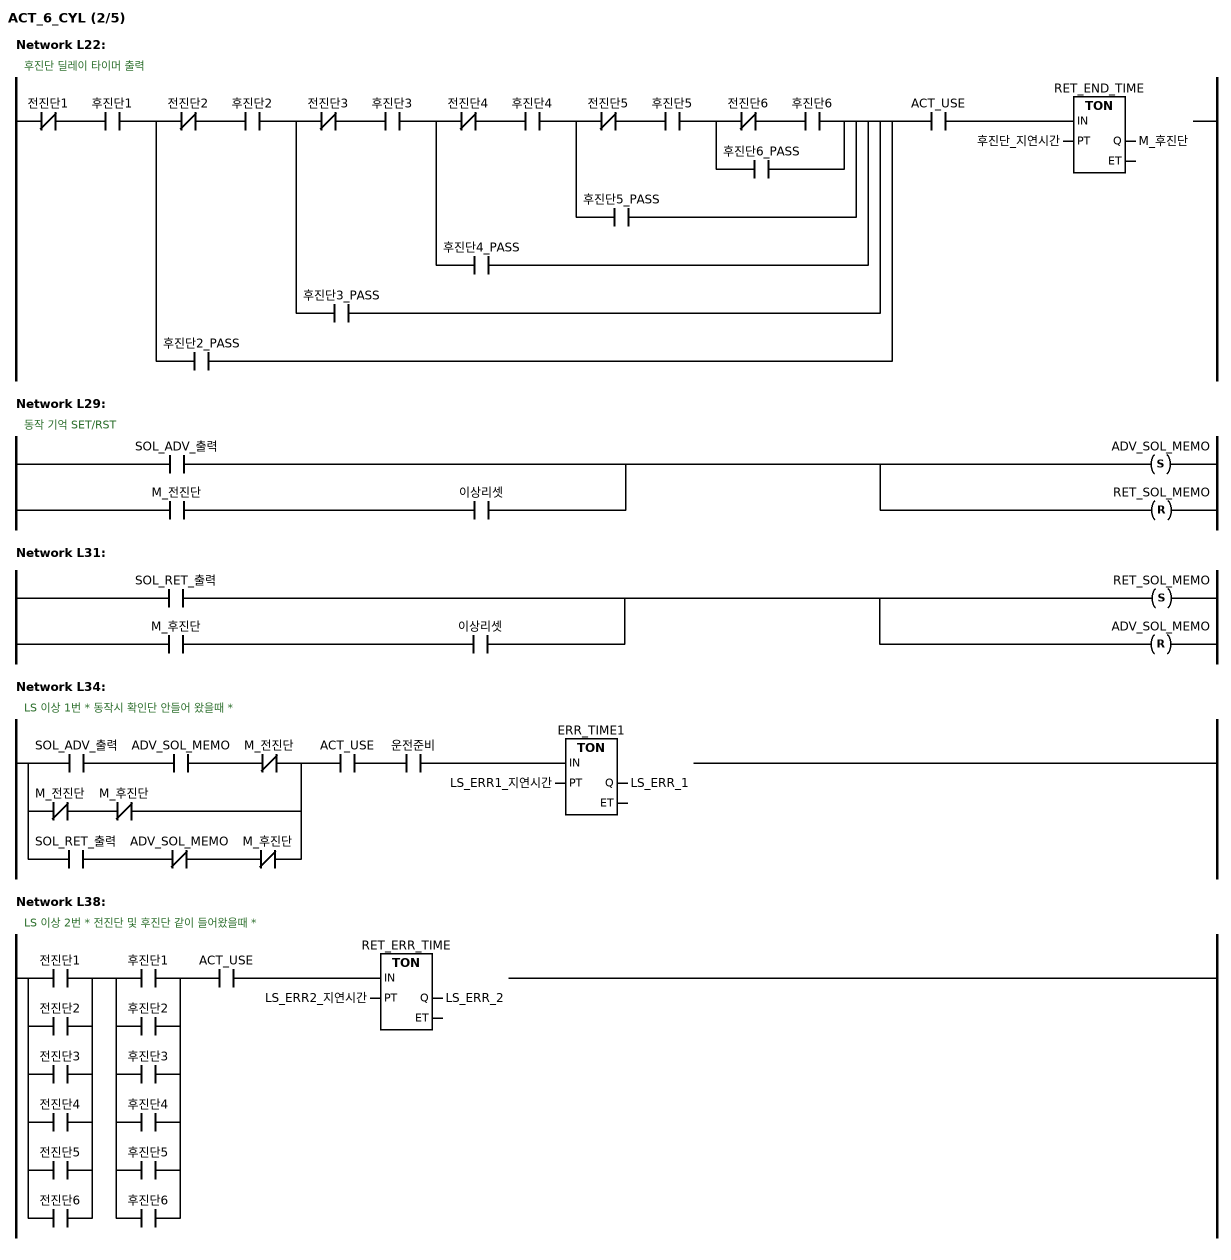
(* 후진단 딜레이 타이머 출력 *)
(* Rung L22 *)
RET_END_TIME(IN := NOT 전진단1 AND 후진단1 AND ((NOT 전진단2 AND 후진단2 AND ((NOT 전진단3 AND 후진단3 AND ((NOT 전진단4 AND 후진단4 AND ((NOT 전진단5 AND 후진단5 AND ((NOT 전진단6 AND 후진단6) OR 후진단6_PASS)) OR 후진단5_PASS)) OR 후진단4_PASS)) OR 후진단3_PASS)) OR 후진단2_PASS) AND ACT_USE, PT := 후진단_지연시간, Q => M_후진단);
(* 동작 기억 SET/RST *)
(* Rung L29 *)
IF SOL_ADV_출력 OR (M_전진단 AND 이상리셋) THEN
    ADV_SOL_MEMO := TRUE;
    RET_SOL_MEMO := FALSE;
END_IF;
(* Rung L31 *)
IF SOL_RET_출력 OR (M_후진단 AND 이상리셋) THEN
    RET_SOL_MEMO := TRUE;
    ADV_SOL_MEMO := FALSE;
END_IF;
(* LS 이상 1번 * 동작시 확인단 안들어 왔을때 * *)
(* Rung L34 *)
ERR_TIME1(IN := ((SOL_ADV_출력 AND ADV_SOL_MEMO AND NOT M_전진단) OR (NOT M_전진단 AND NOT M_후진단) OR (SOL_RET_출력 AND NOT ADV_SOL_MEMO AND NOT M_후진단)) AND ACT_USE AND 운전준비, PT := LS_ERR1_지연시간, Q => LS_ERR_1);
(* LS 이상 2번 * 전진단 및 후진단 같이 들어왔을때 * *)
(* Rung L38 *)
RET_ERR_TIME(IN := (전진단1 OR 전진단2 OR 전진단3 OR 전진단4 OR 전진단5 OR 전진단6) AND (후진단1 OR 후진단2 OR 후진단3 OR 후진단4 OR 후진단5 OR 후진단6) AND ACT_USE, PT := LS_ERR2_지연시간, Q => LS_ERR_2);

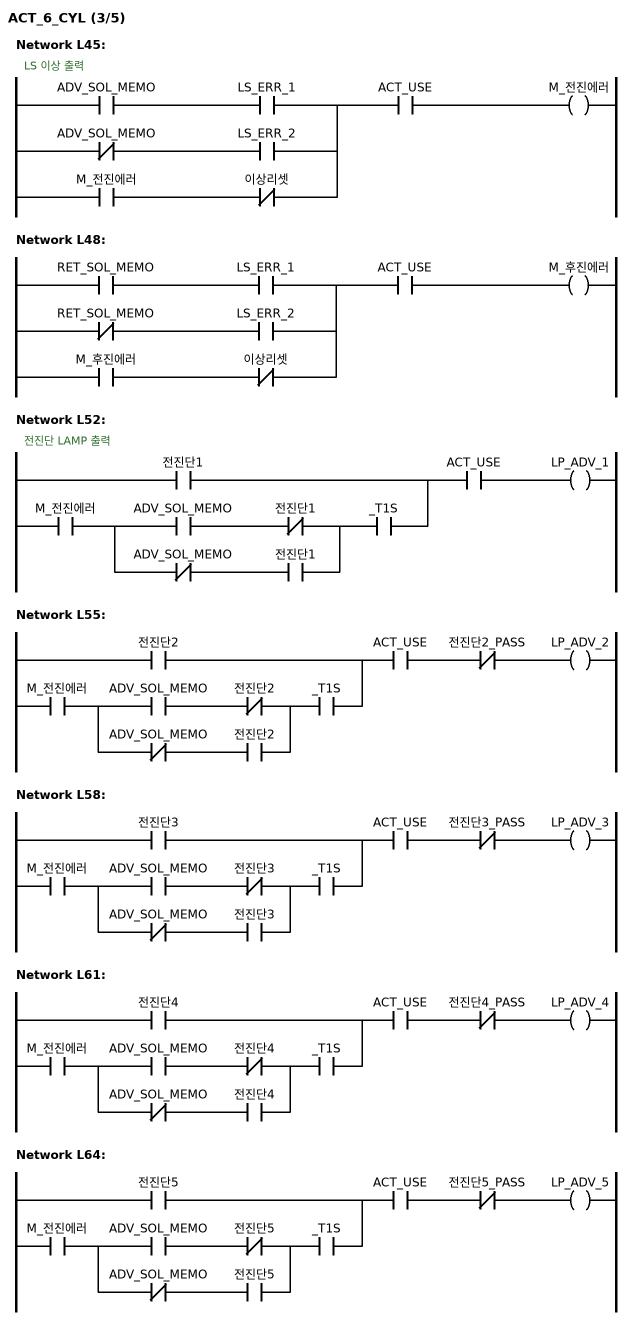
(* LS 이상 출력 *)
(* Rung L45 *)
M_전진에러 := ((ADV_SOL_MEMO AND LS_ERR_1) OR (NOT ADV_SOL_MEMO AND LS_ERR_2) OR (M_전진에러 AND NOT 이상리셋)) AND ACT_USE;
(* Rung L48 *)
M_후진에러 := ((RET_SOL_MEMO AND LS_ERR_1) OR (NOT RET_SOL_MEMO AND LS_ERR_2) OR (M_후진에러 AND NOT 이상리셋)) AND ACT_USE;
(* 전진단 LAMP 출력 *)
(* Rung L52 *)
LP_ADV_1 := (전진단1 OR (M_전진에러 AND ((ADV_SOL_MEMO AND NOT 전진단1) OR (NOT ADV_SOL_MEMO AND 전진단1)) AND _T1S)) AND ACT_USE;
(* Rung L55 *)
LP_ADV_2 := (전진단2 OR (M_전진에러 AND ((ADV_SOL_MEMO AND NOT 전진단2) OR (NOT ADV_SOL_MEMO AND 전진단2)) AND _T1S)) AND ACT_USE AND NOT 전진단2_PASS;
(* Rung L58 *)
LP_ADV_3 := (전진단3 OR (M_전진에러 AND ((ADV_SOL_MEMO AND NOT 전진단3) OR (NOT ADV_SOL_MEMO AND 전진단3)) AND _T1S)) AND ACT_USE AND NOT 전진단3_PASS;
(* Rung L61 *)
LP_ADV_4 := (전진단4 OR (M_전진에러 AND ((ADV_SOL_MEMO AND NOT 전진단4) OR (NOT ADV_SOL_MEMO AND 전진단4)) AND _T1S)) AND ACT_USE AND NOT 전진단4_PASS;
(* Rung L64 *)
LP_ADV_5 := (전진단5 OR (M_전진에러 AND ((ADV_SOL_MEMO AND NOT 전진단5) OR (NOT ADV_SOL_MEMO AND 전진단5)) AND _T1S)) AND ACT_USE AND NOT 전진단5_PASS;

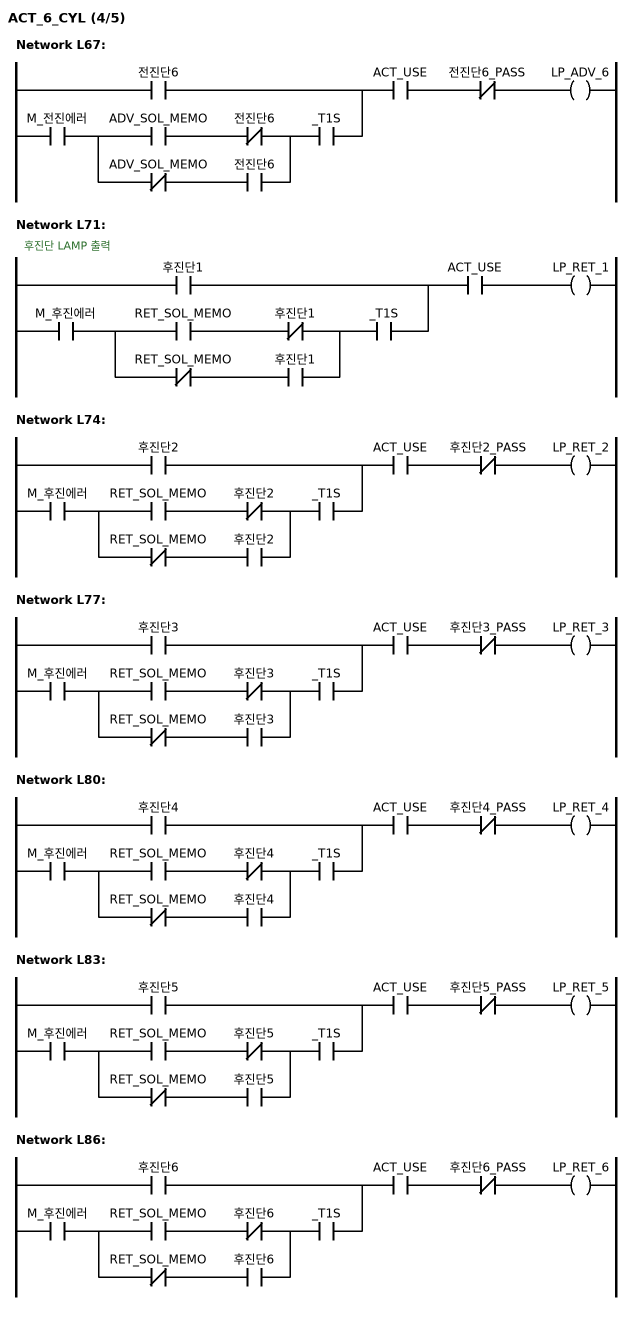
(* Rung L67 *)
LP_ADV_6 := (전진단6 OR (M_전진에러 AND ((ADV_SOL_MEMO AND NOT 전진단6) OR (NOT ADV_SOL_MEMO AND 전진단6)) AND _T1S)) AND ACT_USE AND NOT 전진단6_PASS;
(* 후진단 LAMP 출력 *)
(* Rung L71 *)
LP_RET_1 := (후진단1 OR (M_후진에러 AND ((RET_SOL_MEMO AND NOT 후진단1) OR (NOT RET_SOL_MEMO AND 후진단1)) AND _T1S)) AND ACT_USE;
(* Rung L74 *)
LP_RET_2 := (후진단2 OR (M_후진에러 AND ((RET_SOL_MEMO AND NOT 후진단2) OR (NOT RET_SOL_MEMO AND 후진단2)) AND _T1S)) AND ACT_USE AND NOT 후진단2_PASS;
(* Rung L77 *)
LP_RET_3 := (후진단3 OR (M_후진에러 AND ((RET_SOL_MEMO AND NOT 후진단3) OR (NOT RET_SOL_MEMO AND 후진단3)) AND _T1S)) AND ACT_USE AND NOT 후진단3_PASS;
(* Rung L80 *)
LP_RET_4 := (후진단4 OR (M_후진에러 AND ((RET_SOL_MEMO AND NOT 후진단4) OR (NOT RET_SOL_MEMO AND 후진단4)) AND _T1S)) AND ACT_USE AND NOT 후진단4_PASS;
(* Rung L83 *)
LP_RET_5 := (후진단5 OR (M_후진에러 AND ((RET_SOL_MEMO AND NOT 후진단5) OR (NOT RET_SOL_MEMO AND 후진단5)) AND _T1S)) AND ACT_USE AND NOT 후진단5_PASS;
(* Rung L86 *)
LP_RET_6 := (후진단6 OR (M_후진에러 AND ((RET_SOL_MEMO AND NOT 후진단6) OR (NOT RET_SOL_MEMO AND 후진단6)) AND _T1S)) AND ACT_USE AND NOT 후진단6_PASS;

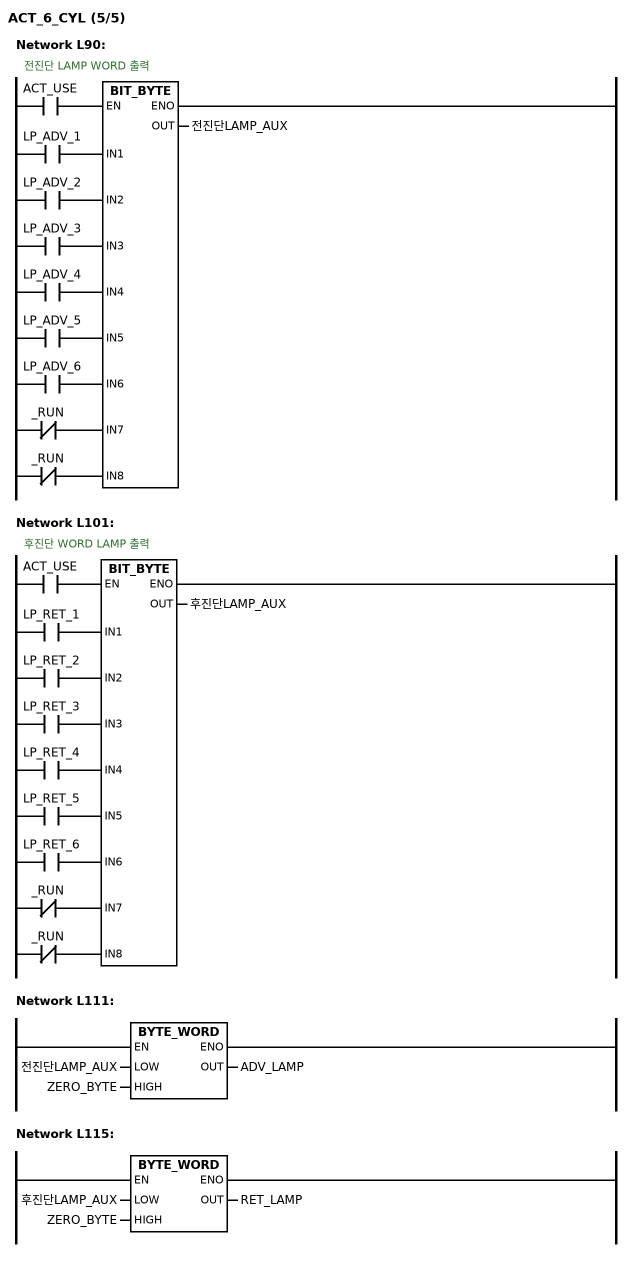
(* 전진단 LAMP WORD 출력 *)
(* Rung L90 *)
IF ACT_USE THEN
    전진단LAMP_AUX := BIT_BYTE(LP_ADV_1, LP_ADV_2, LP_ADV_3, LP_ADV_4, LP_ADV_5, LP_ADV_6, NOT _RUN, NOT _RUN);
END_IF;
(* 후진단 WORD LAMP 출력 *)
(* Rung L101 *)
IF ACT_USE THEN
    후진단LAMP_AUX := BIT_BYTE(LP_RET_1, LP_RET_2, LP_RET_3, LP_RET_4, LP_RET_5, LP_RET_6, NOT _RUN, NOT _RUN);
END_IF;
(* Rung L111 *)
ADV_LAMP := BYTE_WORD(LOW := 전진단LAMP_AUX, HIGH := ZERO_BYTE);
(* Rung L115 *)
RET_LAMP := BYTE_WORD(LOW := 후진단LAMP_AUX, HIGH := ZERO_BYTE);
END_FUNCTION_BLOCK

FUNCTION_BLOCK FB494_Robot_Hyundai_HMMI_v1
VAR_INPUT
    IN_START_Add : ARRAY[0..3] OF WORD;
    RBT_Prog_No : INT;
    X_Ready_On : BOOL;
    M_Auto : BOOL;
    T_START : TIME;
    M_START_OK : BOOL;
    M_Prog_OK : BOOL;
    M_RESTART_OK : BOOL;
    M_Stn_Fault : BOOL;
    M_Error_Rst : BOOL;
    M_Cycle_Set : BOOL;
    M_LAST_WK_COMP_RST : BOOL;
    M_ATD_OK : BOOL;
    M_TIP_CHANGE_START : BOOL;
    M_TIP_CHANGE_COMPL : BOOL;
    M_WATER_CUT_OFF : BOOL;
    M_BUZZ_STOP_AUX : BOOL;
    M_PLT_COUNT_RST_AUX : BOOL;
    M_GATE_CLOSED : BOOL;
    M_EM_STOP : BOOL;
    M_VIP_MODE : BOOL;
    M_TEST : BOOL;
    M_A_In_Ok : BOOL;
    M_B_In_Ok : BOOL;
    M_C_In_Ok : BOOL;
    M_D_In_Ok : BOOL;
    M_E_In_Ok : BOOL;
    M_F_In_Ok : BOOL;
    M_G_In_Ok : BOOL;
    M_H_In_Ok : BOOL;
    M_2nd_In_Ok : BOOL;
    M_3rd_In_Ok : BOOL;
    M_4th_In_Ok : BOOL;
    M_5th_In_Ok : BOOL;
    M_6th_In_Ok : BOOL;
    M_7th_In_Ok : BOOL;
    M_1st_Comp_Rst : BOOL;
    M_2nd_Comp_Rst : BOOL;
    M_3rd_Comp_Rst : BOOL;
    M_4th_Comp_Rst : BOOL;
    M_5th_Comp_Rst : BOOL;
    M_6th_Comp_Rst : BOOL;
    M_7th_Comp_Rst : BOOL;
    Mutual_Int1 : BOOL;
    Mutual_Int2 : BOOL;
    Mutual_Int3 : BOOL;
    Mutual_Int4 : BOOL;
    Mutual_Int5 : BOOL;
    Mutual_Int6 : BOOL;
    Mutual_Int7 : BOOL;
    Mutual_Int8 : BOOL;
    M_PLT1_In_Ok : BOOL;
    M_PLT2_In_Ok : BOOL;
    M_PLT3_In_Ok : BOOL;
    M_PLT4_In_Ok : BOOL;
    M_PLT5_In_Ok : BOOL;
    M_PLT6_In_Ok : BOOL;
    M_PLT7_In_Ok : BOOL;
    M_PLT8_In_Ok : BOOL;
    M_PLT9_In_Ok : BOOL;
    M_PLT10_In_Ok : BOOL;
    M_PLT11_In_Ok : BOOL;
    M_PLT12_In_Ok : BOOL;
END_VAR
VAR_OUTPUT
    OUT_Start_Add : ARRAY[0..3] OF WORD;
    M_RBT_Ready : BOOL;
    M_RBT_Auto : BOOL;
    M_RBT_Fault : BOOL;
    M_RBT_Home : BOOL;
    M_RBT_EM_Stop : BOOL;
    M_RBT_PAUSE : BOOL;
    M_RBT_PROGRAM_ERR : BOOL;
    M_RBT_PLC_RUN_CHK_ERR : BOOL;
    M_Last_Comp : BOOL;
    M_1st_Comp : BOOL;
    M_2nd_Comp : BOOL;
    M_3rd_Comp : BOOL;
    M_4th_Comp : BOOL;
    M_5th_Comp : BOOL;
    M_6th_Comp : BOOL;
    M_7th_Comp : BOOL;
    M_NO_INTF1 : BOOL;
    M_NO_INTF2 : BOOL;
    M_NO_INTF3 : BOOL;
    M_NO_INTF4 : BOOL;
    M_NO_INTF5 : BOOL;
    M_NO_INTF6 : BOOL;
    M_NO_INTF7 : BOOL;
    M_NO_INTF8 : BOOL;
    M_NO_INTF9 : BOOL;
    M_NO_INTF10 : BOOL;
    M_NO_INTF11 : BOOL;
    M_NO_INTF12 : BOOL;
END_VAR
VAR
    EM_STOP_DELAY : TOF;
    GATE_CLOSED_DELAY : TOF;
    Home_Delay : TON;
    IN_Add : ARRAY[0..3] OF WORD;
    M_RBT_Home_Aux : BOOL;
    OUT_Add : ARRAY[0..3] OF WORD;
    RBT_PLC_RUN_CHK_TIMER1 : TON;
    RBT_PLC_RUN_CHK_TIMER2 : TON;
    RBT_PRG_ARR : WORD;
    RBT_PRG_ECHO : INT;
    RBT_PRG_ECHO_ARR : WORD;
    RBT_PRG_Match_Ok : BOOL;
    RBT_RESTART : BOOL;
    RBT_START_Aux : BOOL;
    RBT_Start_Delay : TON;
    RBT_START_Off_DT : BOOL;
    RBT_Work_Rst_Aux : BOOL;
    RBT_X00_Home : BOOL;
    RBT_X01_LAST_WK_COMP : BOOL;
    RBT_X02_TOTAL_ERR : BOOL;
    RBT_X03_Ready_ON : BOOL;
    RBT_X04_Auto : BOOL;
    RBT_X05_Running : BOOL;
    RBT_X06_ABNORMAL_SEL : BOOL;
    RBT_X07_Tip_Dressing : BOOL;
    RBT_X08_EM_STOP : BOOL;
    RBT_X09_1ST_WK_COMP : BOOL;
    RBT_X10_2ND_WK_COMP : BOOL;
    RBT_X11_3RD_WK_COMP : BOOL;
    RBT_X12_4TH_WK_COMP : BOOL;
    RBT_X13_5TH_WK_COMP : BOOL;
    RBT_X14_6TH_WK_COMP : BOOL;
    RBT_X15_7TH_WK_COMP : BOOL;
    RBT_X16_NON_INTF1 : BOOL;
    RBT_X17_NON_INTF2 : BOOL;
    RBT_X18_NON_INTF3 : BOOL;
    RBT_X19_NON_INTF4 : BOOL;
    RBT_X20_NON_INTF5 : BOOL;
    RBT_X21_NON_INTF6 : BOOL;
    RBT_X22_NON_INTF7 : BOOL;
    RBT_X23_NON_INTF8 : BOOL;
    RBT_X24_NON_INTF9 : BOOL;
    RBT_X25_NON_INTF10 : BOOL;
    RBT_X26_NON_INTF11 : BOOL;
    RBT_X27_NON_INTF12 : BOOL;
    RBT_X28_SP : BOOL;
    RBT_X29_SP : BOOL;
    RBT_X30_SP : BOOL;
    RBT_X31_SP : BOOL;
    RBT_X32_Prog_Echo1 : BOOL;
    RBT_X33_Prog_Echo2 : BOOL;
    RBT_X34_Prog_Echo4 : BOOL;
    RBT_X35_Prog_Echo8 : BOOL;
    RBT_X36_Prog_Echo16 : BOOL;
    RBT_X37_Prog_Echo32 : BOOL;
    RBT_X38_Prog_Echo64 : BOOL;
    RBT_X39_Prog_Echo128 : BOOL;
    RBT_X40_TC_ERR : BOOL;
    RBT_X41_AIR_ERR : BOOL;
    RBT_X42_WATER_ERR : BOOL;
    RBT_X43_LS_ERR : BOOL;
    RBT_X44_COMM_ERR : BOOL;
    RBT_X45_SEALER_ERR : BOOL;
    RBT_X46_VISION_ERR : BOOL;
    RBT_X47_WELD_COUNT_ERR : BOOL;
    RBT_X48_MUTUAL_INT1 : BOOL;
    RBT_X49_MUTUAL_INT2 : BOOL;
    RBT_X50_MUTUAL_INT3 : BOOL;
    RBT_X51_MUTUAL_INT4 : BOOL;
    RBT_X52_MUTUAL_INT5 : BOOL;
    RBT_X53_MUTUAL_INT6 : BOOL;
    RBT_X54_MUTUAL_INT7 : BOOL;
    RBT_X55_MUTUAL_INT8 : BOOL;
    RBT_X56_SP : BOOL;
    RBT_X57_SP : BOOL;
    RBT_X58_PLT_COUNT_RST_COMPL : BOOL;
    RBT_X59_PLT_UNLOAD_COMPL : BOOL;
    RBT_X60_PLT_LAST_UNLOAD_COMPL : BOOL;
    RBT_X61_TIP_CHANGE : BOOL;
    RBT_X62_FLICKER_COMM_CHK : BOOL;
    RBT_X63_MOTOR_MC_ON : BOOL;
    RBT_Y00_Prog_SEL1 : BOOL;
    RBT_Y01_Prog_SEL2 : BOOL;
    RBT_Y02_Prog_SEL4 : BOOL;
    RBT_Y03_Prog_SEL8 : BOOL;
    RBT_Y04_Prog_SEL16 : BOOL;
    RBT_Y05_Prog_SEL32 : BOOL;
    RBT_Y06_Prog_SEL64 : BOOL;
    RBT_Y07_Prog_SEL128 : BOOL;
    RBT_Y08_WK_COMP_RST : BOOL;
    RBT_Y09_START : BOOL;
    RBT_Y10_Error_Rst : BOOL;
    RBT_Y11_EXT_READY : BOOL;
    RBT_Y12_ATD_START : BOOL;
    RBT_Y13_Pause : BOOL;
    RBT_Y14_EACH_WORK_COMPL_RST : BOOL;
    RBT_Y15_WATER_CUT_OFF : BOOL;
    RBT_Y16_A_1ST_IN_Ok : BOOL;
    RBT_Y17_B_1ST_IN_Ok : BOOL;
    RBT_Y18_C_1ST_IN_Ok : BOOL;
    RBT_Y19_D_1ST_IN_Ok : BOOL;
    RBT_Y20_E_1ST_IN_Ok : BOOL;
    RBT_Y21_F_1ST_IN_Ok : BOOL;
    RBT_Y22_G_1ST_IN_Ok : BOOL;
    RBT_Y23_H_1ST_IN_Ok : BOOL;
    RBT_Y24_2ND_IN_OK : BOOL;
    RBT_Y25_3RD_IN_OK : BOOL;
    RBT_Y26_4TH_IN_OK : BOOL;
    RBT_Y27_5TH_IN_OK : BOOL;
    RBT_Y28_6TH_IN_OK : BOOL;
    RBT_Y29_7TH_IN_OK : BOOL;
    RBT_Y30_SP : BOOL;
    RBT_Y31_SP : BOOL;
    RBT_Y32_PLT1_IN_OK : BOOL;
    RBT_Y33_PLT2_IN_OK : BOOL;
    RBT_Y34_PLT3_IN_OK : BOOL;
    RBT_Y35_PLT4_IN_OK : BOOL;
    RBT_Y36_PLT5_IN_OK : BOOL;
    RBT_Y37_PLT6_IN_OK : BOOL;
    RBT_Y38_PLT7_IN_OK : BOOL;
    RBT_Y39_PLT8_IN_OK : BOOL;
    RBT_Y40_PLT9_IN_OK : BOOL;
    RBT_Y41_PLT10_IN_OK : BOOL;
    RBT_Y42_PLT11_IN_OK : BOOL;
    RBT_Y43_PLT12_IN_OK : BOOL;
    RBT_Y44_SP : BOOL;
    RBT_Y45_SP : BOOL;
    RBT_Y46_SP : BOOL;
    RBT_Y47_TEST : BOOL;
    RBT_Y48_MUTUAL_INT1 : BOOL;
    RBT_Y49_MUTUAL_INT2 : BOOL;
    RBT_Y50_MUTUAL_INT3 : BOOL;
    RBT_Y51_MUTUAL_INT4 : BOOL;
    RBT_Y52_MUTUAL_INT5 : BOOL;
    RBT_Y53_MUTUAL_INT6 : BOOL;
    RBT_Y54_MUTUAL_INT7 : BOOL;
    RBT_Y55_MUTUAL_INT8 : BOOL;
    RBT_Y56_TIP_CHANGE_START : BOOL;
    RBT_Y57_TIP_CHANGE_END : BOOL;
    RBT_Y58_PLT_COUNT_RST : BOOL;
    RBT_Y59_GATE_CLOSED : BOOL;
    RBT_Y60_EM_STOP : BOOL;
    RBT_Y61_BUZZ_STOP : BOOL;
    RBT_Y62_FLICKER_COMM_CHK : BOOL;
    RBT_Y63_VIP_MODE : BOOL;
    Start_off_Delay : TON;
END_VAR
VAR
    _t1 : BOOL;
    _t2 : BOOL;
    _t3 : BOOL;
    _t4 : BOOL;
    _t5 : BOOL;
    _t6 : BOOL;
    _t7 : BOOL;
    _t8 : BOOL;
END_VAR

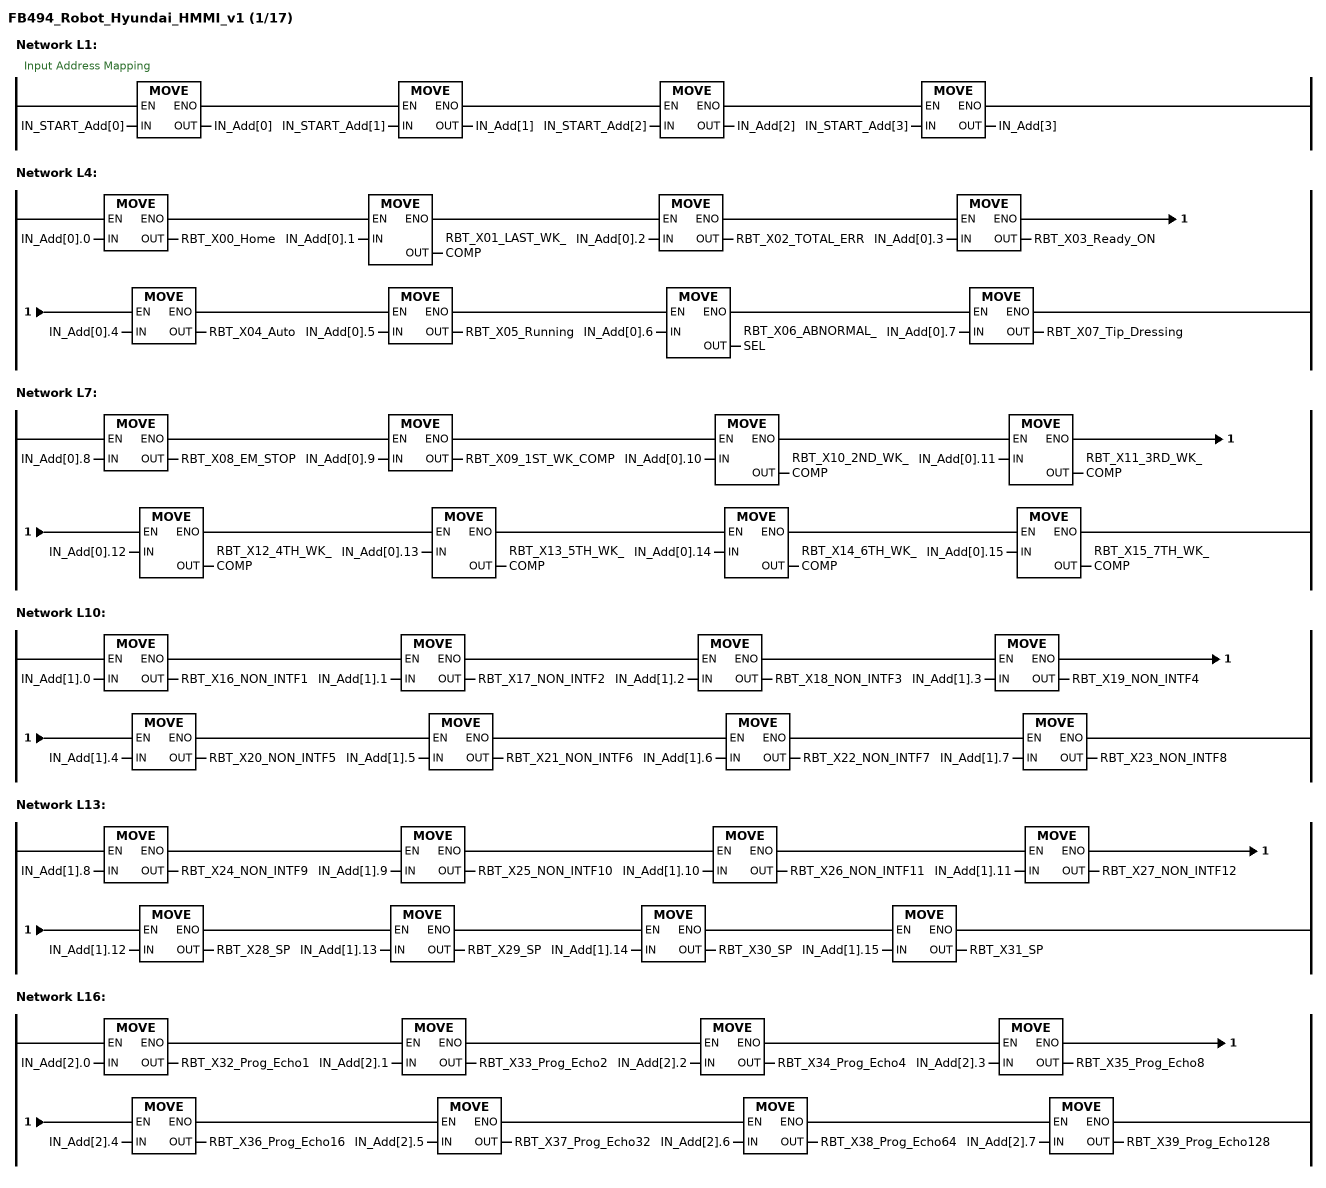
(* Input Address Mapping *)
(* Rung L1 *)
IN_Add[0] := IN_START_Add[0];
IN_Add[1] := IN_START_Add[1];
IN_Add[2] := IN_START_Add[2];
IN_Add[3] := IN_START_Add[3];
(* Rung L4 *)
RBT_X00_Home := IN_Add[0].0;
RBT_X01_LAST_WK_COMP := IN_Add[0].1;
RBT_X02_TOTAL_ERR := IN_Add[0].2;
RBT_X03_Ready_ON := IN_Add[0].3;
RBT_X04_Auto := IN_Add[0].4;
RBT_X05_Running := IN_Add[0].5;
RBT_X06_ABNORMAL_SEL := IN_Add[0].6;
RBT_X07_Tip_Dressing := IN_Add[0].7;
(* Rung L7 *)
RBT_X08_EM_STOP := IN_Add[0].8;
RBT_X09_1ST_WK_COMP := IN_Add[0].9;
RBT_X10_2ND_WK_COMP := IN_Add[0].10;
RBT_X11_3RD_WK_COMP := IN_Add[0].11;
RBT_X12_4TH_WK_COMP := IN_Add[0].12;
RBT_X13_5TH_WK_COMP := IN_Add[0].13;
RBT_X14_6TH_WK_COMP := IN_Add[0].14;
RBT_X15_7TH_WK_COMP := IN_Add[0].15;
(* Rung L10 *)
RBT_X16_NON_INTF1 := IN_Add[1].0;
RBT_X17_NON_INTF2 := IN_Add[1].1;
RBT_X18_NON_INTF3 := IN_Add[1].2;
RBT_X19_NON_INTF4 := IN_Add[1].3;
RBT_X20_NON_INTF5 := IN_Add[1].4;
RBT_X21_NON_INTF6 := IN_Add[1].5;
RBT_X22_NON_INTF7 := IN_Add[1].6;
RBT_X23_NON_INTF8 := IN_Add[1].7;
(* Rung L13 *)
RBT_X24_NON_INTF9 := IN_Add[1].8;
RBT_X25_NON_INTF10 := IN_Add[1].9;
RBT_X26_NON_INTF11 := IN_Add[1].10;
RBT_X27_NON_INTF12 := IN_Add[1].11;
RBT_X28_SP := IN_Add[1].12;
RBT_X29_SP := IN_Add[1].13;
RBT_X30_SP := IN_Add[1].14;
RBT_X31_SP := IN_Add[1].15;
(* Rung L16 *)
RBT_X32_Prog_Echo1 := IN_Add[2].0;
RBT_X33_Prog_Echo2 := IN_Add[2].1;
RBT_X34_Prog_Echo4 := IN_Add[2].2;
RBT_X35_Prog_Echo8 := IN_Add[2].3;
RBT_X36_Prog_Echo16 := IN_Add[2].4;
RBT_X37_Prog_Echo32 := IN_Add[2].5;
RBT_X38_Prog_Echo64 := IN_Add[2].6;
RBT_X39_Prog_Echo128 := IN_Add[2].7;

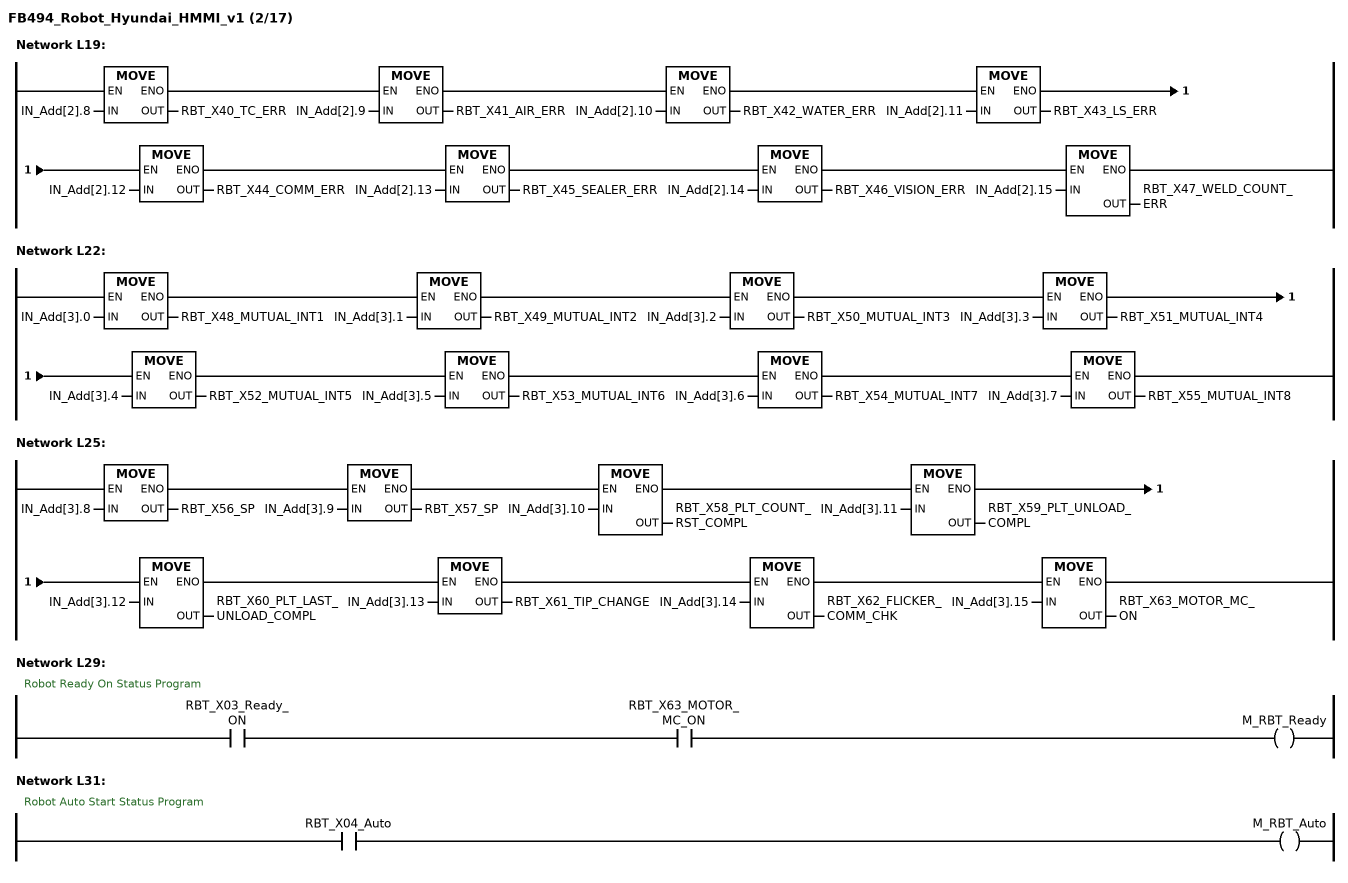
(* Rung L19 *)
RBT_X40_TC_ERR := IN_Add[2].8;
RBT_X41_AIR_ERR := IN_Add[2].9;
RBT_X42_WATER_ERR := IN_Add[2].10;
RBT_X43_LS_ERR := IN_Add[2].11;
RBT_X44_COMM_ERR := IN_Add[2].12;
RBT_X45_SEALER_ERR := IN_Add[2].13;
RBT_X46_VISION_ERR := IN_Add[2].14;
RBT_X47_WELD_COUNT_ERR := IN_Add[2].15;
(* Rung L22 *)
RBT_X48_MUTUAL_INT1 := IN_Add[3].0;
RBT_X49_MUTUAL_INT2 := IN_Add[3].1;
RBT_X50_MUTUAL_INT3 := IN_Add[3].2;
RBT_X51_MUTUAL_INT4 := IN_Add[3].3;
RBT_X52_MUTUAL_INT5 := IN_Add[3].4;
RBT_X53_MUTUAL_INT6 := IN_Add[3].5;
RBT_X54_MUTUAL_INT7 := IN_Add[3].6;
RBT_X55_MUTUAL_INT8 := IN_Add[3].7;
(* Rung L25 *)
RBT_X56_SP := IN_Add[3].8;
RBT_X57_SP := IN_Add[3].9;
RBT_X58_PLT_COUNT_RST_COMPL := IN_Add[3].10;
RBT_X59_PLT_UNLOAD_COMPL := IN_Add[3].11;
RBT_X60_PLT_LAST_UNLOAD_COMPL := IN_Add[3].12;
RBT_X61_TIP_CHANGE := IN_Add[3].13;
RBT_X62_FLICKER_COMM_CHK := IN_Add[3].14;
RBT_X63_MOTOR_MC_ON := IN_Add[3].15;
(* Robot Ready On Status Program *)
(* Rung L29 *)
M_RBT_Ready := RBT_X03_Ready_ON AND RBT_X63_MOTOR_MC_ON;
(* Robot Auto Start Status Program *)
(* Rung L31 *)
M_RBT_Auto := RBT_X04_Auto;

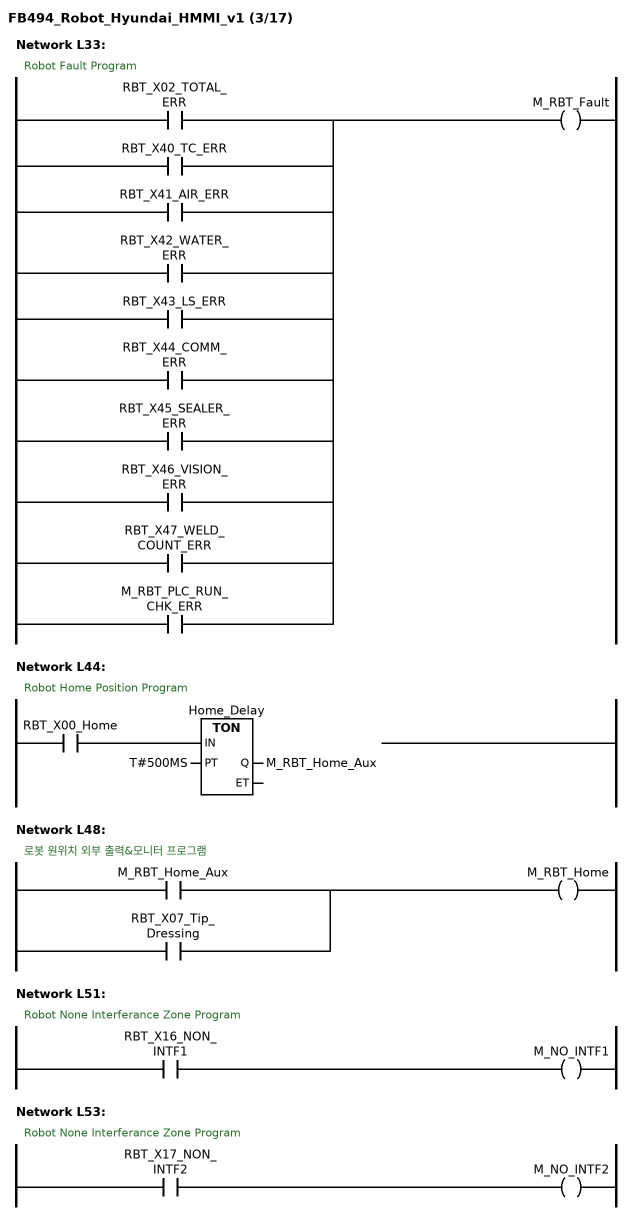
(* Robot Fault Program *)
(* Rung L33 *)
M_RBT_Fault := RBT_X02_TOTAL_ERR OR RBT_X40_TC_ERR OR RBT_X41_AIR_ERR OR RBT_X42_WATER_ERR OR RBT_X43_LS_ERR OR RBT_X44_COMM_ERR OR RBT_X45_SEALER_ERR OR RBT_X46_VISION_ERR OR RBT_X47_WELD_COUNT_ERR OR M_RBT_PLC_RUN_CHK_ERR;
(* Robot Home Position Program *)
(* Rung L44 *)
Home_Delay(IN := RBT_X00_Home, PT := T#500MS, Q => M_RBT_Home_Aux);
(* 로봇 원위치 외부 출력&모니터 프로그램 *)
(* Rung L48 *)
M_RBT_Home := M_RBT_Home_Aux OR RBT_X07_Tip_Dressing;
(* Robot None Interferance Zone Program *)
(* Rung L51 *)
M_NO_INTF1 := RBT_X16_NON_INTF1;
(* Robot None Interferance Zone Program *)
(* Rung L53 *)
M_NO_INTF2 := RBT_X17_NON_INTF2;

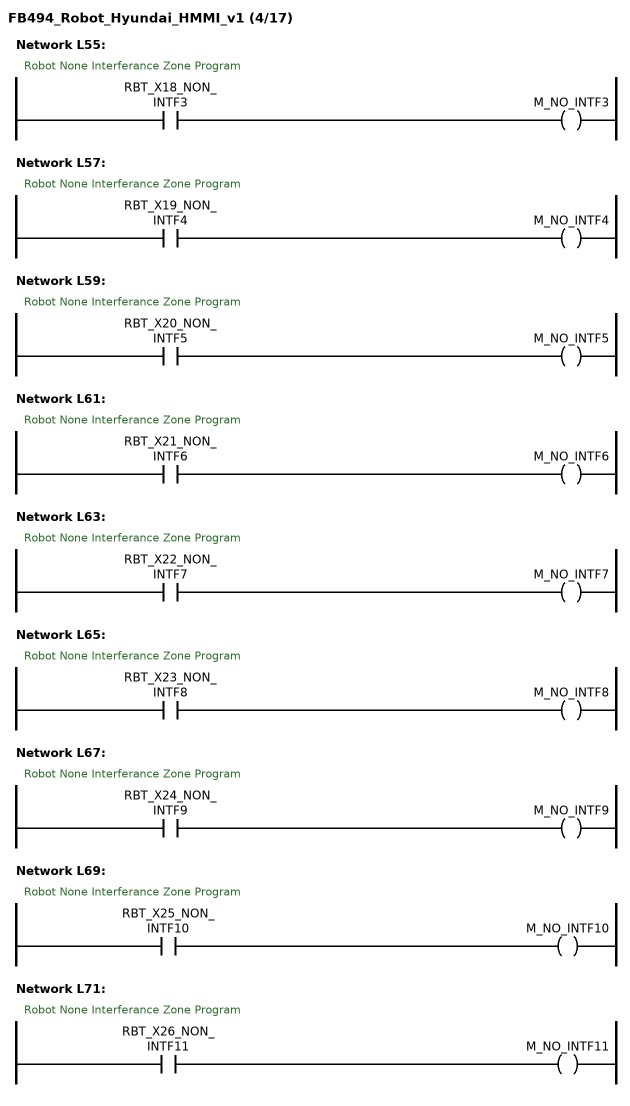
(* Robot None Interferance Zone Program *)
(* Rung L55 *)
M_NO_INTF3 := RBT_X18_NON_INTF3;
(* Robot None Interferance Zone Program *)
(* Rung L57 *)
M_NO_INTF4 := RBT_X19_NON_INTF4;
(* Robot None Interferance Zone Program *)
(* Rung L59 *)
M_NO_INTF5 := RBT_X20_NON_INTF5;
(* Robot None Interferance Zone Program *)
(* Rung L61 *)
M_NO_INTF6 := RBT_X21_NON_INTF6;
(* Robot None Interferance Zone Program *)
(* Rung L63 *)
M_NO_INTF7 := RBT_X22_NON_INTF7;
(* Robot None Interferance Zone Program *)
(* Rung L65 *)
M_NO_INTF8 := RBT_X23_NON_INTF8;
(* Robot None Interferance Zone Program *)
(* Rung L67 *)
M_NO_INTF9 := RBT_X24_NON_INTF9;
(* Robot None Interferance Zone Program *)
(* Rung L69 *)
M_NO_INTF10 := RBT_X25_NON_INTF10;
(* Robot None Interferance Zone Program *)
(* Rung L71 *)
M_NO_INTF11 := RBT_X26_NON_INTF11;

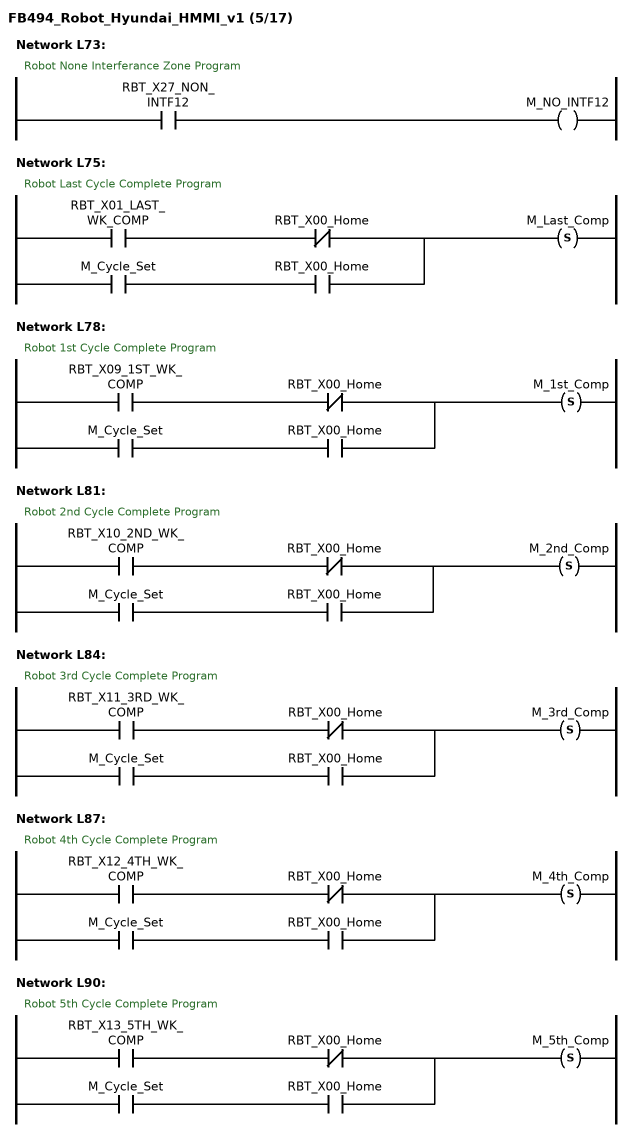
(* Robot None Interferance Zone Program *)
(* Rung L73 *)
M_NO_INTF12 := RBT_X27_NON_INTF12;
(* Robot Last Cycle Complete Program *)
(* Rung L75 *)
IF (RBT_X01_LAST_WK_COMP AND NOT RBT_X00_Home) OR (M_Cycle_Set AND RBT_X00_Home) THEN
    M_Last_Comp := TRUE;
END_IF;
(* Robot 1st Cycle Complete Program *)
(* Rung L78 *)
IF (RBT_X09_1ST_WK_COMP AND NOT RBT_X00_Home) OR (M_Cycle_Set AND RBT_X00_Home) THEN
    M_1st_Comp := TRUE;
END_IF;
(* Robot 2nd Cycle Complete Program *)
(* Rung L81 *)
IF (RBT_X10_2ND_WK_COMP AND NOT RBT_X00_Home) OR (M_Cycle_Set AND RBT_X00_Home) THEN
    M_2nd_Comp := TRUE;
END_IF;
(* Robot 3rd Cycle Complete Program *)
(* Rung L84 *)
IF (RBT_X11_3RD_WK_COMP AND NOT RBT_X00_Home) OR (M_Cycle_Set AND RBT_X00_Home) THEN
    M_3rd_Comp := TRUE;
END_IF;
(* Robot 4th Cycle Complete Program *)
(* Rung L87 *)
IF (RBT_X12_4TH_WK_COMP AND NOT RBT_X00_Home) OR (M_Cycle_Set AND RBT_X00_Home) THEN
    M_4th_Comp := TRUE;
END_IF;
(* Robot 5th Cycle Complete Program *)
(* Rung L90 *)
IF (RBT_X13_5TH_WK_COMP AND NOT RBT_X00_Home) OR (M_Cycle_Set AND RBT_X00_Home) THEN
    M_5th_Comp := TRUE;
END_IF;

